(* CODESYS project kr_achse.library
   Title: Kr_Achse
   Version: 2.23.0.7
   Placeholder: Kr_Achse
   Company: Progress

Project tree, tasks and I/O mapping:
  libraries: Tc2_Standard, * (Beckhoff Automation GmbH)
  Data types/
    Achsen/
      data type TAchs_To_DriveAdapter
      data type TES_Achse_IN
      data type TES_Achse_OUT
      data type TIV_RB
      data type TKont_Achse_IN
      data type TKont_Achse_OUT
      data type TPDO_SI6_IN
      data type TPDO_SI6_OUT
      data type TPDO_SI6_V3_IN
      data type TPDO_SI6_V3_OUT
  POUs/
    Achsen_Bausteinen/
      Adapter/
        function block Adapter_Drive_Analog [ST]
        function block Adapter_Drive_BeckhoffEL7201 [ST]
        function block Adapter_Drive_MDS [ST]
        function block Adapter_Drive_SI6 [ST]
        function block Adapter_Drive_SI6_V3 [ST]
        function block Adapter_DriveBased_U [ST]
      FB/
        function block Bremsweg [FBD]
        function block calc_Rbist_inPhase3 [ST]
        function block calc_Val3_inPhase123 [ST]
        function block calc_Val567_inPhase45 [ST]
        function block calc_Val67_inPhase6 [ST]
        function block calc_Val7_inPhase7 [ST]
        function block CDLR [ST]
        function block Phase0 [FBD]
        function block Phase12 [FBD]
        function block Phase3 [FBD]
        function block Phase4 [FBD]
        function block Phase56 [FBD]
        function block Phase7 [FBD]
        function block switchPhase [ST]
        function block Trnsf1Lreal [ST]
      function block ES_AnalogIN [ST]
      function block ES_EL5001_A [ST]
      function block ES_EL5xx1_A [ST]
      function block ES_KL2552 [ST]
      function block ES_KL5001_A [ST]
      function block ES_KL51x1_A [ST]
      function block ES_M3120 [ST]
      function block KR_Achse_V2 [FBD]: encoder, ohne_RB, Regelung
    Nockenachsen/
      function block Nock_Incr_S_Achs [ST]
  Visualizations/
*)

// Data types/Achsen/TAchs_To_DriveAdapter
TYPE TAchs_To_DriveAdapter :
STRUCT
	motorSpeed:REAL; (*rpm*)
	SA_MotUmdr:REAL;(*Schleppabstand in Motorumdrehungen zur berechnung des IPM-Mod bei ext. Encoder  (Adapter_Drive_MDS_ExtEnc). !!! Der Schleppabstand beinhaltet schon das Vorzeichen aufgrund Achse Invers/ Not Invers !!! *)
END_STRUCT
END_TYPE

// Data types/Achsen/TES_Achse_IN
TYPE TES_Achse_IN :
STRUCT
(*#################### EingangsVariablen: NC-Baustein -> STRUKTUR(IN) -> ANWENDER-PRG. ###################################*)
	IstPos: LREAL;(*Istposition Achse *)
	SYNC: BOOL:= FALSE;
	STILL:BOOL;(*Stillstand:Dises Bit ist TRUE, wenn bei gesetztem Ausgang VOR(ZUR) der Istwert nicht größer (nicht kleiner) wird*)
	PEH:BOOL;(*Position erreicht: wird ausgegeben, solange sich der Antrieb innerhalb dem PEH-Fenster befindet*)
	RET_SollPos:LREAL;(*Rückmeldung der übergebenen Sollposition*)
	VEL_IST:REAL;(*Istwert der Geschwindigkeit: -2,-1,0,1,2 (schnell zurück, langsam zurück, steht, langsam vor, schnell vor*)
END_STRUCT
END_TYPE

// Data types/Achsen/TES_Achse_OUT
TYPE TES_Achse_OUT :
STRUCT
(*############ OUT-VARIABLEN: ANWENDER-PRG. -> STRUKTUR(OUT) -> NC-Baustein ################################*)
	MODULO:BOOL;(*Modulowert ermitteln, es müssen die Incrmente für Modulowert angegeben werden. Achtung:MODULO-Funktion wird vom Baustein nur gemacht, solange die Incrementezahl ( IstPos/IBW) kleiner den Grenzen eines DINT ist, andernfalls wird MOD ignoriert*)
	MODULOVAL_INC:REAL;(*Wert in Incrementen für MODULO-Funktion*)
	SETPOS:BOOL;(*Istposition auf "Refpos" setzen *)
	REF:BOOL; (*Anwahl der Referenzfahrt unter beachtung von REFVEL1,REFVEL2 (VAR_IN am FB) und Modus "REF_ON" *)
	Refpos: REAL; (*Wert für "REF" und "SETPOS" *)
	Start_Pos: BOOL;(*Start-Bit zur Positionierung. *)
	SollPos: LREAL;(*Zielposition bei Positionierung*)
	V_Pos:REAL:=2.0;(*Geschwindigkeit beim Positionieren: 1= nur schleich,2= EIL-Schleich
						!! bei Verwendung der DC-Klemme KL2552 als ES-Achse wird hier die Geschwindigkeit in % angegeben !! *)
	JOGFW: BOOL;(*Manuell vor*)
	JOGBW: BOOL;(*manuell zurück*)
	V_JOG: REAL:=1.0;(*manuelle Geschwindigkeit: 1=langsam, 2=schnell
					!! bei Verwendung der DC-Klemme KL2552 als ES-Achse wird hier die Geschwindigkeit in % angegeben !! Beim Positioniervorgang wird hier die Schleichgeschwindigkeit angegeben !!! *)
END_STRUCT
END_TYPE

// Data types/Achsen/TIV_RB
TYPE TIV_RB :
STRUCT
	Phase:INT;(*akutelle Phase: 0 = Stillstand / 1..7 = Fahrt vorwärts / -1..-7 = Fahrt rückwärts*)
	PhCng:INT;(*aktuelle Phase x100 /letztePhase x10 / Ursache des Phasenwechsels x1:

071=Phase 0 wurde aus Phase 7 eingeleitet
  da das Ziel mit VE7=0 erreicht war.
072=Phase 0 wurde aus Phase 7 eingeleitet
   da ACC=0 und VEL=0 waren, das Ziel war nicht erreicht oder es war nicht Start_Pos gesetzt 
073=Phase 0 wurde aus Phase 7 eingeleitet da Fehler in Phase 7 auftrat (Geschw. 0 oder ACC=0 wurde nicht erreicht

0X8 = Phase=0 aus PhaseX gesetzt da Ruck=0, Stillstand, 
  Fehler oder abbruch durch anderen Achsbefehl vorliegt

101=Phase 1 wurde aus Phase 0 eingeleitet da Ziel in positiver richtung liegt
102=Phase -1 wurde aus Phase 0 eingeleitet da Ziel in negativer richtung liegt

123=Phase 1 wurde aus Phase 2 eingeleitet da Acc höher geworden ist

131=Phase 1 wurde aus Phase 3 eingeleitet
  da weder Ziel noch VEL_Soll noch ACC_Soll erreicht ist/wird
141=Phase 1 wurde eingeleitet weil Sollgeschw. unterschritten war 


2x1=Phase 2 wurde eingeleitet da die Sollbeschleunigung erreicht ist
311=Phase 3 wurde aus Phase1 eingeleitet da VE3 den Wert für V_Pos erreicht hat
321=Phase 3 wurde aus Phase2 eingeleitet da VE3 den Wert für V_Pos erreicht hat

312=Phase 3 wurde aus Ph.1 eingeleitet da der Resverfahrweg aufgebraucht ist
322=Phase 3 wurde aus Ph.2 eingeleitet da der Resverfahrweg aufgebraucht ist

313=Phase 3 wurde aus Ph.1 eingeleitet da die 
323=Phase 3 wurde aus Ph.2 eingeleitet da die 
 Istbeschleunigung höher ist als die Vorgegebene ACC-Soll.

431=Phase 4 wurde aus Phase 3 eingeleitet
 da die Istbeschleunigung=0 ist
472=Phase 4 wurde aus Phase 7 eingeleitet
  da ACC_IST=0 aber VE7>0

541=Phase 5 wurde aus Phase 4 eingeleitet weil Zieldiff aufbegraucht war
542=Phase 5 wurde eingeleitet weil Sollgeschw. überschritten war 
563=Phase 5 wurde aus Phase 6 eingeleitet weil kein Befehl ansteht und (dadurch) die Bremsrampe steiler geworden ist
573=Phase 5 wurde aus Phase 7 eingeleitet weil VE7>0 und das Ziel überschritten würde
574=Phase 5 wurde aus Phase 7 eingeleitet weil VE7>0 und VE7>sollvel
535=Phase 5 wurde aus Phase 3 eingeleitet weil Restweg aufgebraucht war und ACC_IST im nächsten Zyklus < 0 war


651=Phase 6 wurde aus Phase 5 eingeleitet da die Soll-DCC erreicht war

751=Phase 7 wurde aus Ph.5 eingeleitet
 da VE7=0 erreicht wird (VE7 darf nicht neg. werden) 
761=Phase 7 wurde aus Ph.6 eingeleitet da
  da VE7=0 erreicht wird (VE7 darf nicht neg. werden) 
752=Phase 7 wurde aus Ph.5 eingeleitet da da nicht das Ziel, aber da die Sollgeschwindigkeit VE7=V_Soll und VE7>0 erreicht wird (Online-Änder. von V_soll durch niedrigeren Wert)
762=Phase 7 wurde aus Ph.6 eingeleitet da da nicht das Ziel, aber da die Sollgeschwindigkeit VE7=V_Soll und VE7>0 erreicht wird (Online-Änder. von V_soll durch niedrigeren Wert)
753=Phase 7 wurde aus Ph.5 eingeleitet da da nicht das Ziel, aber da die Sollbeschleunigung überschritten ist
763=Phase 7 wurde aus Ph.6 eingeleitet da da nicht das Ziel, aber da die Sollbeschleunigung überschritten ist

*)
	FL_PhChnge:BOOL;(*Flanke Phasenänderung *)
	VSoll_Ph4_ok:BOOL;(* Der Merker besagt: V-Soll wird in Phase 4 exackt erreicht, denn die vorausichtliche Endgeschwindigkeit VE3 überstieg in Phase 1 oder 2 für
min. 1Zyklus nicht V_Soll, diese wurde anschliessend nicht mehr geändert und die Phase 3 wurde wegen erreichen von VE3>=V_Soll eingeleitet. In Phase3 wurde ebenso 
nie V_Soll geändert.D.h. in Phase 3 wird Die Endgeschw. VE3= V4sein. Die Infomation ist notwendig um in Phase4 die VEL_IST der V_Soll gleichsetzen zu können
Ähnlich verhält es sich wenn eine niedrigere Geschwindigkeit in Phase 5 angefahren wird, das Ende der Phase5 schliesst dann in Phase4 mit V_Soll=Vel_IST an*)
	P_T:LREAL;
	VEL_IST:LREAL;
	ACC_IST:LREAL;
	VEL_IST_LAST:LREAL;
	ACC_IST_Last:LREAL;
	Sollpos_Return:LREAL;(*Die Sollosition wird übernommen: Bei Phase ><0:  wenn das Ziel nicht überfahren wird / aus Phase0 heraus bei Start_Pos *)
	ZielDiff: LREAL;(*Die Zieldiff ist die Differenz zum Ziel in Fahrtrichtung ( neg= Ziel wurde überfahren).
Sie wird im Positioniermodus aus der Sollposition, bei Jog aus LimitposJog berechnet.
Zieldiff=0 steht auch für "kein Befehl - Stoppen"*)
	SollVel_ubrn:LREAL;
	SollAcc_ubrn:LREAL;
	SollDcc_ubrn:LREAL;
	SollRb_ubrn:LREAL;
	StartPos_ubrn:BOOL;(*Zielfahrt läuft (Positionierung) wurde übernommen*)
	Jog_ubrn:BOOL; (* Jog vorwärts oder rückwärts(auch Referenzfahrt) *)
	Err_ID:LREAL;(*Fehler-Nr (vorkomma)  in Phase (nachkomma). Siehe Beschreibung in TKont_Achse_IN. positiver Fehler führen zum Abbremsen und Schnellhalt ohne Ruckbegrenzung*)
	PosTime:LREAL;(*Restzeit beim positionieren bis zum Erreichen des Zieles . -1 = unbekannt*)
	BrakingDist:LREAL;(*Bremsweg bei Wegnahme aller Befehle mit aktueller Deccel  und RB*)
	BrakingTime:LREAL;(*Bremszeit bei Wegnahme aller Befehle mit aktueller Deccel  und RB*)
	HalfBreakErrorWay:LREAL;(* Der halbe BremsfehlerWeg ist die halbe Differenz der Bremswegänderung zwischen 2 Zyklen, Vorzeichenbehaftet, d.h. + Bremsweg wird grösser / - Bremsweg wird kleiner *)
	ErrorWay:LREAL;(*Der höchste Fehler-Weg (Absolutwert, immer positiv) der während einer Phase<>0 aufgetreten ist, er setzt sich zusammen aus dem gefahrenen Weg zwischen 2 Zyklen + BremsfehlerWeg*)
	ErrorVel:LREAL;(*Die Geschwindigkeitsdifferenz die aufgrund der höchsten aufgetrenden Beschleunigung  in Latenzzeit erreicht wurde*)
	HalfCyklWay:LREAL;(*Der Weg der aufgrund der aktuellen Geschwindigkeit in 1/2 Zykluszeit zurückgelegt würde, Absoluter Wert*)
	HalfCyklVelDiff:LREAL;(*Die Geschwindigkeitsdfifferenz aufgrund der  Beschleunigung in einem  1/2 Zyklus. Vorzeichenbehaftet!!! HalfCyklVelDiff=ACC_IST*T_Zykl/2: pos: Geschwindigkeitsbetrag wird größer / neg=wird kleiner*)

	PhasenCalc_done:BOOL;	(*Berechnungen von AccIst und VelIst für diesen Zyklus wurden gemacht  - keinen weiteren Phasen-FB bearbeiten *)
	LimitPosJog_activ:BOOL;(* die Limitpos_Jog ist aktiv: Achse hält im Jog-Modus an vor der angegebenen Grenze*)
	T_Zykl:LREAL;

END_STRUCT
END_TYPE

// Data types/Achsen/TKont_Achse_IN
TYPE TKont_Achse_IN :
STRUCT
(*#################### EingangsVariablen: NC-Baustein -> STRUKTUR(IN) -> ANWENDER-PRG. ###################################*)
	IstPos: LREAL;(*Istposition Achse *)
	SYNC: BOOL := FALSE;(*Achse ist referenziert. SYNC wird gelöscht, wenn REF-Modus angewählt wird*)
	Schleppabst: REAL;(*aktueller Schleppabstand in mm*)
	PEH:BOOL;(*Position erreicht,PEH-Fenster am FB als Parameter übergeben!! PEH wird bei Positioniermodus und bei REF-Modus ausgegeben*)
	RET_SollPos:LREAL;(*Rückmeldung der übergebenen Sollposition. Wird mit Ruckbegrenzung positioniert, dann wird die Sollposition nur zurückgemeldet, sofern sie angefahren kann. Das bedeutet: wird während dem Positioniervorgang eine neue Sollposition übergeben, aber diese nicht in RET_SollPos zurückgemeldet, war eine online-Zieländerung nicht möglich . Der Antrieb fährt dann das alte Ziel an, gibt nach erreichen des alten Zieles und Stillstand die neue Sollposition aus(nicht PEH) und fährt diese an. *)
	ACC_IST:REAL;(*Istwert der Beschleunigung, positiv=Beschleunigen, negativ=Bremsen*)
	VEL_IST:REAL;(*Istwert der Geschwindigkeit, positiv oder negativ*)
	Err_ID:INT;(*Fehler-Nr .
 positiver Fehler führen zum Abbremsen und Schnellhalt ohne Ruckbegrenzung
Err_ID <> 0 bleibt erhalten bis alle Befehle (Start, Jog) zurückgenommen wurden und die Achse im Stillstand ist.
	1=ungültige Geschwindigkeit
	2=ungültige Beschleunigung
	3=ungültige verzögerung
	4=ungültige Ruckbegrenzung
	5=doppelbefehl
	6=Abbruch der Positionierung in Phase1 da der Restweg kleiner als der theoretische Weg in einem Zyklus ist
	7=Watchdog: Ruckbegrenzung wurde überschritten
	8=Watchdog: Beschleunigung (Hochlauframpe) wurde überschritten
	9=Watchdog: Verzögerung (Bremsrampe) wurde überschritten
	-10=zu Hohe Ruckbegrenzung: die Ruckbegrenzung muss mindestens 10 Zyklen aktiv sein bis zum erreichen der Endbeschleunigung! - Die Positionierung wird ohne Ruckbegrenzung ausgeführt
	-11=Geschwindigkeitsdifferenz bei Übergang in Phase 4 überschreitet zulässiges Maximum. Die Istgeschw. wird nicht =Sollgeschwindigkeit gesetzt.
	12=Die entfernteste übergeben Zielposition wäre mit Ruckbegrenzung überschritten worden 
	13=Geschwindigkeitsvorzeichen stimmt nicht mit Phasenvorzeichung überein
	14=Fehler in Phase7: Es wird nicht Ruckbegrenzt abgebremst

	100=Fehlerhafte parametrierung der Eingangswerte VAR_INPUT am FB
	101=Unzulaessiger Istwertoffset
		*)
	Err_in_Phase:INT;(*Phase, in welcher der Fehler (Err_ID) aufgetreten ist*)
	PosTime:LREAL;(*Restzeit beim positionieren bis zum Erreichen des Zieles . -1 = unbekannt*)
	BrakingDist:LREAL;(*Bremsweg im Positioniermodus oder im Jog-Modus*)
	BrakingTime:LREAL;(*Bremszeit im Positioniermodus oder im Jog-Modus*)
	Phase:INT;
	P_T:LREAL;
END_STRUCT
END_TYPE

// Data types/Achsen/TKont_Achse_OUT
TYPE TKont_Achse_OUT :
STRUCT
(*############ OUT-VARIABLEN: ANWENDER-PRG. -> STRUKTUR(OUT) -> NC-Baustein ################################*)
	RESET: BOOL;(*Reset: setzt den Schleppabstand auf 0, somit findet keine Lageregelung mit KV-Faktor statt. Unterbricht das Positionieren mit Ruckbegrenzung (Antrieb fährt ohne Ruckbegrenzung weiter, positionieren, Jog oder Ref). Kann unabhängig zu allen Fahrbefehlen gesetzt werden *)
	SETPOS:BOOL;(* Istposition setzen: der Schleppabstand wird auf 0 gesetzt und die Istposition auf"REFPOS", solange SETPOS TRUE ist.Achse fährt ohne Ruckbegrenzung weiter. Hat keine Funktion bei KR_MDS_Ethercat wenn Incrementalgeber=false*)
	REF:BOOL;(*Referenzfahrt ausführen.Die beiden Referenzgeschwindigkeiten (REFVEL1=zum suchen des Endschalters, REFVEL2=zum
				suchen der Nullspur)müssen am FB der Achse als Eingangsparameter übergeben werden. !! ACHTUNG: Nachdem bei 
				Angewählter "REF" die Achse "SYNC" gesetzt hat, fährt sie mit "REFVEL2" und "ACC_SJR" auf Zielposition= "Refpos"
				und gibt bei erreichen von "Refpos" "PEH" aus. Wird "REF" mit setzen von "SYNC" weggenommen, bremst die Achse mit
				"ACC_SJR"  bis zum Stillstand ab und bleibt stehen.Hat keine Funktion wenn Incrementalgeber=false*)
	Refpos: REAL; (*Istwert bei Modus REF oder SETPOS*)
	Start_Pos: BOOL;(*Start-Bit zur Positionierung. Achtung: wird bei Ruckbegrenztem Positioniervorgang Start weggenommen, Bremst der Antrieb erst ab, nachdem er die Positionier-Geschwindigkeit erreicht hat. Soll er sofort ohne Ruckbegrenzung abbremsen, muß "RESET" für mind. 1 Zyklus gesetzt werden.*)
	SollPos: LREAL;(*Zielposition bei Positionierung. Das Ziel kann während der Positionierung geändert werden. Das neue Ziel wird sofort angefahren, außer beim Positionieren mit Ruckbegtenzung. In diesem Fall hat die Achse die neue Position übernommen, wenn sie in "Sollpos.RET" die neue Position zurückmeldet *)
	V_Pos:REAL:=500;(*Geschwindigkeit beim Positionieren, sie kann während der Positionierung geändert werden*)
	ACC_Pos: REAL:=300;(*Beschleunigung beim positionieren, sie kann während der Positionierung geändert werden*)
	DCC_Pos: REAL:=300;(*Verzögerung beim positionieren  sie kann während der Positionierung geändert werden*)
	JOGFW: BOOL; (*Hand-Betrieb vor, mit V_JOG*)
	JOGBW: BOOL; (*Hand-Betrieb zurück, mit V_JOG*)
	V_JOG: REAL; (*Geschwindigkeit bei Handbetrieb, sie kann während der Positionierung geändert werden*)
	ACC_JR: REAL:=800;(*Beschleunigung im Jog-Modus und bei Referenzfahrt*)
	DCC_JRS: REAL:=800;(*Verzögerung  im Jog-Modus, bei Referenzfahrt und beim Anhalten ohne Ruckbegrenzung*)

	RB:LREAL;(*Ruckbegrenzung. Sie wird nur in Phase 0 (im Stillstand der Achse) übernommen oder in jeder Phase wenn RB=0 ist, dann wird nicht RB-Begrenzt weiterpositioniert. RB kann jederzeit geändert werden.*)
	LimitposJog:LREAL:=1E100;(*Die Limit-pos Jog bietet die Möglichkeit, im Jog-Betrieb exackt an der angegebenen Position anzuhalten. Die Achse fährt im Jog-Betrieb nur, wenn die LimitposJog in Fahrtrichtung liegt. Der Initialwert 1E100 bedeutet, dass die Funktion deaktiviert ist (Achse hält nicht an)*)
	IstWertOffset:LREAL;(*Offset, der  auf dem Istwert(Benutzereinheit bzw. mm) Online aufgerechnent wird. Bei Absolutgebern (Incrementalgeber=false) wird der Offset in Incremente
						umgerechnet und addiert, sodass ein Geber-Überschlag intern ausserhalb den Verfahrbereich verschoben wird*)
END_STRUCT
END_TYPE

// Data types/Achsen/TPDO_SI6_IN
{attribute 'pack_mode' := '1'}
TYPE TPDO_SI6_IN :
(*
	IO Struktur für SI6-Achsen
*)
STRUCT
	A516_StatusWord:WORD;	(*
	BIT:
		0 Ready to switch on 
		1 Switched on 
		2 Operation enabled 
		3 Fault 
		4 Voltage enabled 
		5 Quick stop (1 = Kein Schnellhalt aktiv )
		6 Switch on disabled 
		7 Warning 
*)
	A545_AktPosition:DINT;	(*Aktuelle Position [inc]*)
	A632_SchleppFehler:DINT;	(*Aktueller Schleppfehler [inc]*)
	E00_I_Motor:REAL;		(*Aktueller Strom [A]*)
	E03_UZK:REAL;			(*Aktuelle Zwischenkreisspannung [V]*)
	E15_AktVel:REAL;			(*Aktuelle Geschwindigkeit [U/m]*)
	E43_ErrUrsache:SINT;		(*Ursache für das zuletzt aufgetretene Ereignis E82*)
	E48_GerateStatus:SINT;	(*Zustand des Umrichters
		0 Selbsttest 
		1 Einschaltsperre 
		2 Einschaltbereit 
		3 Eingeschaltet 
		4 Freigegeben 
		5 Störung 
		6 Störungsreaktion 
		7 Schnellhalt 
*)
	E82_ErrArt:SINT;			(*Anzeige des aktuelle aktiven Ereignises/Störung*)
	E90_AktMoment:REAL;	(*Aktuelles Moment im Bezug auf C09 [0.01%]*)
END_STRUCT
END_TYPE

// Data types/Achsen/TPDO_SI6_OUT
{attribute 'pack_mode' := '1'}
TYPE TPDO_SI6_OUT :
(*
	IO Struktur für SI6-Achsen
*)
STRUCT

	A515_ControlWord:WORD;	(*
	BIT:
		0 Switch on 
		1 Enable voltage 
		2 Quick stop	(0 = Schnellhalt angefordert; 1 = Kein Schnellhalt angefordert )
		3 Enable operation 
		4– 6: Operation mode specific * 
		8 Halt
		9
		10
		11 Bit0 Parameterumschaltung
		12 Bit1 Paramterumschaltung 
		13 Anforderung Paramterumschaltung aktivieren
*)
	A559_MaxTorque:WORD:=1500;	(*Maximal zulässiges Drehmoment  [0.1%]  (In E65/E66 kann das effektive maximale Moment ausgelesen werden) *)
	A567_TargetPos:DINT;		(*Sollposition für Controllerbased-Achsen (OP-Mode 8) [inc]*)
	A638_TargetVel:DINT;		(*Sollgeschwindigkeit für Drivebased-Achsen (OP-Mode 3) [inc/s]*)
	A541_OpMode:BYTE;		(*Operationsmodus*)

END_STRUCT
END_TYPE

// Data types/Achsen/TPDO_SI6_V3_IN
{attribute 'pack_mode' := '1'}
TYPE TPDO_SI6_V3_IN :
(*
	IO Struktur für SI6-Achsen
*)
STRUCT
	A516_StatusWord:WORD;	(*
	BIT:
		0 Ready to switch on 
		1 Switched on 
		2 Operation enabled 
		3 Fault 
		4 Voltage enabled 
		5 Quick stop (1 = Kein Schnellhalt aktiv )
		6 Switch on disabled 
		7 Warning 
*)
	A545_AktPosition:DINT;	(*Aktuelle Position [inc]*)
	A595_Rot_Touch_Probe_Status :WORD;	(*
	BIT:
		0 Touch Probe enabled
		1  Positive Flanke erkannt
		2 Negative Flanke erkannt
*)
	E00_I_Motor:REAL;		(*Aktueller Strom [A]*)
	E15_AktVel:REAL;			(*Aktuelle Geschwindigkeit [upm]*)
	E22_i2t_Umrichter :REAL;	(*i2t Umrichter [%]*)
	E23_i2t_Motor :REAL;		(*i2t Motor [%]*)
	E43_ErrUrsache:SINT;		(*Ursache für das zuletzt aufgetretene Ereignis E82*)
	E48_GerateStatus:SINT;	(*Zustand des Umrichters
		0 Selbsttest 
		1 Einschaltsperre 
		2 Einschaltbereit 
		3 Eingeschaltet 
		4 Freigegeben 
		5 Störung 
		6 Störungsreaktion 
		7 Schnellhalt 
*)
	E82_ErrArt:SINT;			(*Anzeige des aktuelle aktiven Ereignises/Störung*)
	E90_AktMoment:REAL;	(*Aktuelles Moment im Bezug auf C09 [0.01%]*)
	E201_Statusword2 : WORD; (*
	BIT: 
		0: Betriebsbereitschaft (Quelle: E79[0]: 1 = Konfiguration aktiv, Selbsttest nicht aktiv, keine Störung und keine Störungsreaktion) 
		1: Betriebsbereitschaft (Quelle: E79[1]: 1 = Konfiguration aktiv, Selbsttest nicht aktiv, Anlaufsperre ok (Zustand <> Einschaltsperre), keine Störung und keine Störungsreaktion) 
		2: Betriebsbereitschaft (Quelle: E79[2]: 1 = Selbsttest nicht aktiv)
		3: Bremse eingefallen (Quelle: F08[0], gegebenenfalls übersteuert durch Sicherheitsmodul) 0 = Bremse nicht einfallend angesteuert oder einfallend angesteuert, Einfallzeit ist noch nicht abgelaufen; 1 = Bremse einfallend angesteuert, Einfallzeit ist abgelaufen (F05) 
		4: Bremse gelüftet (Quelle: F09[0], gegebenenfalls übersteuert durch Sicherheitsmodul) 0 = Bremse nicht lüftend angesteuert oder lüftend angesteuert, Lüftzeit ist nicht abgelaufen; 1 = Bremse lüftend angesteuert, Lüftzeit ist abgelaufen (F04) 
		5: Sollwertbereit (Quelle: I97: 1= Status "Freigegeben", Bremse ist gelüftet und bei Asynchronmotoren ist die Magnetisierung aufgebaut. Es liegt kein Halt oder Schnellhalt vor. ) 
		6: Tippen aktiv 
		7: Wirksames Signal Positiver Hardware-Endschalter (Quelle: I805)
		8: Wirksames Signal Negativer Hardware-Endschalter (Quelle: I806) 
		9: In Referenz (Quelle: I86) 
		10: STO	
		11: SS1
		12: SS2
*)
END_STRUCT
END_TYPE

// Data types/Achsen/TPDO_SI6_V3_OUT
{attribute 'pack_mode' := '1'}
TYPE TPDO_SI6_V3_OUT :
(*
	IO Struktur für SI6-Achsen
*)
STRUCT

	A515_ControlWord:WORD;	(*
	BIT:
		0 Switch on 
		1 Enable voltage 
		2 Quick stop	(0 = Schnellhalt angefordert; 1 = Kein Schnellhalt angefordert )
		3 Enable operation 
		4– 6: Operation mode specific * 
		8 Halt
		9
		10
		11 Bit0 Parameterumschaltung
		12 Bit1 Paramterumschaltung 
		13 Anforderung Paramterumschaltung aktivieren
*)
	A541_OpMode:BYTE;		(*Operationsmodus*)
	A559_MaxTorque:WORD:=1500;	(*Maximal zulässiges Drehmoment  [0.1%]  (In E65/E66 kann das effektive maximale Moment ausgelesen werden) *)
	A567_TargetPos:DINT;		(*Sollposition für Controllerbased-Achsen (OP-Mode 8) [inc]*)
	A594_Rot_Touch_Probe_Function:WORD;	(*
	BIT:
		0 = enable Touch Probe
		1  = Trigger type (0=bei erstem Flankenwechsel; 1=bei jedem Flankenwechsel)
		2 = Trigger source (0=Binärsignal I110; 1=Nullimpuls des Positionsencoders)
		3 	
		4 = Positive Edge  (Flankenerkennung aktivieren)
		5 = Negative Edge (Flankenerkennung aktivieren)
*)
	A638_TargetVel:DINT;		(*Sollgeschwindigkeit für Drivebased-Achsen (OP-Mode 3) [inc/s]*)
END_STRUCT
END_TYPE

// POUs/Achsen_Bausteinen/Adapter/Adapter_Drive_Analog
FUNCTION_BLOCK Adapter_Drive_Analog(*Adapter für  Analoge Ausgangsklemme
 *)
VAR
END_VAR
VAR_INPUT
	DriveAdapter_from_Achs:TAchs_To_DriveAdapter;
	nMax_Motor:REAL:=3000.0;(*Maximaldrehzahl in upm für Skalierung.durch Angabe eines negativen Wertes wird der Drehzahlsollwert invertiert *)
END_VAR
VAR_OUTPUT
	U_Out: INT; (*Output Int*)
END_VAR

U_Out:=REAL_TO_INT(LIMIT(-32767,(32767*DriveAdapter_from_Achs.motorSpeed/nMax_Motor),32767));

END_FUNCTION_BLOCK

// POUs/Achsen_Bausteinen/Adapter/Adapter_Drive_BeckhoffEL7201
FUNCTION_BLOCK Adapter_Drive_BeckhoffEL7201 (*Adapter für Beckhoff Servomotorklemme EL7201
 *)
VAR
END_VAR
VAR_INPUT
	DriveAdapter_from_Achs:TAchs_To_DriveAdapter;
	VelEncRes_9010_14:REAL:=268435; (*Velocity encoder resolution in CoE 9010:14*)
	nMax_Motor:REAL:=1000.0;(*Maximaldrehzahl in upm für Skalierung.durch Angabe eines negativen Wertes wird der Drehzahlsollwert invertiert *)
END_VAR
VAR_OUTPUT
	TargetVel: DINT; (*Target Velocity*)
END_VAR

TargetVel:=REAL_TO_DINT(
	LIMIT(
		-1,
		DriveAdapter_from_Achs.motorSpeed / nMax_Motor,
		1
	)*VelEncRes_9010_14*nMax_Motor/60
);

END_FUNCTION_BLOCK

// POUs/Achsen_Bausteinen/Adapter/Adapter_Drive_MDS
FUNCTION_BLOCK Adapter_Drive_MDS (*Adapter für MDS-Umrichter (Option IPM-Mode)
 *)
VAR
END_VAR
VAR_INPUT
	DriveAdapter_from_Achs:TAchs_To_DriveAdapter;
	D02_nMax_Motor:REAL:=3000.0;(*Maximaldrehzahl in upm für Skalierung.durch Angabe eines negativen Wertes wird der Drehzahlsollwert invertiert *)
	E153_EngineCounterVal: DWORD;(* Counter-Wert E153. Der Wert wird zur Berechnung von "I421_TargetPos" herangezogen. Nur bei IPM-Mod relevant, wird "I421_TargetPos" des Umrichters nicht verwendet, bracuh hier nichts parametriert zu werden!*)
	IncPerTurnEngine: DWORD;(*Impulse / Motroumdrehung des Motorgebers. Bei EnDat ist 10_0000H anzugeben. Der Wert wird zur Berechnung von "I421_TargetPos" herangezogen. Nur bei IPM-Mod relevant, wird "I421_TargetPos" des Umrichters nicht verwendet, bracuh hier nichts parametriert zu werden!*)
END_VAR
VAR_OUTPUT
	D230_nSoll: INT;
	I421_TargetPos: DWORD;
END_VAR

D230_nSoll:=REAL_TO_INT(LIMIT(-16384,(16384*DriveAdapter_from_Achs.motorSpeed/D02_nMax_Motor),16384));

IF D02_nMax_Motor>0 THEN
	I421_TargetPos:=E153_EngineCounterVal+REAL_TO_DWORD(DriveAdapter_from_Achs.SA_MotUmdr*DWORD_TO_REAL(IncPerTurnEngine));
ELSE
	I421_TargetPos:=E153_EngineCounterVal-REAL_TO_DWORD(DriveAdapter_from_Achs.SA_MotUmdr*DWORD_TO_REAL(IncPerTurnEngine));
END_IF

END_FUNCTION_BLOCK

// POUs/Achsen_Bausteinen/Adapter/Adapter_Drive_SI6
FUNCTION_BLOCK Adapter_Drive_SI6 (*Adapter für SI6-Umrichter (Drive und Controllerbased)	*)
VAR
END_VAR
VAR_INPUT
	DriveAdapter_from_Achs:TAchs_To_DriveAdapter;
	B13_nMax_Motor:REAL:=3000.0;(*Maximaldrehzahl in Upm für Skalierung.durch Angabe eines negativen Wertes wird der Drehzahlsollwert invertiert *)
	A585_IncPerTurnEngine: DWORD;(*Impulse / Motroumdrehung des Motorgebers*)
	A559_MaxTorque:WORD:=1500;	(*Maximales Drehmoment [0.1%]*)
END_VAR
VAR_IN_OUT
	Achs_IO_IN :TPDO_SI6_IN;				(*Verknüpfung zu de IN-Struktur der Achse*)
	Achs_IO_OUT :TPDO_SI6_OUT;			(*Verknüpfung zu de OUT-Struktur der Achse*)
END_VAR

Achs_IO_OUT.A638_TargetVel:=REAL_TO_DINT(LIMIT(((DriveAdapter_from_Achs.motorSpeed/60.0) *DWORD_TO_REAL(A585_IncPerTurnEngine)), -ABS((B13_nMax_Motor/60.0)*DWORD_TO_REAL(A585_IncPerTurnEngine)), ABS((B13_nMax_Motor/60.0)*DWORD_TO_REAL(A585_IncPerTurnEngine))));

IF B13_nMax_Motor>0 THEN
	Achs_IO_OUT.A567_TargetPos:=Achs_IO_IN.A545_AktPosition + REAL_TO_DINT(LIMIT(-2147483648, DriveAdapter_from_Achs.SA_MotUmdr*DWORD_TO_REAL(A585_IncPerTurnEngine), 2147483647));
ELSE
	Achs_IO_OUT.A567_TargetPos:=Achs_IO_IN.A545_AktPosition - REAL_TO_DINT(LIMIT(-2147483648 ,DriveAdapter_from_Achs.SA_MotUmdr*DWORD_TO_REAL(A585_IncPerTurnEngine), 2147483647));
END_IF

Achs_IO_OUT.A559_MaxTorque := A559_MaxTorque;

END_FUNCTION_BLOCK

// POUs/Achsen_Bausteinen/Adapter/Adapter_Drive_SI6_V3
FUNCTION_BLOCK Adapter_Drive_SI6_V3 (*Adapter für SI6-Umrichter (Drive und Controllerbased)	*)
VAR
END_VAR
VAR_INPUT
	DriveAdapter_from_Achs:TAchs_To_DriveAdapter;
	B13_nMax_Motor:REAL:=3000.0;(*Maximaldrehzahl in Upm für Skalierung.durch Angabe eines negativen Wertes wird der Drehzahlsollwert invertiert *)
	A585_IncPerTurnEngine: DWORD;(*Impulse / Motroumdrehung des Motorgebers*)
END_VAR
VAR_IN_OUT
	Achs_IO_IN :TPDO_SI6_V3_IN;				(*Verknüpfung zu de IN-Struktur der Achse*)
	Achs_IO_OUT :TPDO_SI6_V3_OUT;			(*Verknüpfung zu de OUT-Struktur der Achse*)
END_VAR

Achs_IO_OUT.A638_TargetVel:=REAL_TO_DINT(LIMIT(((DriveAdapter_from_Achs.motorSpeed/60.0) *DWORD_TO_REAL(A585_IncPerTurnEngine)), -ABS((B13_nMax_Motor/60.0)*DWORD_TO_REAL(A585_IncPerTurnEngine)), ABS((B13_nMax_Motor/60.0)*DWORD_TO_REAL(A585_IncPerTurnEngine))));

IF B13_nMax_Motor>0 THEN
	Achs_IO_OUT.A567_TargetPos:=Achs_IO_IN.A545_AktPosition + REAL_TO_DINT(LIMIT(-2147483648, DriveAdapter_from_Achs.SA_MotUmdr*DWORD_TO_REAL(A585_IncPerTurnEngine), 2147483647));
ELSE
	Achs_IO_OUT.A567_TargetPos:=Achs_IO_IN.A545_AktPosition - REAL_TO_DINT(LIMIT(-2147483648 ,DriveAdapter_from_Achs.SA_MotUmdr*DWORD_TO_REAL(A585_IncPerTurnEngine), 2147483647));
END_IF

END_FUNCTION_BLOCK

// POUs/Achsen_Bausteinen/Adapter/Adapter_DriveBased_U
FUNCTION_BLOCK Adapter_DriveBased_U (*Universal-Adapter für Umrichter Drive-based (z.b. AX5000 Beckhoff
V1.0 30.08.2018 WLA. *)
VAR
END_VAR
VAR_INPUT
	DriveAdapter_from_Achs:TAchs_To_DriveAdapter;
	nMax_Motor:REAL;(*Maximaldrehzahl in Upm für Skalierung.durch Angabe eines negativen Wertes wird der Drehzahlsollwert invertiert. Der Sollwert wird auch auf diesen Wert limitiert *)
	Skale_dig_p_rpm: REAL;	(*Drivebased Skalierung: Einheit in Digit/rpm für Targvel (=Digits für 1 Umdrehung pro Minute*)
END_VAR

VAR_OUTPUT
	Targvel: DINT;
END_VAR

Targvel:=REAL_TO_DINT(LIMIT((DriveAdapter_from_Achs.motorSpeed *Skale_dig_p_rpm), -ABS(nMax_Motor*Skale_dig_p_rpm), ABS(nMax_Motor*Skale_dig_p_rpm)));

END_FUNCTION_BLOCK

// POUs/Achsen_Bausteinen/FB/Bremsweg
FUNCTION_BLOCK Bremsweg(*Bremsweg berechnet den aktuellen Bremsweg. Das Ergebnis versteht sich für
den Fall das  sofort Phase 3 ->5 -> 6 -> 7 eingeleitet wird.*)
VAR_INPUT
	Vel_Ist:LREAL; (*das Vorzeichen hat keine Relevanz da ABS gebildet wird *)
	Acc_Ist:LREAL; (*Beschleunigung vorzeichenbehaftet: neg=verzögerung*)
	Dcc_Max: LREAL;(*maximale verzögerung vom Anwender; positiver Wert!!*)
	RB:LREAL;(*Ruckbegrenzung mm/s^3*)
	Phase: INT;(*0..7*)
	ErrorVel_in_P7: LREAL;(*Der Wert ist für die Entscheidung Notwendig, ob nach Phase 7 Geschwindigkeit=0=Stop erreicht wird (VE7A<=ErrorVel_in_P7) oder
ob der VE7A >0 (VE7A>ErrorVel_in_P7) ist und nochmal Phase 5-6-7 folgen. In diesem Fall werhäht sich T_Brems und S_Brems entsprechend*)
END_VAR
VAR_OUTPUT
	s_Brems:LREAL;
	t_brems:LREAL;
	VE3A_inPhase123: LREAL;(*VE3A_inPhase123 ist die Geschwindigkeit ABS(VE3) in Phase 1,2 oder 3 die beim einleiten der Phase3 erreicht würde*)
	VE7A_inPhase7: LREAL;
END_VAR
VAR
	Val3: calc_Val3_inPhase123;
	Val567: calc_Val567_inPhase45;
	Val67: calc_Val67_inPhase6;
	Val7: calc_Val7_inPhase7;
	Abs_Phase: INT;
END_VAR
VAR // added by the converter: edge detectors and wires of the graphical bodies
    _w1 : ANY;
END_VAR

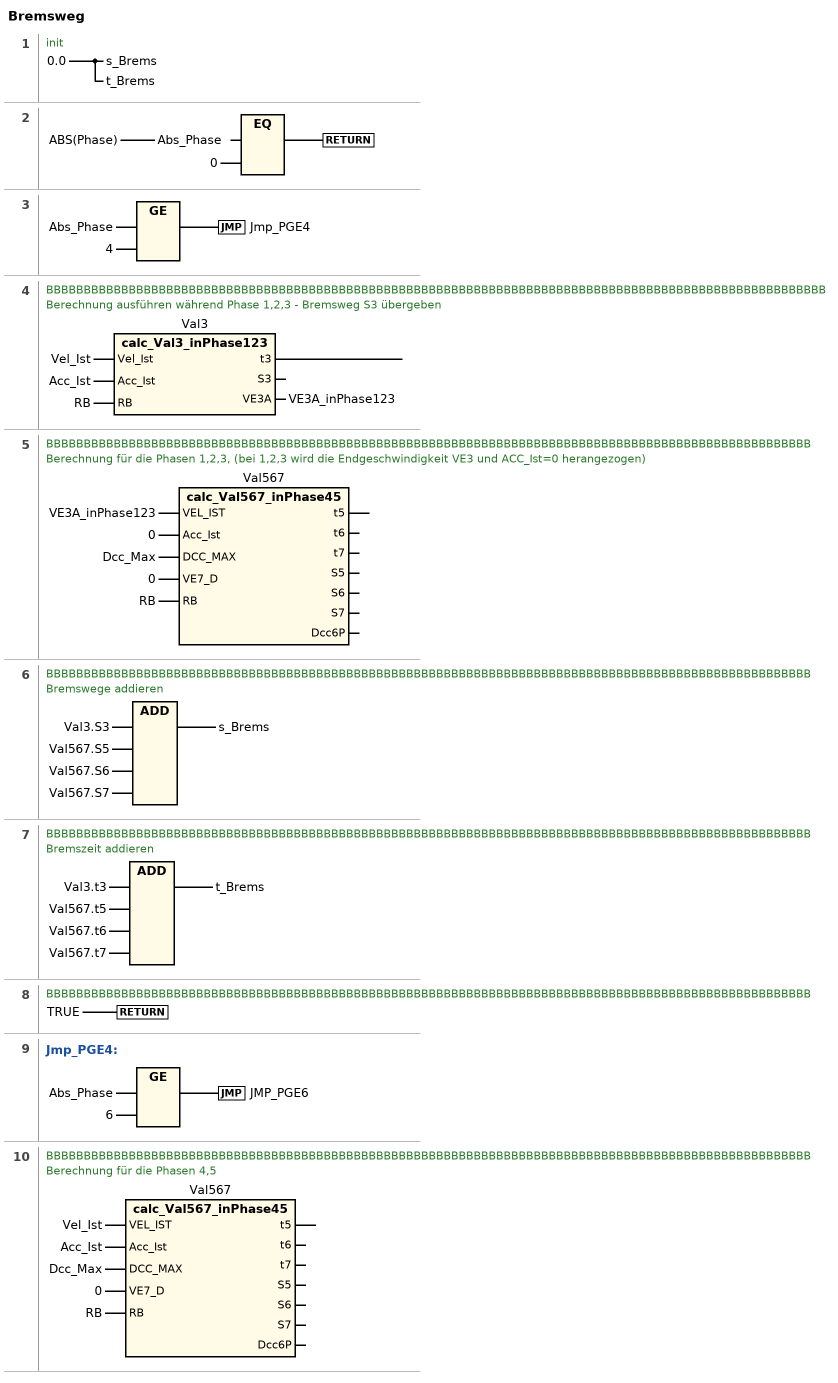
// NETWORK 1
// init
s_Brems := 0.0;
t_Brems := 0.0;

// NETWORK 2
_w1 := ABS(Phase);
Abs_Phase := _w1;
IF _w1 = 0 THEN RETURN; END_IF

// NETWORK 3
IF Abs_Phase >= 4 THEN JMP Jmp_PGE4; END_IF

// NETWORK 4
// 					BBBBBBBBBBBBBBBBBBBBBBBBBBBBBBBBBBBBBBBBBBBBBBBBBBBBBBBBBBBBBBBBBBBBBBBBBBBBBBBBBBBBBBBBBBBBBBBBBBBBBBBB
// Berechnung ausführen während Phase 1,2,3 - Bremsweg S3 übergeben
//
Val3(Vel_Ist := Vel_Ist, Acc_Ist := Acc_Ist, RB := RB, VE3A => VE3A_inPhase123); // calc_Val3_inPhase123

// NETWORK 5
// 					BBBBBBBBBBBBBBBBBBBBBBBBBBBBBBBBBBBBBBBBBBBBBBBBBBBBBBBBBBBBBBBBBBBBBBBBBBBBBBBBBBBBBBBBBBBBBBBBBBBBBB
// Berechnung für die Phasen 1,2,3, (bei 1,2,3 wird die Endgeschwindigkeit VE3 und ACC_Ist=0 herangezogen)
//
Val567(VEL_IST := VE3A_inPhase123, Acc_Ist := 0, DCC_MAX := Dcc_Max, VE7_D := 0, RB := RB); // calc_Val567_inPhase45

// NETWORK 6
// 					BBBBBBBBBBBBBBBBBBBBBBBBBBBBBBBBBBBBBBBBBBBBBBBBBBBBBBBBBBBBBBBBBBBBBBBBBBBBBBBBBBBBBBBBBBBBBBBBBBBBBB
// Bremswege addieren
//
s_Brems := Val3.S3 + Val567.S5 + Val567.S6 + Val567.S7;

// NETWORK 7
// 					BBBBBBBBBBBBBBBBBBBBBBBBBBBBBBBBBBBBBBBBBBBBBBBBBBBBBBBBBBBBBBBBBBBBBBBBBBBBBBBBBBBBBBBBBBBBBBBBBBBBBB
// Bremszeit addieren
//
t_Brems := Val3.t3 + Val567.t5 + Val567.t6 + Val567.t7;

// NETWORK 8
// 					BBBBBBBBBBBBBBBBBBBBBBBBBBBBBBBBBBBBBBBBBBBBBBBBBBBBBBBBBBBBBBBBBBBBBBBBBBBBBBBBBBBBBBBBBBBBBBBBBBBBBB
//
//
RETURN;

// NETWORK 9
Jmp_PGE4:
IF Abs_Phase >= 6 THEN JMP JMP_PGE6; END_IF

// NETWORK 10
// 					BBBBBBBBBBBBBBBBBBBBBBBBBBBBBBBBBBBBBBBBBBBBBBBBBBBBBBBBBBBBBBBBBBBBBBBBBBBBBBBBBBBBBBBBBBBBBBBBBBBBBB
// Berechnung für die Phasen 4,5
//
Val567(VEL_IST := Vel_Ist, Acc_Ist := Acc_Ist, DCC_MAX := Dcc_Max, VE7_D := 0, RB := RB); // calc_Val567_inPhase45

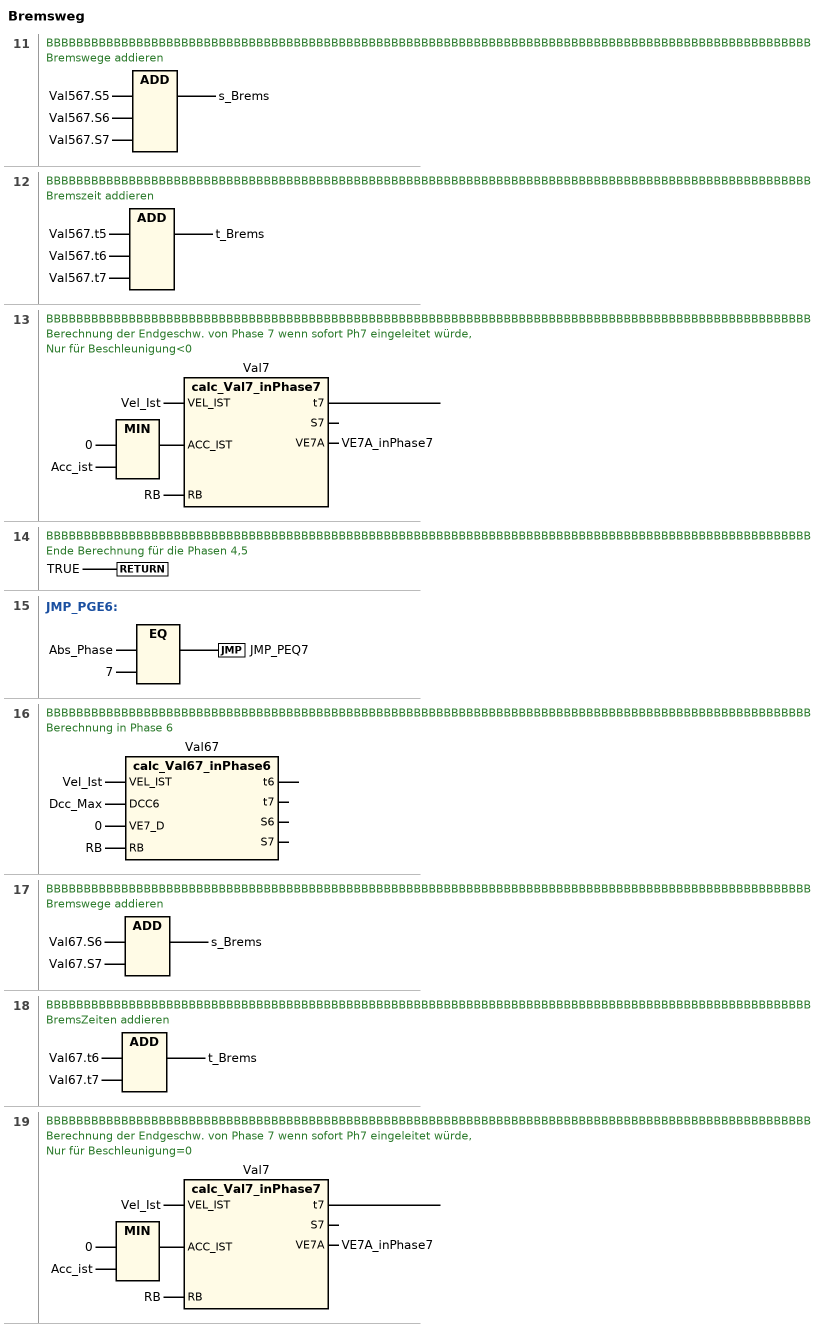
// NETWORK 11
// 					BBBBBBBBBBBBBBBBBBBBBBBBBBBBBBBBBBBBBBBBBBBBBBBBBBBBBBBBBBBBBBBBBBBBBBBBBBBBBBBBBBBBBBBBBBBBBBBBBBBBBB
// Bremswege addieren
//
s_Brems := Val567.S5 + Val567.S6 + Val567.S7;

// NETWORK 12
// 					BBBBBBBBBBBBBBBBBBBBBBBBBBBBBBBBBBBBBBBBBBBBBBBBBBBBBBBBBBBBBBBBBBBBBBBBBBBBBBBBBBBBBBBBBBBBBBBBBBBBBB
// Bremszeit addieren
//
t_Brems := Val567.t5 + Val567.t6 + Val567.t7;

// NETWORK 13
// 					BBBBBBBBBBBBBBBBBBBBBBBBBBBBBBBBBBBBBBBBBBBBBBBBBBBBBBBBBBBBBBBBBBBBBBBBBBBBBBBBBBBBBBBBBBBBBBBBBBBBBB
// Berechnung der Endgeschw. von Phase 7 wenn sofort Ph7 eingeleitet würde,
// Nur für Beschleunigung<0
//
Val7(VEL_IST := Vel_Ist, ACC_IST := MIN(0, Acc_ist), RB := RB, VE7A => VE7A_inPhase7); // calc_Val7_inPhase7

// NETWORK 14
// 					BBBBBBBBBBBBBBBBBBBBBBBBBBBBBBBBBBBBBBBBBBBBBBBBBBBBBBBBBBBBBBBBBBBBBBBBBBBBBBBBBBBBBBBBBBBBBBBBBBBBBB
// Ende Berechnung für die Phasen 4,5
//
RETURN;

// NETWORK 15
JMP_PGE6:
IF Abs_Phase = 7 THEN JMP JMP_PEQ7; END_IF

// NETWORK 16
// 					BBBBBBBBBBBBBBBBBBBBBBBBBBBBBBBBBBBBBBBBBBBBBBBBBBBBBBBBBBBBBBBBBBBBBBBBBBBBBBBBBBBBBBBBBBBBBBBBBBBBBB
// Berechnung in Phase 6
//
Val67(VEL_IST := Vel_Ist, DCC6 := Dcc_Max, VE7_D := 0, RB := RB); // calc_Val67_inPhase6

// NETWORK 17
// 					BBBBBBBBBBBBBBBBBBBBBBBBBBBBBBBBBBBBBBBBBBBBBBBBBBBBBBBBBBBBBBBBBBBBBBBBBBBBBBBBBBBBBBBBBBBBBBBBBBBBBB
// Bremswege addieren
//
s_Brems := Val67.S6 + Val67.S7;

// NETWORK 18
// 					BBBBBBBBBBBBBBBBBBBBBBBBBBBBBBBBBBBBBBBBBBBBBBBBBBBBBBBBBBBBBBBBBBBBBBBBBBBBBBBBBBBBBBBBBBBBBBBBBBBBBB
// BremsZeiten addieren
//
t_Brems := Val67.t6 + Val67.t7;

// NETWORK 19
// 					BBBBBBBBBBBBBBBBBBBBBBBBBBBBBBBBBBBBBBBBBBBBBBBBBBBBBBBBBBBBBBBBBBBBBBBBBBBBBBBBBBBBBBBBBBBBBBBBBBBBBB
// Berechnung der Endgeschw. von Phase 7 wenn sofort Ph7 eingeleitet würde,
// Nur für Beschleunigung=0
//
Val7(VEL_IST := Vel_Ist, ACC_IST := MIN(0, Acc_ist), RB := RB, VE7A => VE7A_inPhase7); // calc_Val7_inPhase7

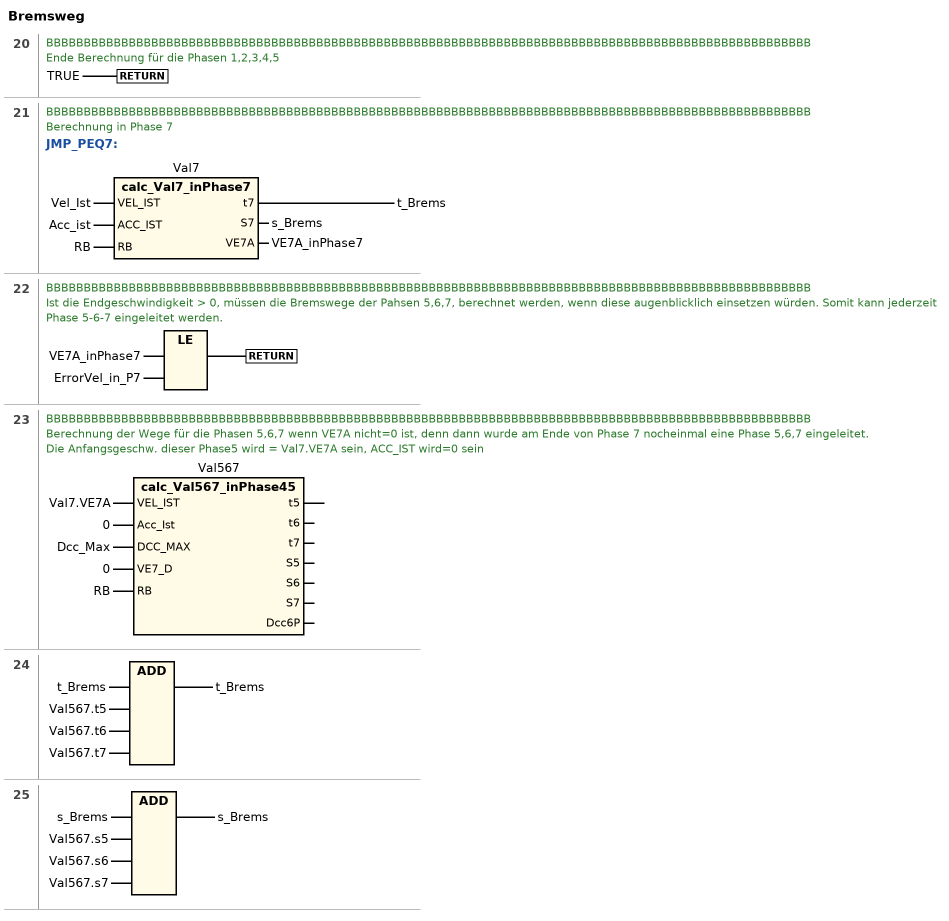
// NETWORK 20
// 					BBBBBBBBBBBBBBBBBBBBBBBBBBBBBBBBBBBBBBBBBBBBBBBBBBBBBBBBBBBBBBBBBBBBBBBBBBBBBBBBBBBBBBBBBBBBBBBBBBBBBB
// Ende Berechnung für die Phasen 1,2,3,4,5
//
RETURN;

// NETWORK 21
// 					BBBBBBBBBBBBBBBBBBBBBBBBBBBBBBBBBBBBBBBBBBBBBBBBBBBBBBBBBBBBBBBBBBBBBBBBBBBBBBBBBBBBBBBBBBBBBBBBBBBBBB
// Berechnung in Phase 7
//
JMP_PEQ7:
Val7(VEL_IST := Vel_Ist, ACC_IST := Acc_ist, RB := RB, S7 => s_Brems, VE7A => VE7A_inPhase7); // calc_Val7_inPhase7
t_Brems := Val7.t7;

// NETWORK 22
// 					BBBBBBBBBBBBBBBBBBBBBBBBBBBBBBBBBBBBBBBBBBBBBBBBBBBBBBBBBBBBBBBBBBBBBBBBBBBBBBBBBBBBBBBBBBBBBBBBBBBBBB
// Ist die Endgeschwindigkeit > 0, müssen die Bremswege der Pahsen 5,6,7, berechnet werden, wenn diese augenblicklich einsetzen würden. Somit kann jederzeit Phase 5-6-7 eingeleitet werden.
//
IF VE7A_inPhase7 <= ErrorVel_in_P7 THEN RETURN; END_IF

// NETWORK 23
// 					BBBBBBBBBBBBBBBBBBBBBBBBBBBBBBBBBBBBBBBBBBBBBBBBBBBBBBBBBBBBBBBBBBBBBBBBBBBBBBBBBBBBBBBBBBBBBBBBBBBBBB
// Berechnung der Wege für die Phasen 5,6,7 wenn VE7A nicht=0 ist, denn dann wurde am Ende von Phase 7 nocheinmal eine Phase 5,6,7 eingeleitet.
// Die Anfangsgeschw. dieser Phase5 wird = Val7.VE7A sein, ACC_IST wird=0 sein
//
Val567(VEL_IST := Val7.VE7A, Acc_Ist := 0, DCC_MAX := Dcc_Max, VE7_D := 0, RB := RB); // calc_Val567_inPhase45

// NETWORK 24
t_Brems := t_Brems + Val567.t5 + Val567.t6 + Val567.t7;

// NETWORK 25
s_Brems := s_Brems + Val567.s5 + Val567.s6 + Val567.s7;

END_FUNCTION_BLOCK

// POUs/Achsen_Bausteinen/FB/calc_Val3_inPhase123
FUNCTION_BLOCK calc_Val3_inPhase123(*Die Funktion berechnet t3,S3 und VE3 in den Phasen 1,2 oder 3 wenn sofort Phase3 eingeleitet würde.
Bedingung: Phase = 0,1,2,3 / ACC_IST>=0 

t3 ist die Restzeit bis zum Ende der Phase3, also wo ACC_IST zu 0 abgebaut wurde.
VE3  ist die Endgeschwindigkeit am Ende der Phase 3
S3: Sie ist die Reststrecke die bis zum Ende der Phase 3 verbraucht sein wird.
*)

VAR_INPUT
	Vel_Ist:LREAL;(*aktuelle Geschw. pos. oder negativ, das Vorzeichen hat keine Relevanz das ABS gebildet wird*)
	Acc_Ist:LREAL;(*ACC_IST ist in Phase3 immer positiv, es wird aber dennoch ABS gebildet*)
	RB:LREAL;(*Soll - Ruckbegtenzungswert in mm/s^3. Zulässige Werte: RB >=0. Bei 0 ist RB deaktiviert*)
END_VAR
VAR_OUTPUT
	t3:LREAL;(*Zeit für Phase 3*)
	S3:LREAL;(*Strecke für Phase3, >=0*)
	VE3A:LREAL;(*Absolutwert der Geschw. am Ende Phase3, pos. oder negativ (abhängig von Vel_IST*)
END_VAR
VAR
	DV3P: LREAL;(*positiver Wert der Geschwindigkeitsdifferenz in Phase 3*)
	Acc_IstA: LREAL;
END_VAR

Acc_IstA:=ABS(Acc_Ist);

IF RB<=0 THEN
	t3:=0;
	DV3P:=0;
	VE3A:=ABS(VEL_IST);
	s3:=0;
	RETURN;
END_IF

t3:=Acc_IstA/RB;(*Beschl. muss in Phase3 zu 0 abgebaut werden, t3 ergibt die Zeit die notwendig ist bis ACC=0 ist*)
DV3P:=Acc_IstA*t3-0.5*RB*EXPT(t3,2); (*test ok Exel*)
VE3A:=ABS(VEL_IST)+DV3P;(* test ok Exel*)
s3:=ABS(Vel_Ist) * t3 + 0.5*Acc_IstA*EXPT(t3,2) - 1/6.0*RB*EXPT(t3,3);(*test ok Exel*)

END_FUNCTION_BLOCK

// POUs/Achsen_Bausteinen/FB/Phase3
FUNCTION_BLOCK Phase3
VAR_INPUT
	Achs_CMD:TKont_Achse_OUT;
END_VAR
VAR_OUTPUT
END_VAR
VAR_IN_OUT
	IV_RB: TIV_RB;
END_VAR
VAR
	Bremsweg: Bremsweg;
	Temp_LReal: LREAL;
	calc_Rbist_inPhase3: calc_Rbist_inPhase3;
	AccLimit0: BOOL;
	switchPhase1_3: switchPhase;
	switchPhase5_5: switchPhase;
	switchPhase4_1: switchPhase;
	RbKomp_Ph3: BOOL;
END_VAR
VAR // added by the converter: edge detectors and wires of the graphical bodies
    _w1 : LREAL;
    _w2, _w3, _w4 : BOOL;
END_VAR

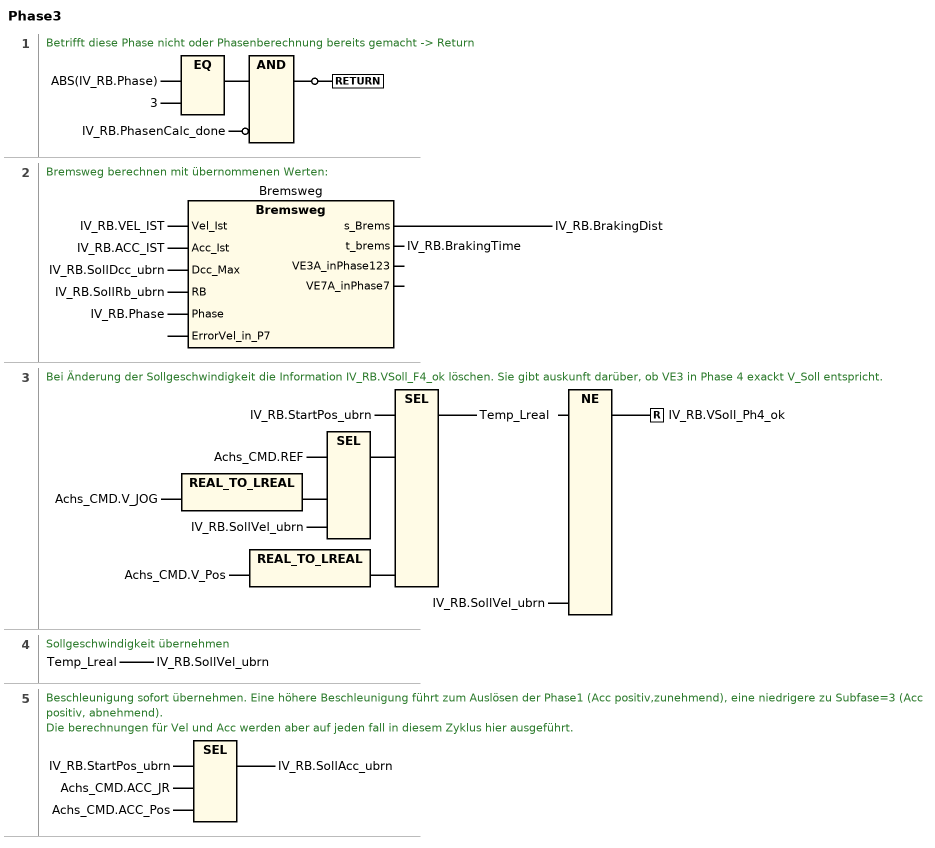
// NETWORK 1
// Betrifft diese Phase nicht oder Phasenberechnung bereits gemacht -> Return
IF NOT ((ABS(IV_RB.Phase)) = 3 AND NOT IV_RB.PhasenCalc_done) THEN RETURN; END_IF

// NETWORK 2
// Bremsweg berechnen mit übernommenen Werten:
Bremsweg(
    Vel_Ist := IV_RB.VEL_IST,
    Acc_Ist := IV_RB.ACC_IST,
    Dcc_Max := IV_RB.SollDcc_ubrn,
    RB := IV_RB.SollRb_ubrn,
    Phase := IV_RB.Phase,
    t_brems => IV_RB.BrakingTime);
IV_RB.BrakingDist := Bremsweg.s_Brems;

// NETWORK 3
// Bei Änderung der Sollgeschwindigkeit die Information IV_RB.VSoll_F4_ok löschen. Sie gibt auskunft darüber, ob VE3 in Phase 4 exackt V_Soll entspricht.
_w1 := SEL(IV_RB.StartPos_ubrn, SEL(Achs_CMD.REF, REAL_TO_LREAL(Achs_CMD.V_JOG), IV_RB.SollVel_ubrn), REAL_TO_LREAL(Achs_CMD.V_Pos));
Temp_Lreal := _w1;
IV_RB.VSoll_Ph4_ok R= _w1 <> IV_RB.SollVel_ubrn;

// NETWORK 4
// Sollgeschwindigkeit übernehmen
IV_RB.SollVel_ubrn := Temp_Lreal;

// NETWORK 5
// 					Beschleunigung sofort übernehmen. Eine höhere Beschleunigung führt zum Auslösen der Phase1 (Acc positiv,zunehmend), eine niedrigere zu Subfase=3 (Acc positiv, abnehmend).
// Die berechnungen für Vel und Acc werden aber auf jeden fall in diesem Zyklus hier ausgeführt.
//
IV_RB.SollAcc_ubrn := SEL(IV_RB.StartPos_ubrn, Achs_CMD.ACC_JR, Achs_CMD.ACC_Pos);

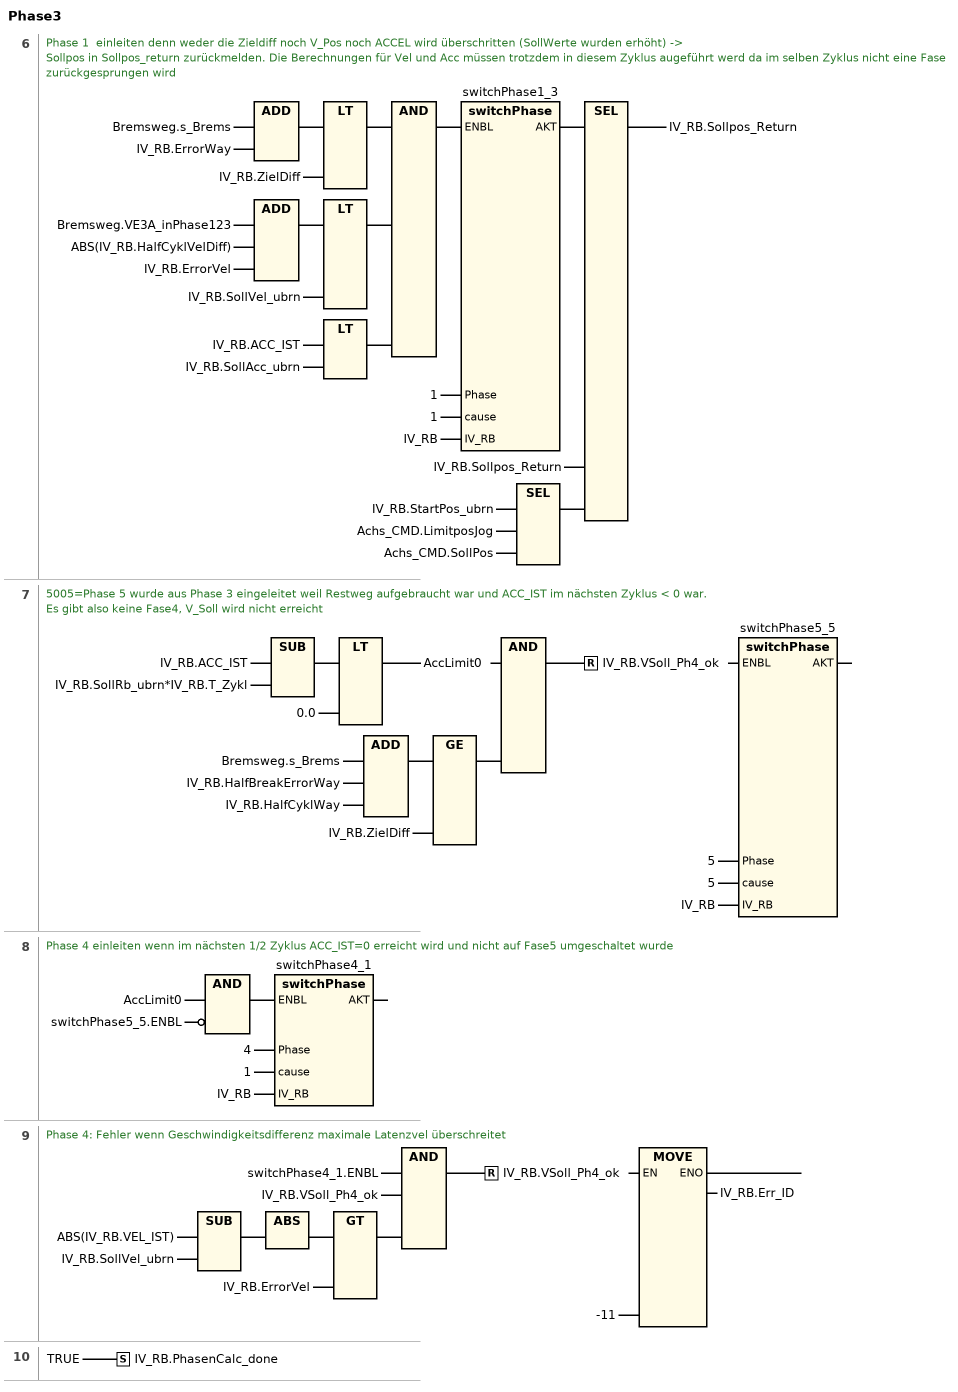
// NETWORK 6
// 					 Phase 1  einleiten denn weder die Zieldiff noch V_Pos noch ACCEL wird überschritten (SollWerte wurden erhöht) ->
//  Sollpos in Sollpos_return zurückmelden. Die Berechnungen für Vel und Acc müssen trotzdem in diesem Zyklus augeführt werd da im selben Zyklus nicht eine Fase zurückgesprungen wird
//
switchPhase1_3(
    ENBL := Bremsweg.s_Brems + IV_RB.ErrorWay < IV_RB.ZielDiff AND Bremsweg.VE3A_inPhase123 + (ABS(IV_RB.HalfCyklVelDiff)) + IV_RB.ErrorVel < IV_RB.SollVel_ubrn AND IV_RB.ACC_IST < IV_RB.SollAcc_ubrn,
    Phase := 1,
    cause := 1,
    IV_RB := IV_RB); // switchPhase
IV_RB.Sollpos_Return := SEL(switchPhase1_3.AKT, IV_RB.Sollpos_Return, SEL(IV_RB.StartPos_ubrn, Achs_CMD.LimitposJog, Achs_CMD.SollPos));

// NETWORK 7
// 					5005=Phase 5 wurde aus Phase 3 eingeleitet weil Restweg aufgebraucht war und ACC_IST im nächsten Zyklus < 0 war.
// Es gibt also keine Fase4, V_Soll wird nicht erreicht
//
_w2 := IV_RB.ACC_IST - (IV_RB.SollRb_ubrn*IV_RB.T_Zykl) < 0.0;
AccLimit0 := _w2;
_w3 := _w2 AND Bremsweg.s_Brems + IV_RB.HalfBreakErrorWay + IV_RB.HalfCyklWay >= IV_RB.ZielDiff;
IV_RB.VSoll_Ph4_ok R= _w3;
switchPhase5_5(ENBL := _w3, Phase := 5, cause := 5, IV_RB := IV_RB); // switchPhase

// NETWORK 8
// Phase 4 einleiten wenn im nächsten 1/2 Zyklus ACC_IST=0 erreicht wird und nicht auf Fase5 umgeschaltet wurde
switchPhase4_1(ENBL := AccLimit0 AND NOT switchPhase5_5.ENBL, Phase := 4, cause := 1, IV_RB := IV_RB); // switchPhase

// NETWORK 9
//
// Phase 4: Fehler wenn Geschwindigkeitsdifferenz maximale Latenzvel überschreitet
//
_w4 := switchPhase4_1.ENBL AND IV_RB.VSoll_Ph4_ok AND ABS((ABS(IV_RB.VEL_IST)) - IV_RB.SollVel_ubrn) > IV_RB.ErrorVel;
IV_RB.VSoll_Ph4_ok R= _w4;
IF _w4 THEN IV_RB.Err_ID := -11; END_IF

// NETWORK 10
IV_RB.PhasenCalc_done S= TRUE;

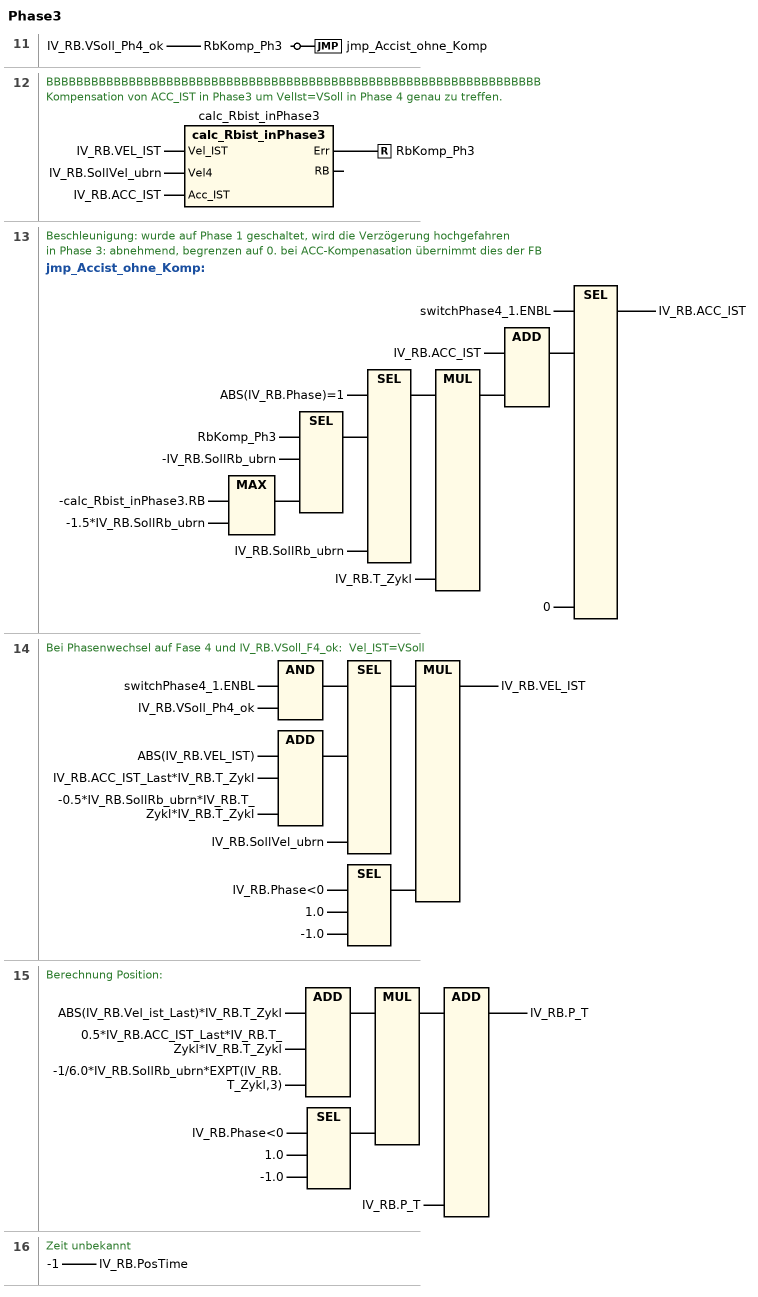
// NETWORK 11
RbKomp_Ph3 := IV_RB.VSoll_Ph4_ok;
IF NOT IV_RB.VSoll_Ph4_ok THEN JMP jmp_Accist_ohne_Komp; END_IF

// NETWORK 12
// 					BBBBBBBBBBBBBBBBBBBBBBBBBBBBBBBBBBBBBBBBBBBBBBBBBBBBBBBBBBBBBBBBBB
// Kompensation von ACC_IST in Phase3 um VelIst=VSoll in Phase 4 genau zu treffen.
//
calc_Rbist_inPhase3(Vel_IST := IV_RB.VEL_IST, Vel4 := IV_RB.SollVel_ubrn, Acc_IST := IV_RB.ACC_IST);
RbKomp_Ph3 R= calc_Rbist_inPhase3.Err;

// NETWORK 13
// 					Beschleunigung: wurde auf Phase 1 geschaltet, wird die Verzögerung hochgefahren
// in Phase 3: abnehmend, begrenzen auf 0. bei ACC-Kompenasation übernimmt dies der FB
//
jmp_Accist_ohne_Komp:
IV_RB.ACC_IST := SEL(switchPhase4_1.ENBL, IV_RB.ACC_IST + SEL(ABS(IV_RB.Phase)=1, SEL(RbKomp_Ph3, -IV_RB.SollRb_ubrn, MAX(-calc_Rbist_inPhase3.RB, -1.5*IV_RB.SollRb_ubrn)), IV_RB.SollRb_ubrn) * IV_RB.T_Zykl, 0);

// NETWORK 14
// 					Bei Phasenwechsel auf Fase 4 und IV_RB.VSoll_F4_ok:  Vel_IST=VSoll
//
//
IV_RB.VEL_IST := SEL(switchPhase4_1.ENBL AND IV_RB.VSoll_Ph4_ok, (ABS(IV_RB.VEL_IST)) + (IV_RB.ACC_IST_Last*IV_RB.T_Zykl) + (-0.5*IV_RB.SollRb_ubrn*IV_RB.T_Zykl*IV_RB.T_Zykl), IV_RB.SollVel_ubrn) * SEL(IV_RB.Phase<0, 1.0, -1.0);

// NETWORK 15
// Berechnung Position:
IV_RB.P_T := ((ABS(IV_RB.Vel_ist_Last)*IV_RB.T_Zykl) + (0.5*IV_RB.ACC_IST_Last*IV_RB.T_Zykl*IV_RB.T_Zykl) + (-1/6.0*IV_RB.SollRb_ubrn*EXPT(IV_RB.T_Zykl,3))) * SEL(IV_RB.Phase<0, 1.0, -1.0) + IV_RB.P_T;

// NETWORK 16
// Zeit unbekannt
IV_RB.PosTime := -1;

END_FUNCTION_BLOCK

// POUs/Achsen_Bausteinen/FB/switchPhase
FUNCTION_BLOCK switchPhase (*übergit die angegeben Phase - Nr, wobei das Vorzeichen erhalten bleibt, es wird nur der Betrag übernommen*)
VAR_INPUT
	ENBL: BOOL;
	Phase: INT;
	cause: INT;(*Ursache der Phasenänderung*)
END_VAR
VAR_OUTPUT
	AKT: BOOL;
END_VAR
VAR
END_VAR
VAR_IN_OUT
	IV_RB:TIV_RB;
END_VAR

IF ENBL THEN

	AKT:=TRUE;

	IF ABS(IV_RB.Phase)<>ABS(Phase) THEN
		IV_RB.FL_PhChnge:=TRUE;
		IV_RB.PhCng:=ABS(Phase*100)+ABS(IV_RB.Phase)*10+cause;
	END_IF

	IF IV_RB.Phase<0 THEN(*aktuelle Phase ist negativ*)
		IV_RB.Phase:=-ABS(Phase); (*altes vorzeichen beibehalten!*)
	ELSIF IV_RB.Phase>0 THEN(*aktuelle Phase ist positiv und nicht 0*)
		IV_RB.Phase:=ABS(Phase);
	ELSE (*Es wurde aus Phase=0 gestartet, Vorzeichen wird übernommen*)
		IV_RB.Phase:=Phase;
	END_IF

ELSE

	AKT:=FALSE;
END_IF

END_FUNCTION_BLOCK

// POUs/Achsen_Bausteinen/FB/calc_Rbist_inPhase3
FUNCTION_BLOCK calc_Rbist_inPhase3 (*Damit in Phase 4 die Geschwindigkeit VEL_IST=Vel4 gesetzt werden kann (die Sollgeschw. trotz Latenzzeitfehler genau „getroffen“ wird), wird
die Ruckbegrenzung durch eine Funktion berechnet. Über diese wird dann ACC_IST und VEL_Ist berechnet:
RB=f(ACC_IST,DV3P)
DV3P = 1/2 * ACC_IST^2 / RB  ->  RB = 1/2 * ACC_IST^2 / DV3P

*) 

VAR_INPUT
	Vel_IST: LREAL;(*das Vorzeichen hat keine Relevanz da ABS gebildet wird *)
	Vel4:LREAL;(* Sollgeschwindigkeit die in Fase4 erreicht werden soll. Das Vorzeichen hat keine Relevanz da ABS gebildet wird *)
	Acc_IST: LREAL;(*korrigierte Geschwindigkeit*)
END_VAR
VAR_OUTPUT
	Err: BOOL;
	RB: LREAL;
END_VAR
VAR
	DV3P: LREAL;
END_VAR

DV3P:= ABS(Vel4) - ABS(Vel_Ist);
IF DV3P<=0 THEN
	Err:=TRUE;
	RETURN;
ELSE
	Err:=FALSE;
	RB:= 0.5 * EXPT(ACC_IST,2)/DV3P;
END_IF

END_FUNCTION_BLOCK

// POUs/Achsen_Bausteinen/FB/calc_Val567_inPhase45
FUNCTION_BLOCK calc_Val567_inPhase45 (*Die Funktion gibt die Werte t5, t6, t7, s5, s6, s7, DCC6 zurück, die bis zum erreichen von VEL_IST = VE7_D mit ACC_IST=0 benötigt werden.*)

VAR_INPUT
	VEL_IST: LREAL;(* Vorzeichen hat keine Relevanz da ABS gebildet wird. Wenn die Achse in Phase 1,2,3 ist: hier VE3 aus Funktion calc_Val3_inPhase123 übergeben*)
	Acc_Ist:LREAL; (* Vorzeichen hat keine Relevanz da ABS gebildet wird. Wenn die Achse in Phase 1,2,3 ist: hier 0  übergeben damit die Vollen Phase 5+6+7 gerechnet wird*)
	DCC_MAX: LREAL;(* positiver Wert!!*)
	VE7_D:LREAL;(*gewünschte Endgeschwindigkeit am Ende von Phase7. ist beim Zielpositionieren = 0*)
	RB:LREAL;(*Ruckbegrenzung mm/s^3*)
END_VAR
VAR_OUTPUT
	t5: LREAL;			(*Restzeit in Phase 5*)
	t6: LREAL;			(*Restzeit in Phase 6*)
	t7: LREAL;			(*Restzeit in Phase 7*)
	S5: LREAL;			(*Reststrecke in Phase5*)
	S6: LREAL;			(*Reststrecke in Phase6*)
	S7: LREAL;			(*Reststrecke in Phase7*)
	Dcc6P: LREAL;	(*Verzögerung in Phase 6 *)
END_VAR
VAR
	DV5P:LREAL;
	DV6P: LREAL;
	DV7P: LREAL;
	VEL_ISTA: LREAL;
	VE7_DA: LREAL;
	ACC_ISTA: LREAL;
END_VAR

VEL_ISTA:=ABS(VEL_IST);
VE7_DA:=MIN(ABS(VE7_D),VEL_ISTA);(*VE7_DA muss eine kleiner Geschwindigkeit als die Istgeschwindigkeit sein*)
ACC_ISTA:=ABS(ACC_IST);

IF DCC_MAX <=0 THEN RETURN;END_IF

IF RB<=0 THEN
	t5:=0;
	DV5P:=0;
	S5:=0;
	t7:=0;
	DV7P:=0;
	S7:=0;

	DV6P:=VEL_ISTA - VE7_DA;
	DCC6P:=DCC_MAX;
	t6:= DV6P / DCC6P;
	S6:=VEL_ISTA * t6 - 0.5 * DCC6P * EXPT(t6, 2);
	RETURN;
END_IF


(*Annahme: DV6P=0 denn DCC6P überschreitet nicht DCC_MAX, VE3 fällt zur hälfte auf DV7  : *)
DCC6P := SQRT(MAX(0,(VEL_ISTA * RB + 0.5 * EXPT(ACC_ISTA, 2) - VE7_DA * RB)));

(*Kontrolle: DCC6 > DCC_MAX ? *)
IF DCC6P <= DCC_MAX THEN (* NEIN -> DCC6  beibehalten*)
	t6:=0;
	S6:=0;
	DV6P:=0;
	DV7P:= 0.5 * EXPT(DCC6P, 2) / RB;
	DV5P:= DV7P - 0.5 * EXPT(ACC_ISTA, 2) / RB;

ELSE	(* Ja -> DCC6 = DCC_MAX setzen *)
	DCC6P:=DCC_MAX;
	DV7P:= 0.5 * EXPT(DCC6P, 2) / RB;
	DV5P:= DV7P - 0.5 * EXPT(ACC_ISTA, 2) / RB;
	DV6P:= VEL_ISTA - DV5P - DV7P - VE7_DA;
	t6:= DV6P / DCC6P;
	t6:= MAX(t6,0);
	S6:= (VEL_ISTA - DV5P  - 0.5 * DCC6P * t6) * t6;
	S6:=MAX(S6,0);
END_IF

(* weitere Berechnungen für t5,(t6)=0, t7, S5, (S6=0), S7. Diese sind für beide Fälle gültig:*)
t5:= (DCC6P - ACC_ISTA) / RB;
t5:= MAX(t5,0);
S5:= Vel_IstA * t5 - 0.5 * ACC_ISTA *EXPT( t5, 2) - 1/6.0 * RB * EXPT(t5, 3);
S5:=MAX(S5,0);
t7:= DCC6P / RB;
S7:=(VE7_DA + DV7P -  0.5*DCC6P*t7 +  1/6.0*RB*EXPT(t7,2))*t7;
S7:=MAX(S7,0);

END_FUNCTION_BLOCK

// POUs/Achsen_Bausteinen/FB/Phase7
FUNCTION_BLOCK Phase7
VAR_INPUT
	Achs_CMD:TKont_Achse_OUT;
END_VAR
VAR_IN_OUT
	IV_RB: TIV_RB;
END_VAR
VAR
	Bremsweg: Bremsweg;
	SollVel: LREAL;
	VE7_caEQ_0: BOOL;		(*Das Ende der Phase 7 (ACCIST=0) wird mit Vel=0 erreicht.*)
	ZielDiff_ueberschr: BOOL;
	switchPhase5_3: switchPhase;
	switchPhase5_4: switchPhase;
	switchPhase4_2: switchPhase;
	switchPhase0_1: switchPhase;
	switchPhase0_2: switchPhase;
	switchPhase0_3: switchPhase;
	Variante2: BOOL;
	Dcc_Komp: LREAL;
	DccKomp_akt: BOOL;
END_VAR
VAR_OUTPUT
	PEH: BOOL;
END_VAR
VAR // added by the converter: edge detectors and wires of the graphical bodies
    _w1 : ANY;
    _w2, _w3 : BOOL;
END_VAR

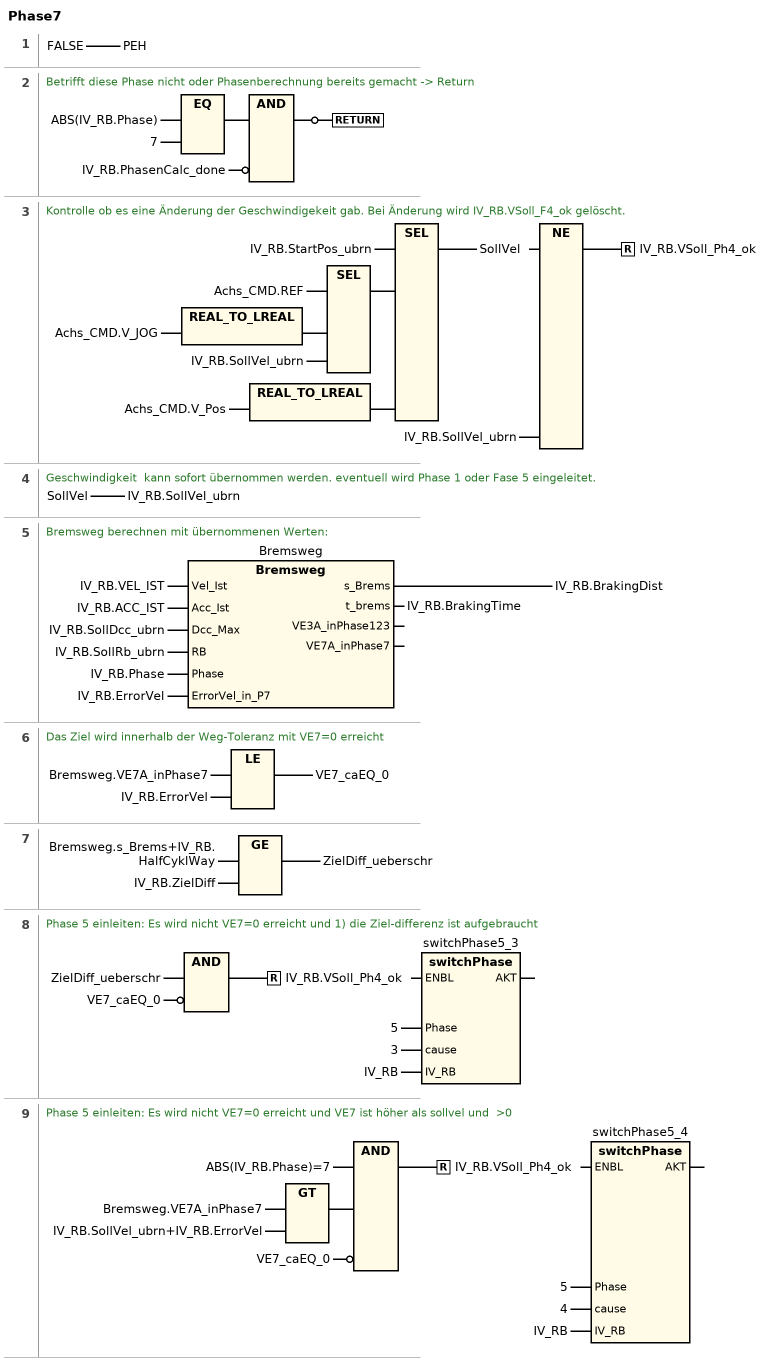
// NETWORK 1
PEH := FALSE;

// NETWORK 2
// Betrifft diese Phase nicht oder Phasenberechnung bereits gemacht -> Return
IF NOT ((ABS(IV_RB.Phase)) = 7 AND NOT IV_RB.PhasenCalc_done) THEN RETURN; END_IF

// NETWORK 3
// Kontrolle ob es eine Änderung der Geschwindigekeit gab. Bei Änderung wird IV_RB.VSoll_F4_ok gelöscht.
_w1 := SEL(IV_RB.StartPos_ubrn, SEL(Achs_CMD.REF, REAL_TO_LREAL(Achs_CMD.V_JOG), IV_RB.SollVel_ubrn), REAL_TO_LREAL(Achs_CMD.V_Pos));
SollVel := _w1;
IV_RB.VSoll_Ph4_ok R= _w1 <> IV_RB.SollVel_ubrn;

// NETWORK 4
// Geschwindigkeit  kann sofort übernommen werden. eventuell wird Phase 1 oder Fase 5 eingeleitet.
IV_RB.SollVel_ubrn := SollVel;

// NETWORK 5
// Bremsweg berechnen mit übernommenen Werten:
Bremsweg(
    Vel_Ist := IV_RB.VEL_IST,
    Acc_Ist := IV_RB.ACC_IST,
    Dcc_Max := IV_RB.SollDcc_ubrn,
    RB := IV_RB.SollRb_ubrn,
    Phase := IV_RB.Phase,
    ErrorVel_in_P7 := IV_RB.ErrorVel,
    t_brems => IV_RB.BrakingTime);
IV_RB.BrakingDist := Bremsweg.s_Brems;

// NETWORK 6
// Das Ziel wird innerhalb der Weg-Toleranz mit VE7=0 erreicht
VE7_caEQ_0 := Bremsweg.VE7A_inPhase7 <= IV_RB.ErrorVel;

// NETWORK 7
ZielDiff_ueberschr := (Bremsweg.s_Brems+IV_RB.HalfCyklWay) >= IV_RB.ZielDiff;

// NETWORK 8
// Phase 5 einleiten: Es wird nicht VE7=0 erreicht und 1) die Ziel-differenz ist aufgebraucht
_w2 := ZielDiff_ueberschr AND NOT VE7_caEQ_0;
IV_RB.VSoll_Ph4_ok R= _w2;
switchPhase5_3(ENBL := _w2, Phase := 5, cause := 3, IV_RB := IV_RB); // switchPhase

// NETWORK 9
// Phase 5 einleiten: Es wird nicht VE7=0 erreicht und VE7 ist höher als sollvel und  >0
_w3 := (ABS(IV_RB.Phase)=7) AND Bremsweg.VE7A_inPhase7 > (IV_RB.SollVel_ubrn+IV_RB.ErrorVel) AND NOT VE7_caEQ_0;
IV_RB.VSoll_Ph4_ok R= _w3;
switchPhase5_4(ENBL := _w3, Phase := 5, cause := 4, IV_RB := IV_RB); // switchPhase

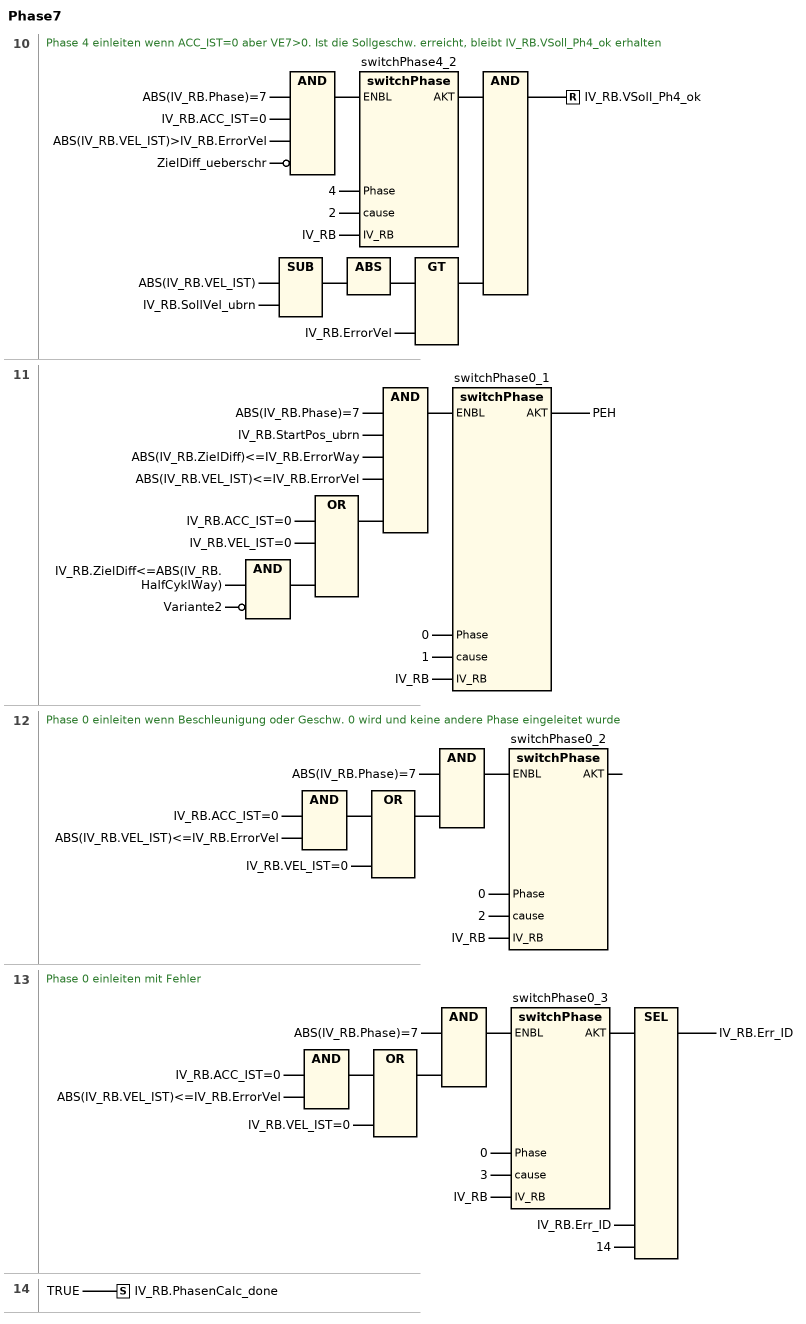
// NETWORK 10
// Phase 4 einleiten wenn ACC_IST=0 aber VE7>0. Ist die Sollgeschw. erreicht, bleibt IV_RB.VSoll_Ph4_ok erhalten
switchPhase4_2(
    ENBL := (ABS(IV_RB.Phase)=7) AND (IV_RB.ACC_IST=0) AND (ABS(IV_RB.VEL_IST)>IV_RB.ErrorVel) AND NOT ZielDiff_ueberschr,
    Phase := 4,
    cause := 2,
    IV_RB := IV_RB); // switchPhase
IV_RB.VSoll_Ph4_ok R= switchPhase4_2.AKT AND ABS((ABS(IV_RB.VEL_IST)) - IV_RB.SollVel_ubrn) > IV_RB.ErrorVel;

// NETWORK 11
switchPhase0_1(
    ENBL := (ABS(IV_RB.Phase)=7) AND IV_RB.StartPos_ubrn AND (ABS(IV_RB.ZielDiff)<=IV_RB.ErrorWay) AND (ABS(IV_RB.VEL_IST)<=IV_RB.ErrorVel) AND ((IV_RB.ACC_IST=0) OR (IV_RB.VEL_IST=0) OR (IV_RB.ZielDiff<=ABS(IV_RB.HalfCyklWay)) AND NOT Variante2),
    Phase := 0,
    cause := 1,
    IV_RB := IV_RB); // switchPhase
PEH := switchPhase0_1.AKT;

// NETWORK 12
// Phase 0 einleiten wenn Beschleunigung oder Geschw. 0 wird und keine andere Phase eingeleitet wurde
switchPhase0_2(
    ENBL := (ABS(IV_RB.Phase)=7) AND ((IV_RB.ACC_IST=0) AND (ABS(IV_RB.VEL_IST)<=IV_RB.ErrorVel) OR (IV_RB.VEL_IST=0)),
    Phase := 0,
    cause := 2,
    IV_RB := IV_RB); // switchPhase

// NETWORK 13
// Phase 0 einleiten mit Fehler
switchPhase0_3(
    ENBL := (ABS(IV_RB.Phase)=7) AND ((IV_RB.ACC_IST=0) AND (ABS(IV_RB.VEL_IST)<=IV_RB.ErrorVel) OR (IV_RB.VEL_IST=0)),
    Phase := 0,
    cause := 3,
    IV_RB := IV_RB); // switchPhase
IV_RB.Err_ID := SEL(switchPhase0_3.AKT, IV_RB.Err_ID, 14);

// NETWORK 14
IV_RB.PhasenCalc_done S= TRUE;

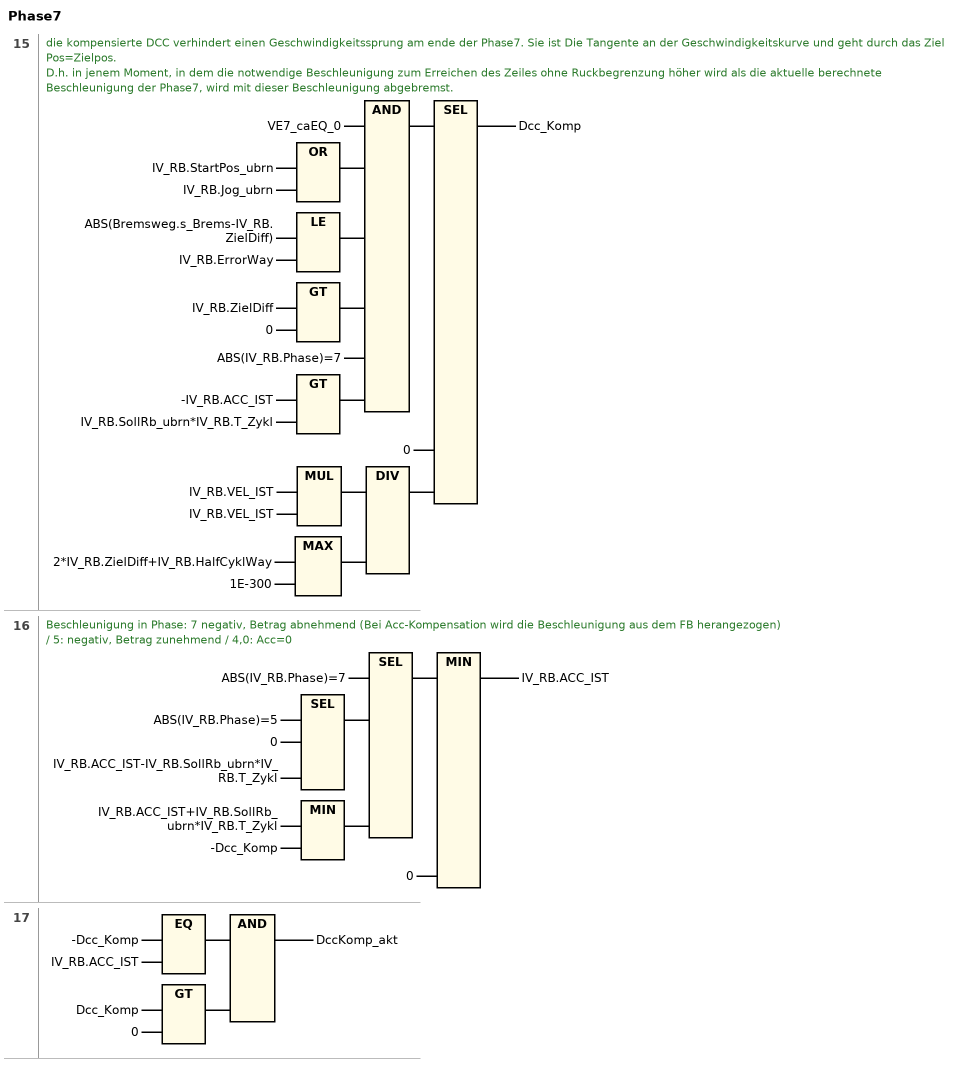
// NETWORK 15
// 					die kompensierte DCC verhindert einen Geschwindigkeitssprung am ende der Phase7. Sie ist Die Tangente an der Geschwindigkeitskurve und geht durch das Ziel Pos=Zielpos.
// D.h. in jenem Moment, in dem die notwendige Beschleunigung zum Erreichen des Zeiles ohne Ruckbegrenzung höher wird als die aktuelle berechnete Beschleunigung der Phase7, wird mit dieser Beschleunigung abgebremst.
//
Dcc_Komp := SEL(VE7_caEQ_0 AND (IV_RB.StartPos_ubrn OR IV_RB.Jog_ubrn) AND (ABS(Bremsweg.s_Brems-IV_RB.ZielDiff)) <= IV_RB.ErrorWay AND IV_RB.ZielDiff > 0 AND (ABS(IV_RB.Phase)=7) AND (-IV_RB.ACC_IST) > (IV_RB.SollRb_ubrn*IV_RB.T_Zykl), 0, (IV_RB.VEL_IST * IV_RB.VEL_IST) / MAX(2*IV_RB.ZielDiff+IV_RB.HalfCyklWay, 1E-300));

// NETWORK 16
// 					Beschleunigung in Phase: 7 negativ, Betrag abnehmend (Bei Acc-Kompensation wird die Beschleunigung aus dem FB herangezogen)
//  / 5: negativ, Betrag zunehmend / 4,0: Acc=0
//
IV_RB.ACC_IST := MIN(SEL(ABS(IV_RB.Phase)=7, SEL(ABS(IV_RB.Phase)=5, 0, IV_RB.ACC_IST-IV_RB.SollRb_ubrn*IV_RB.T_Zykl), MIN(IV_RB.ACC_IST+IV_RB.SollRb_ubrn*IV_RB.T_Zykl, -Dcc_Komp)), 0);

// NETWORK 17
DccKomp_akt := (-Dcc_Komp) = IV_RB.ACC_IST AND Dcc_Komp > 0;

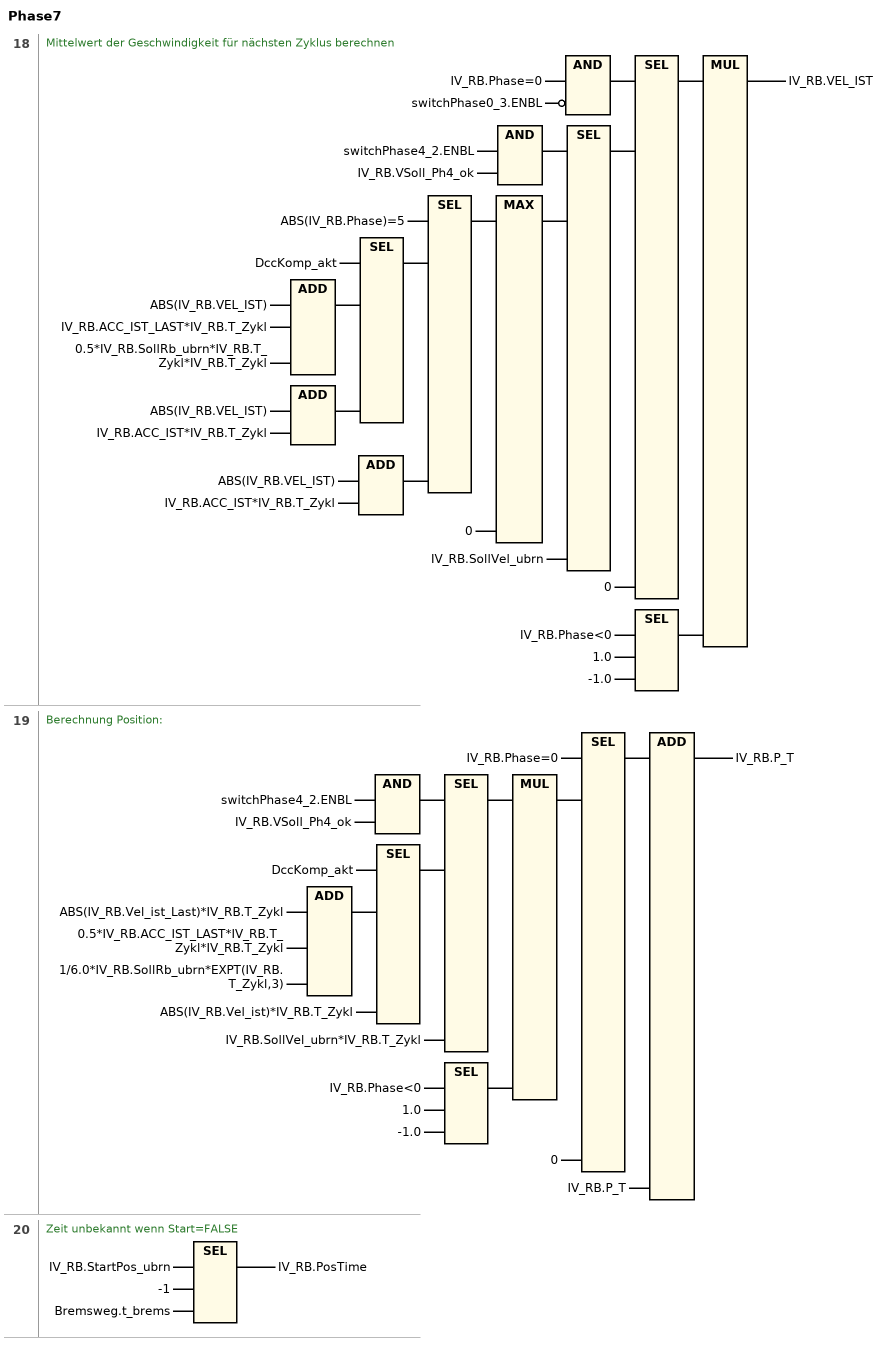
// NETWORK 18
// Mittelwert der Geschwindigkeit für nächsten Zyklus berechnen
IV_RB.VEL_IST := SEL((IV_RB.Phase=0) AND NOT switchPhase0_3.ENBL, SEL(switchPhase4_2.ENBL AND IV_RB.VSoll_Ph4_ok, MAX(SEL(ABS(IV_RB.Phase)=5, SEL(DccKomp_akt, (ABS(IV_RB.VEL_IST)) + (IV_RB.ACC_IST_LAST*IV_RB.T_Zykl) + (0.5*IV_RB.SollRb_ubrn*IV_RB.T_Zykl*IV_RB.T_Zykl), (ABS(IV_RB.VEL_IST)) + (IV_RB.ACC_IST*IV_RB.T_Zykl)), (ABS(IV_RB.VEL_IST)) + (IV_RB.ACC_IST*IV_RB.T_Zykl)), 0), IV_RB.SollVel_ubrn), 0) * SEL(IV_RB.Phase<0, 1.0, -1.0);

// NETWORK 19
// Berechnung Position:
IV_RB.P_T := SEL(IV_RB.Phase=0, SEL(switchPhase4_2.ENBL AND IV_RB.VSoll_Ph4_ok, SEL(DccKomp_akt, (ABS(IV_RB.Vel_ist_Last)*IV_RB.T_Zykl) + (0.5*IV_RB.ACC_IST_LAST*IV_RB.T_Zykl*IV_RB.T_Zykl) + (1/6.0*IV_RB.SollRb_ubrn*EXPT(IV_RB.T_Zykl,3)), ABS(IV_RB.Vel_ist)*IV_RB.T_Zykl), IV_RB.SollVel_ubrn*IV_RB.T_Zykl) * SEL(IV_RB.Phase<0, 1.0, -1.0), 0) + IV_RB.P_T;

// NETWORK 20
// Zeit unbekannt wenn Start=FALSE
IV_RB.PosTime := SEL(IV_RB.StartPos_ubrn, -1, Bremsweg.t_brems);

END_FUNCTION_BLOCK

// POUs/Achsen_Bausteinen/FB/calc_Val7_inPhase7
FUNCTION_BLOCK calc_Val7_inPhase7 (* Die Funktion gibt die Werte S7,t7,VE7 zurück, die bis zum erreichen von ACC=0 erreicht werden, wenn die Achse in Phase 5,6 oder 7 ist, d.h. wenn sofort Phase 7 eingeleitet würde*)
VAR_INPUT
	VEL_IST: LREAL;(*das Vorzeichen hat keine Relevanz da ABS gebildet wird *)
	ACC_IST:LREAL; (*das Vorzeichen hat keine Relevanz da ABS gebildet wird. Istbeschleunigung*)
	RB:LREAL;(*Ruckbegrenzung mm/s^3*)
END_VAR
VAR_OUTPUT
	t7: LREAL;			(*Restzeit in Phase 7*)
	S7: LREAL;			(*Reststrecke in Phase 7*)
	VE7A:LREAL; (* VE7 bei erreichen von ACC_IST=0. Ist der wert negativ, dann kann bis zum Stillstand der Achse ACC_IST nicht mehr auf 0 abgebaut werden*)
END_VAR
VAR
	VEL_ISTA: LREAL;
	DV7P: LREAL;
	ACC_ISTA: LREAL;
END_VAR

VEL_ISTA:=ABS(VEL_IST);
ACC_ISTA:=ABS(ACC_IST);

IF RB<=0 THEN
	t7:=0;
	DV7P:=0;
	S7:=0;
	VE7A:=VEL_ISTA;
	RETURN;
END_IF

t7:=ACC_ISTA / RB; (*Zeit bis ACC_IST=0*)
DV7P:= 0.5 * EXPT(ACC_ISTA, 2) / RB; (*DV7*)
VE7A:=MAX(0,(VEL_ISTA - DV7P));
S7:= ( VEL_ISTA - 1/3.0 * ACC_ISTA * t7 ) * t7;
S7:=MAX(S7,0);

END_FUNCTION_BLOCK

// POUs/Achsen_Bausteinen/FB/calc_Val67_inPhase6
FUNCTION_BLOCK calc_Val67_inPhase6 (*Die Funktion berechnet die Werte t6,t7,S6,S7 während der Phase 6.
*)
VAR_INPUT
	VEL_IST: LREAL;(*das Vorzeichen hat keine Relevanz da ABS gebildet wird *)
	DCC6:LREAL; (*Beschleunigung in Phase6, positiver Wert *)
	VE7_D:LREAL;(*gewünschte Endgeschwindigkeit am Ende von Phase7. ist beim Zielpositionieren = 0.*)
	RB:LREAL;(*Ruckbegrenzung mm/s^3*)
END_VAR
VAR_OUTPUT
	t6: LREAL;			(*Restzeit in Phase 6*)
	t7: LREAL;			(*Restzeit in Phase 7*)
	S6: LREAL;			(*Reststrecke in Phase 6*)
	S7: LREAL;			(*Reststrecke in Phase 7*)
END_VAR
VAR
	VEL_ISTA: LREAL;
	VE7_DA: LREAL;
	DV7P: LREAL;
	DV6P: LREAL;
	DCC6A: LREAL;
END_VAR

VEL_ISTA:=ABS(VEL_IST);
VE7_DA:=MIN(ABS(VE7_D),VEL_ISTA);(*VE7_DA muss eine kleiner Geschwindigkeit als die Istgeschwindigkeit sein*)
DCC6A:=ABS(DCC6);
IF DCC6A=0 THEN RETURN;END_IF

IF RB<=0 THEN
	t7:=0;
	DV7P:=0;
	S7:=0;
	DV6P:=VEL_ISTA - VE7_DA;
	t6:=DV6P / DCC6A;
	S6:=(VEL_ISTA - 0.5 * DCC6A * t6) * t6;
	RETURN;
END_IF

t7:=DCC6A / RB; (*Zeit für Phase 7*)
DV7P:= ( DCC6A - 0.5 * RB * t7)* t7;
S7:=(VE7_DA + DV7P -  0.5*DCC6A*t7 +  1/6.0*RB*EXPT(t7,2))*t7;
S7:=MAX(S7,0);

DV6P:=VEL_ISTA - DV7P - VE7_DA;
t6:=DV6P / DCC6A;
S6:=(VEL_ISTA - 0.5 * DCC6A * t6) * t6;

END_FUNCTION_BLOCK

// POUs/Achsen_Bausteinen/FB/CDLR
FUNCTION_BLOCK CDLR
VAR_INPUT
	IN: LREAL;
END_VAR
VAR_OUTPUT
	Q: BOOL;
END_VAR
VAR
	IN_LAST: LREAL;
END_VAR

Q:=IN <> IN_LAST;
IN_LAST:=IN;

END_FUNCTION_BLOCK

// POUs/Achsen_Bausteinen/FB/Phase0
FUNCTION_BLOCK Phase0
VAR_INPUT
	Achs_CMD:TKont_Achse_OUT;
	P_T: LREAL;
	REFSTATUS: INT;
	RefVel1: LREAL;
	RefVel2: LREAL;
END_VAR
VAR_OUTPUT
END_VAR
VAR_IN_OUT
	IV_RB: TIV_RB;
END_VAR
VAR
	Bremsweg: Bremsweg;
	switchPhase: switchPhase;
END_VAR
VAR // added by the converter: edge detectors and wires of the graphical bodies
    _w1, _w2 : BOOL;
END_VAR

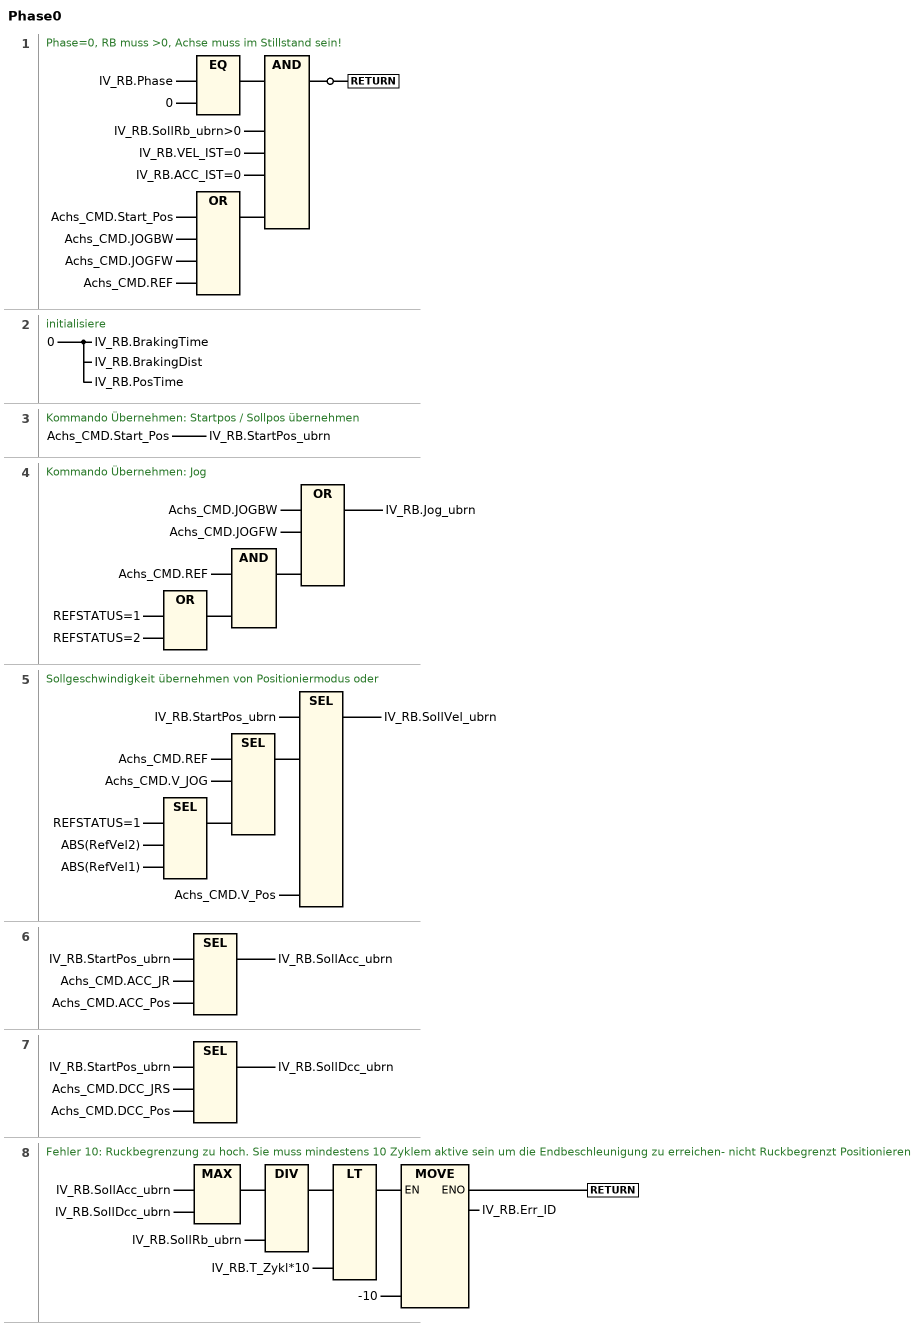
// NETWORK 1
// Phase=0, RB muss >0, Achse muss im Stillstand sein!
IF NOT (IV_RB.Phase = 0 AND (IV_RB.SollRb_ubrn>0) AND (IV_RB.VEL_IST=0) AND (IV_RB.ACC_IST=0) AND (Achs_CMD.Start_Pos OR Achs_CMD.JOGBW OR Achs_CMD.JOGFW OR Achs_CMD.REF)) THEN RETURN; END_IF

// NETWORK 2
// initialisiere
IV_RB.BrakingTime := 0;
IV_RB.BrakingDist := 0;
IV_RB.PosTime := 0;

// NETWORK 3
// Kommando Übernehmen: Startpos / Sollpos übernehmen
IV_RB.StartPos_ubrn := Achs_CMD.Start_Pos;

// NETWORK 4
// Kommando Übernehmen: Jog
IV_RB.Jog_ubrn := Achs_CMD.JOGBW OR Achs_CMD.JOGFW OR Achs_CMD.REF AND ((REFSTATUS=1) OR (REFSTATUS=2));

// NETWORK 5
// Sollgeschwindigkeit übernehmen von Positioniermodus oder
IV_RB.SollVel_ubrn := SEL(IV_RB.StartPos_ubrn, SEL(Achs_CMD.REF, Achs_CMD.V_JOG, SEL(REFSTATUS=1, ABS(RefVel2), ABS(RefVel1))), Achs_CMD.V_Pos);

// NETWORK 6
IV_RB.SollAcc_ubrn := SEL(IV_RB.StartPos_ubrn, Achs_CMD.ACC_JR, Achs_CMD.ACC_Pos);

// NETWORK 7
IV_RB.SollDcc_ubrn := SEL(IV_RB.StartPos_ubrn, Achs_CMD.DCC_JRS, Achs_CMD.DCC_Pos);

// NETWORK 8
// Fehler 10: Ruckbegrenzung zu hoch. Sie muss mindestens 10 Zyklem aktive sein um die Endbeschleunigung zu erreichen- nicht Ruckbegrenzt Positionieren
_w1 := MAX(IV_RB.SollAcc_ubrn, IV_RB.SollDcc_ubrn) / IV_RB.SollRb_ubrn < (IV_RB.T_Zykl*10);
IF _w1 THEN IV_RB.Err_ID := -10; END_IF
IF _w1 THEN RETURN; END_IF

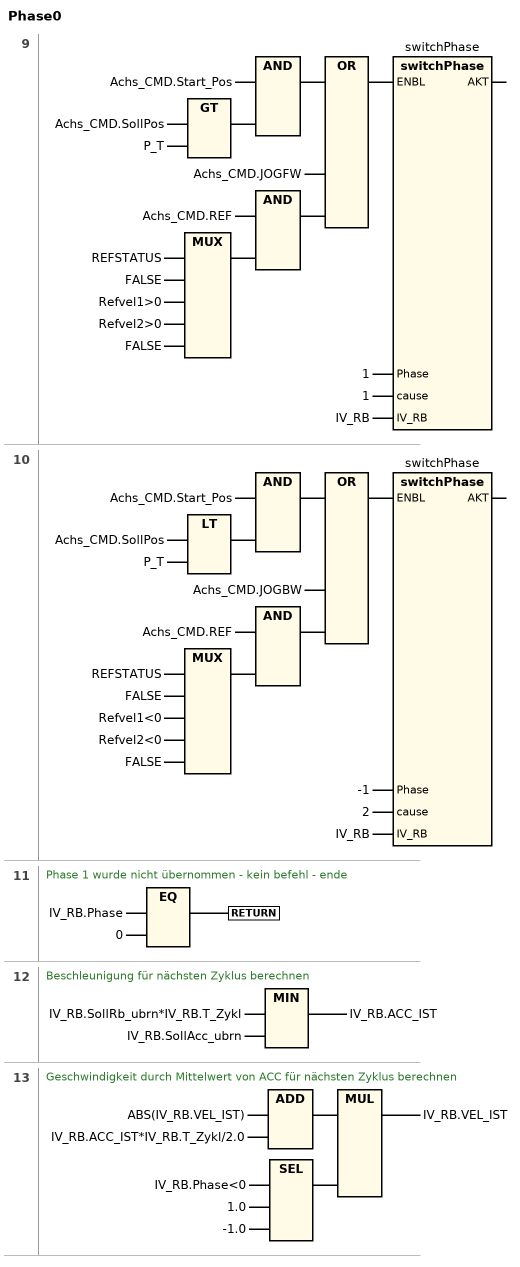
// NETWORK 9
switchPhase(
    ENBL := Achs_CMD.Start_Pos AND Achs_CMD.SollPos > P_T OR Achs_CMD.JOGFW OR Achs_CMD.REF AND MUX(REFSTATUS, FALSE, Refvel1>0, Refvel2>0, FALSE),
    Phase := 1,
    cause := 1,
    IV_RB := IV_RB);

// NETWORK 10
switchPhase(
    ENBL := Achs_CMD.Start_Pos AND Achs_CMD.SollPos < P_T OR Achs_CMD.JOGBW OR Achs_CMD.REF AND MUX(REFSTATUS, FALSE, Refvel1<0, Refvel2<0, FALSE),
    Phase := -1,
    cause := 2,
    IV_RB := IV_RB);

// NETWORK 11
// Phase 1 wurde nicht übernommen - kein befehl - ende
IF IV_RB.Phase = 0 THEN RETURN; END_IF

// NETWORK 12
// Beschleunigung für nächsten Zyklus berechnen
IV_RB.ACC_IST := MIN(IV_RB.SollRb_ubrn*IV_RB.T_Zykl, IV_RB.SollAcc_ubrn);

// NETWORK 13
// Geschwindigkeit durch Mittelwert von ACC für nächsten Zyklus berechnen
IV_RB.VEL_IST := ((ABS(IV_RB.VEL_IST)) + (IV_RB.ACC_IST*IV_RB.T_Zykl/2.0)) * SEL(IV_RB.Phase<0, 1.0, -1.0);

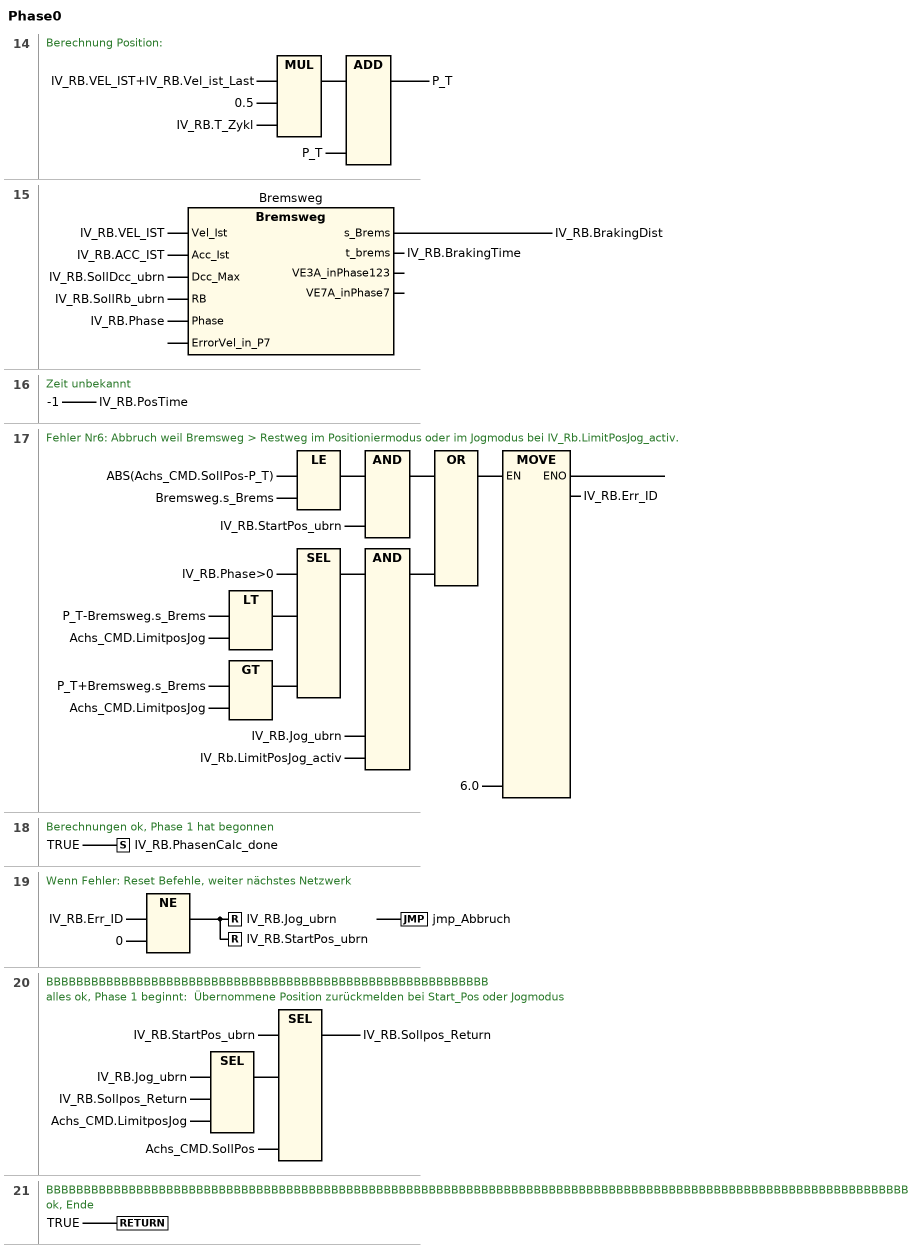
// NETWORK 14
// Berechnung Position:
P_T := (IV_RB.VEL_IST+IV_RB.Vel_ist_Last) * 0.5 * IV_RB.T_Zykl + P_T;

// NETWORK 15
Bremsweg(
    Vel_Ist := IV_RB.VEL_IST,
    Acc_Ist := IV_RB.ACC_IST,
    Dcc_Max := IV_RB.SollDcc_ubrn,
    RB := IV_RB.SollRb_ubrn,
    Phase := IV_RB.Phase,
    t_brems => IV_RB.BrakingTime);
IV_RB.BrakingDist := Bremsweg.s_Brems;

// NETWORK 16
// Zeit unbekannt
IV_RB.PosTime := -1;

// NETWORK 17
// Fehler Nr6: Abbruch weil Bremsweg > Restweg im Positioniermodus oder im Jogmodus bei IV_Rb.LimitPosJog_activ.
IF (ABS(Achs_CMD.SollPos-P_T)) <= Bremsweg.s_Brems AND IV_RB.StartPos_ubrn OR SEL(IV_RB.Phase>0, (P_T-Bremsweg.s_Brems) < Achs_CMD.LimitposJog, (P_T+Bremsweg.s_Brems) > Achs_CMD.LimitposJog) AND IV_RB.Jog_ubrn AND IV_Rb.LimitPosJog_activ THEN
    IV_RB.Err_ID := 6.0;
END_IF

// NETWORK 18
// Berechnungen ok, Phase 1 hat begonnen
IV_RB.PhasenCalc_done S= TRUE;

// NETWORK 19
// Wenn Fehler: Reset Befehle, weiter nächstes Netzwerk
_w2 := IV_RB.Err_ID <> 0;
IV_RB.Jog_ubrn R= _w2;
IV_RB.StartPos_ubrn R= _w2;
IF _w2 THEN JMP jmp_Abbruch; END_IF

// NETWORK 20
// 					BBBBBBBBBBBBBBBBBBBBBBBBBBBBBBBBBBBBBBBBBBBBBBBBBBBBBBBBBBB
// alles ok, Phase 1 beginnt:  Übernommene Position zurückmelden bei Start_Pos oder Jogmodus
//
IV_RB.Sollpos_Return := SEL(IV_RB.StartPos_ubrn, SEL(IV_RB.Jog_ubrn, IV_RB.Sollpos_Return, Achs_CMD.LimitposJog), Achs_CMD.SollPos);

// NETWORK 21
// 					BBBBBBBBBBBBBBBBBBBBBBBBBBBBBBBBBBBBBBBBBBBBBBBBBBBBBBBBBBBBBBBBBBBBBBBBBBBBBBBBBBBBBBBBBBBBBBBBBBBBBBBBBBBBBBBBBBB
// ok, Ende
//
RETURN;

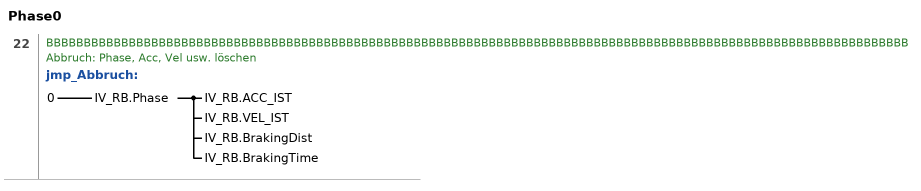
// NETWORK 22
// 					BBBBBBBBBBBBBBBBBBBBBBBBBBBBBBBBBBBBBBBBBBBBBBBBBBBBBBBBBBBBBBBBBBBBBBBBBBBBBBBBBBBBBBBBBBBBBBBBBBBBBBBBBBBBBBBBBBB
// Abbruch: Phase, Acc, Vel usw. löschen
//
jmp_Abbruch:
IV_RB.Phase := 0;
IV_RB.ACC_IST := 0;
IV_RB.VEL_IST := 0;
IV_RB.BrakingDist := 0;
IV_RB.BrakingTime := 0;

END_FUNCTION_BLOCK

// POUs/Achsen_Bausteinen/FB/Phase12
FUNCTION_BLOCK Phase12
VAR_INPUT
	Achs_CMD:TKont_Achse_OUT;
END_VAR
VAR_OUTPUT
END_VAR
VAR_IN_OUT
	IV_RB: TIV_RB;
END_VAR
VAR
	Bremsweg: Bremsweg;
	SollDcc: LREAL;		(*zu prüfender DCC-Wert bzw. Sollwerrt von Achs_CMD*)
	VE3Limit: BOOL;		(*VE3-Limit ist wegen V-Soll erreicht*)
	Temp_Lreal: LREAL;
	aktiv_: BOOL;
	First_Cykl_: BOOL;(*erster Zyklus der Bearbeitung dieser Phase in diesem Basutein*)
	switchPhase3_1: switchPhase;
	switchPhase3_2: switchPhase;
	switchPhase3_3: switchPhase;
	switchPhase2_1: switchPhase;
	switchPhase1_3: switchPhase;
END_VAR
VAR // added by the converter: edge detectors and wires of the graphical bodies
    _w1, _w2, _w5, _w6, _w7, _w8 : BOOL;
    _w3, _w4 : LREAL;
END_VAR

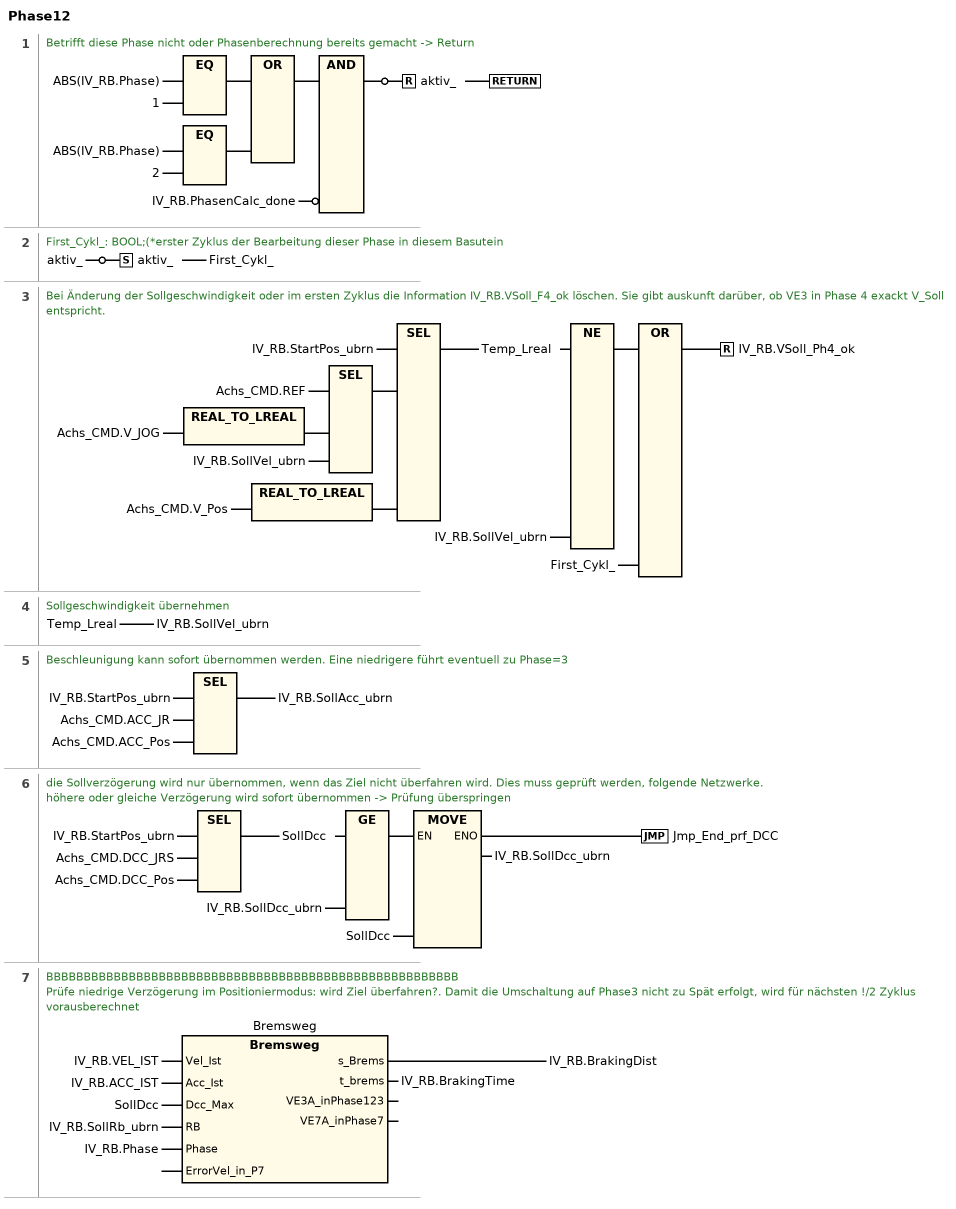
// NETWORK 1
// Betrifft diese Phase nicht oder Phasenberechnung bereits gemacht -> Return
_w1 := NOT (((ABS(IV_RB.Phase)) = 1 OR (ABS(IV_RB.Phase)) = 2) AND NOT IV_RB.PhasenCalc_done);
aktiv_ R= _w1;
IF _w1 THEN RETURN; END_IF

// NETWORK 2
// First_Cykl_: BOOL;(*erster Zyklus der Bearbeitung dieser Phase in diesem Basutein
_w2 := NOT aktiv_;
aktiv_ S= _w2;
First_Cykl_ := _w2;

// NETWORK 3
// Bei Änderung der Sollgeschwindigkeit oder im ersten Zyklus die Information IV_RB.VSoll_F4_ok löschen. Sie gibt auskunft darüber, ob VE3 in Phase 4 exackt V_Soll entspricht.
_w3 := SEL(IV_RB.StartPos_ubrn, SEL(Achs_CMD.REF, REAL_TO_LREAL(Achs_CMD.V_JOG), IV_RB.SollVel_ubrn), REAL_TO_LREAL(Achs_CMD.V_Pos));
Temp_Lreal := _w3;
IV_RB.VSoll_Ph4_ok R= _w3 <> IV_RB.SollVel_ubrn OR First_Cykl_;

// NETWORK 4
// Sollgeschwindigkeit übernehmen
IV_RB.SollVel_ubrn := Temp_Lreal;

// NETWORK 5
// Beschleunigung kann sofort übernommen werden. Eine niedrigere führt eventuell zu Phase=3
IV_RB.SollAcc_ubrn := SEL(IV_RB.StartPos_ubrn, Achs_CMD.ACC_JR, Achs_CMD.ACC_Pos);

// NETWORK 6
// 					die Sollverzögerung wird nur übernommen, wenn das Ziel nicht überfahren wird. Dies muss geprüft werden, folgende Netzwerke.
// höhere oder gleiche Verzögerung wird sofort übernommen -> Prüfung überspringen
//
_w4 := SEL(IV_RB.StartPos_ubrn, Achs_CMD.DCC_JRS, Achs_CMD.DCC_Pos);
SollDcc := _w4;
IF _w4 >= IV_RB.SollDcc_ubrn THEN IV_RB.SollDcc_ubrn := SollDcc; END_IF
IF _w4 >= IV_RB.SollDcc_ubrn THEN JMP Jmp_End_prf_DCC; END_IF

// NETWORK 7
// 					BBBBBBBBBBBBBBBBBBBBBBBBBBBBBBBBBBBBBBBBBBBBBBBBBBBBBBB
// Prüfe niedrige Verzögerung im Positioniermodus: wird Ziel überfahren?. Damit die Umschaltung auf Phase3 nicht zu Spät erfolgt, wird für nächsten !/2 Zyklus vorausberechnet
//
Bremsweg(
    Vel_Ist := IV_RB.VEL_IST,
    Acc_Ist := IV_RB.ACC_IST,
    Dcc_Max := SollDcc,
    RB := IV_RB.SollRb_ubrn,
    Phase := IV_RB.Phase,
    t_brems => IV_RB.BrakingTime);
IV_RB.BrakingDist := Bremsweg.s_Brems;

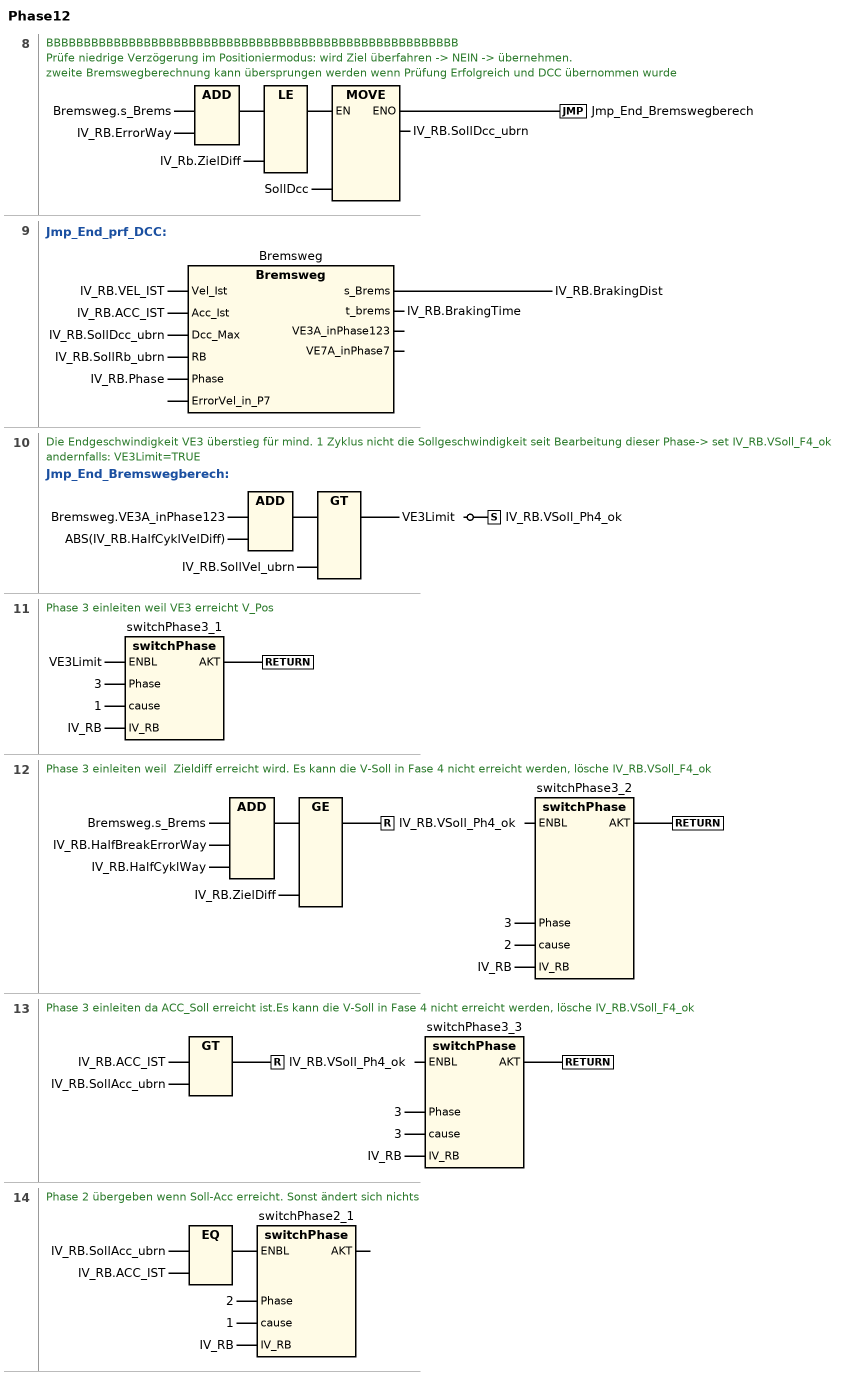
// NETWORK 8
// 					BBBBBBBBBBBBBBBBBBBBBBBBBBBBBBBBBBBBBBBBBBBBBBBBBBBBBBB
// Prüfe niedrige Verzögerung im Positioniermodus: wird Ziel überfahren -> NEIN -> übernehmen.
// zweite Bremswegberechnung kann übersprungen werden wenn Prüfung Erfolgreich und DCC übernommen wurde
//
_w5 := Bremsweg.s_Brems + IV_RB.ErrorWay <= IV_Rb.ZielDiff;
IF _w5 THEN IV_RB.SollDcc_ubrn := SollDcc; END_IF
IF _w5 THEN JMP Jmp_End_Bremswegberech; END_IF

// NETWORK 9
Jmp_End_prf_DCC:
Bremsweg(
    Vel_Ist := IV_RB.VEL_IST,
    Acc_Ist := IV_RB.ACC_IST,
    Dcc_Max := IV_RB.SollDcc_ubrn,
    RB := IV_RB.SollRb_ubrn,
    Phase := IV_RB.Phase,
    t_brems => IV_RB.BrakingTime);
IV_RB.BrakingDist := Bremsweg.s_Brems;

// NETWORK 10
// 					Die Endgeschwindigkeit VE3 überstieg für mind. 1 Zyklus nicht die Sollgeschwindigkeit seit Bearbeitung dieser Phase-> set IV_RB.VSoll_F4_ok
// andernfalls: VE3Limit=TRUE
//
Jmp_End_Bremswegberech:
_w6 := Bremsweg.VE3A_inPhase123 + (ABS(IV_RB.HalfCyklVelDiff)) > IV_RB.SollVel_ubrn;
VE3Limit := _w6;
IV_RB.VSoll_Ph4_ok S= NOT _w6;

// NETWORK 11
// Phase 3 einleiten weil VE3 erreicht V_Pos
switchPhase3_1(ENBL := VE3Limit, Phase := 3, cause := 1, IV_RB := IV_RB); // switchPhase
IF switchPhase3_1.AKT THEN RETURN; END_IF

// NETWORK 12
// Phase 3 einleiten weil  Zieldiff erreicht wird. Es kann die V-Soll in Fase 4 nicht erreicht werden, lösche IV_RB.VSoll_F4_ok
_w7 := Bremsweg.s_Brems + IV_RB.HalfBreakErrorWay + IV_RB.HalfCyklWay >= IV_RB.ZielDiff;
IV_RB.VSoll_Ph4_ok R= _w7;
switchPhase3_2(ENBL := _w7, Phase := 3, cause := 2, IV_RB := IV_RB); // switchPhase
IF switchPhase3_2.AKT THEN RETURN; END_IF

// NETWORK 13
// Phase 3 einleiten da ACC_Soll erreicht ist.Es kann die V-Soll in Fase 4 nicht erreicht werden, lösche IV_RB.VSoll_F4_ok
_w8 := IV_RB.ACC_IST > IV_RB.SollAcc_ubrn;
IV_RB.VSoll_Ph4_ok R= _w8;
switchPhase3_3(ENBL := _w8, Phase := 3, cause := 3, IV_RB := IV_RB); // switchPhase
IF switchPhase3_3.AKT THEN RETURN; END_IF

// NETWORK 14
// Phase 2 übergeben wenn Soll-Acc erreicht. Sonst ändert sich nichts
switchPhase2_1(ENBL := IV_RB.SollAcc_ubrn = IV_RB.ACC_IST, Phase := 2, cause := 1, IV_RB := IV_RB); // switchPhase

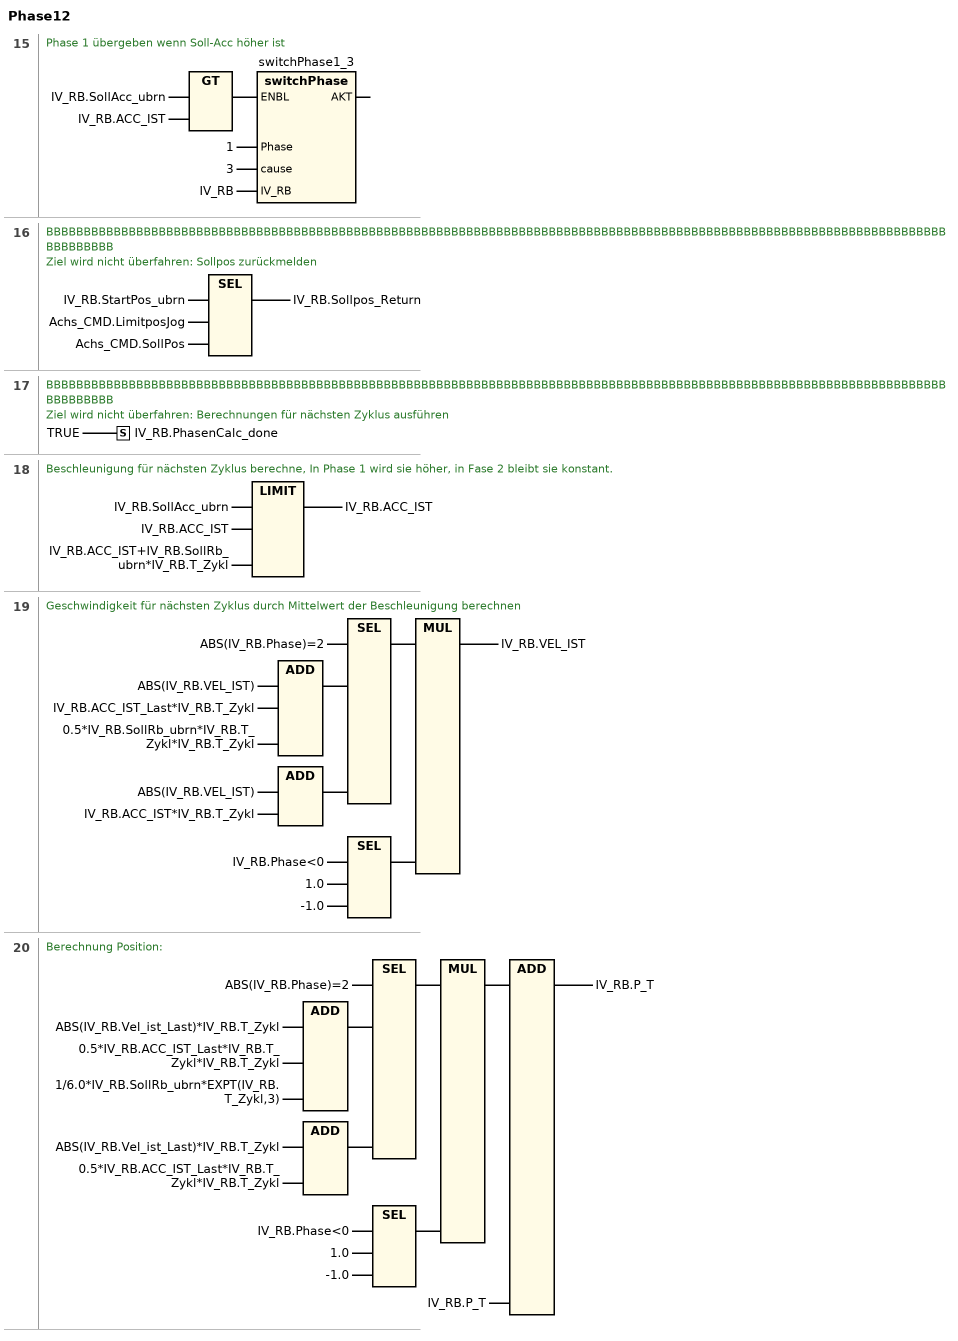
// NETWORK 15
// Phase 1 übergeben wenn Soll-Acc höher ist
switchPhase1_3(ENBL := IV_RB.SollAcc_ubrn > IV_RB.ACC_IST, Phase := 1, cause := 3, IV_RB := IV_RB); // switchPhase

// NETWORK 16
// 					BBBBBBBBBBBBBBBBBBBBBBBBBBBBBBBBBBBBBBBBBBBBBBBBBBBBBBBBBBBBBBBBBBBBBBBBBBBBBBBBBBBBBBBBBBBBBBBBBBBBBBBBBBBBBBBBBBBBBBBBBBBBBBBBB
// Ziel wird nicht überfahren: Sollpos zurückmelden
//
IV_RB.Sollpos_Return := SEL(IV_RB.StartPos_ubrn, Achs_CMD.LimitposJog, Achs_CMD.SollPos);

// NETWORK 17
// 					BBBBBBBBBBBBBBBBBBBBBBBBBBBBBBBBBBBBBBBBBBBBBBBBBBBBBBBBBBBBBBBBBBBBBBBBBBBBBBBBBBBBBBBBBBBBBBBBBBBBBBBBBBBBBBBBBBBBBBBBBBBBBBBBB
// Ziel wird nicht überfahren: Berechnungen für nächsten Zyklus ausführen
//
IV_RB.PhasenCalc_done S= TRUE;

// NETWORK 18
// Beschleunigung für nächsten Zyklus berechne, In Phase 1 wird sie höher, in Fase 2 bleibt sie konstant.
IV_RB.ACC_IST := LIMIT(IV_RB.SollAcc_ubrn, IV_RB.ACC_IST, IV_RB.ACC_IST+IV_RB.SollRb_ubrn*IV_RB.T_Zykl);

// NETWORK 19
// Geschwindigkeit für nächsten Zyklus durch Mittelwert der Beschleunigung berechnen
IV_RB.VEL_IST := SEL(ABS(IV_RB.Phase)=2, (ABS(IV_RB.VEL_IST)) + (IV_RB.ACC_IST_Last*IV_RB.T_Zykl) + (0.5*IV_RB.SollRb_ubrn*IV_RB.T_Zykl*IV_RB.T_Zykl), (ABS(IV_RB.VEL_IST)) + (IV_RB.ACC_IST*IV_RB.T_Zykl)) * SEL(IV_RB.Phase<0, 1.0, -1.0);

// NETWORK 20
// Berechnung Position:
IV_RB.P_T := SEL(ABS(IV_RB.Phase)=2, (ABS(IV_RB.Vel_ist_Last)*IV_RB.T_Zykl) + (0.5*IV_RB.ACC_IST_Last*IV_RB.T_Zykl*IV_RB.T_Zykl) + (1/6.0*IV_RB.SollRb_ubrn*EXPT(IV_RB.T_Zykl,3)), (ABS(IV_RB.Vel_ist_Last)*IV_RB.T_Zykl) + (0.5*IV_RB.ACC_IST_Last*IV_RB.T_Zykl*IV_RB.T_Zykl)) * SEL(IV_RB.Phase<0, 1.0, -1.0) + IV_RB.P_T;

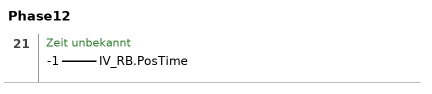
// NETWORK 21
// Zeit unbekannt
IV_RB.PosTime := -1;

END_FUNCTION_BLOCK

// POUs/Achsen_Bausteinen/FB/Phase4
FUNCTION_BLOCK Phase4
VAR_INPUT
	Achs_CMD:TKont_Achse_OUT;
END_VAR
VAR_OUTPUT
END_VAR
VAR_IN_OUT
	IV_RB: TIV_RB;
END_VAR
VAR
	Bremsweg: Bremsweg;
	SollDcc: LREAL;		(*zu prüfender DCC-Wert bzw. Sollwerrt von Achs_CMD*)
	switchPhase5_1: switchPhase;
	switchPhase5_2: switchPhase;
	switchPhase1_4: switchPhase;
END_VAR
VAR // added by the converter: edge detectors and wires of the graphical bodies
    _w1 : LREAL;
    _w2 : BOOL;
END_VAR

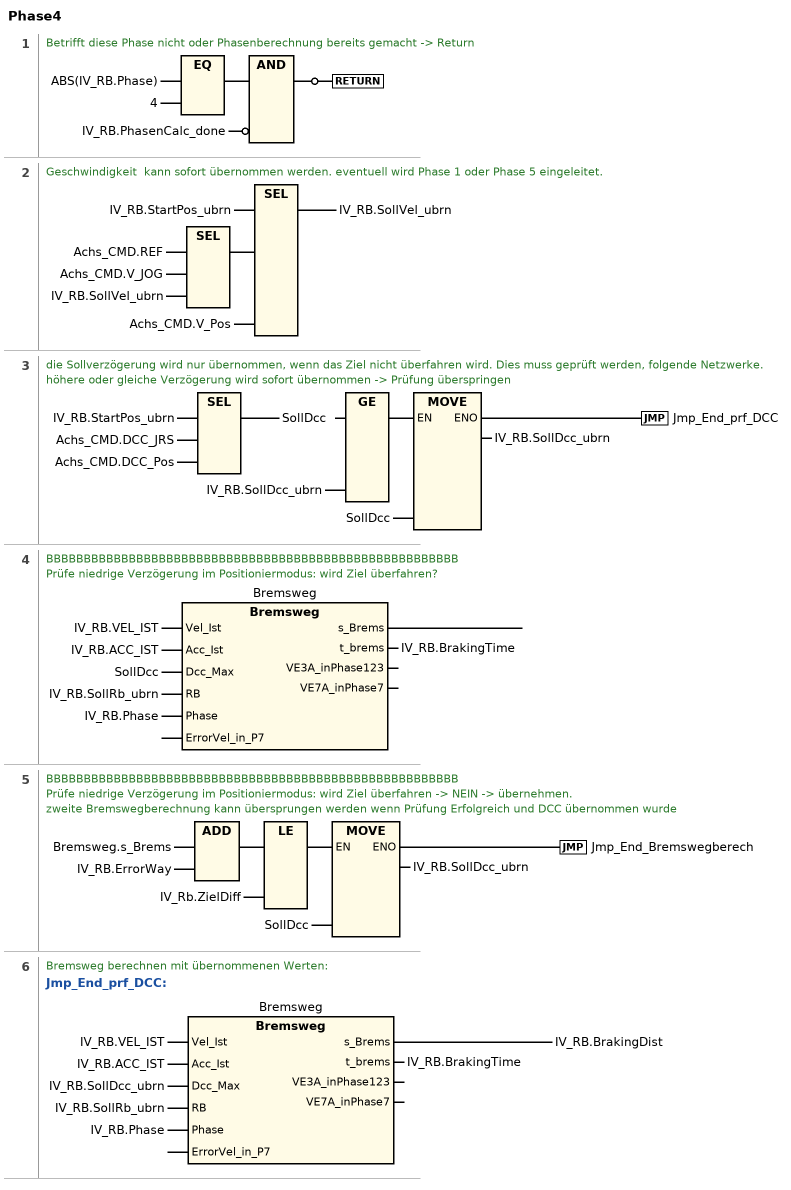
// NETWORK 1
// Betrifft diese Phase nicht oder Phasenberechnung bereits gemacht -> Return
IF NOT ((ABS(IV_RB.Phase)) = 4 AND NOT IV_RB.PhasenCalc_done) THEN RETURN; END_IF

// NETWORK 2
// Geschwindigkeit  kann sofort übernommen werden. eventuell wird Phase 1 oder Phase 5 eingeleitet.
IV_RB.SollVel_ubrn := SEL(IV_RB.StartPos_ubrn, SEL(Achs_CMD.REF, Achs_CMD.V_JOG, IV_RB.SollVel_ubrn), Achs_CMD.V_Pos);

// NETWORK 3
// 					die Sollverzögerung wird nur übernommen, wenn das Ziel nicht überfahren wird. Dies muss geprüft werden, folgende Netzwerke.
// höhere oder gleiche Verzögerung wird sofort übernommen -> Prüfung überspringen
//
_w1 := SEL(IV_RB.StartPos_ubrn, Achs_CMD.DCC_JRS, Achs_CMD.DCC_Pos);
SollDcc := _w1;
IF _w1 >= IV_RB.SollDcc_ubrn THEN IV_RB.SollDcc_ubrn := SollDcc; END_IF
IF _w1 >= IV_RB.SollDcc_ubrn THEN JMP Jmp_End_prf_DCC; END_IF

// NETWORK 4
// 					BBBBBBBBBBBBBBBBBBBBBBBBBBBBBBBBBBBBBBBBBBBBBBBBBBBBBBB
// Prüfe niedrige Verzögerung im Positioniermodus: wird Ziel überfahren?
//
Bremsweg(
    Vel_Ist := IV_RB.VEL_IST,
    Acc_Ist := IV_RB.ACC_IST,
    Dcc_Max := SollDcc,
    RB := IV_RB.SollRb_ubrn,
    Phase := IV_RB.Phase,
    t_brems => IV_RB.BrakingTime);

// NETWORK 5
// 					BBBBBBBBBBBBBBBBBBBBBBBBBBBBBBBBBBBBBBBBBBBBBBBBBBBBBBB
// Prüfe niedrige Verzögerung im Positioniermodus: wird Ziel überfahren -> NEIN -> übernehmen.
// zweite Bremswegberechnung kann übersprungen werden wenn Prüfung Erfolgreich und DCC übernommen wurde
//
_w2 := Bremsweg.s_Brems + IV_RB.ErrorWay <= IV_Rb.ZielDiff;
IF _w2 THEN IV_RB.SollDcc_ubrn := SollDcc; END_IF
IF _w2 THEN JMP Jmp_End_Bremswegberech; END_IF

// NETWORK 6
// Bremsweg berechnen mit übernommenen Werten:
Jmp_End_prf_DCC:
Bremsweg(
    Vel_Ist := IV_RB.VEL_IST,
    Acc_Ist := IV_RB.ACC_IST,
    Dcc_Max := IV_RB.SollDcc_ubrn,
    RB := IV_RB.SollRb_ubrn,
    Phase := IV_RB.Phase,
    t_brems => IV_RB.BrakingTime);
IV_RB.BrakingDist := Bremsweg.s_Brems;

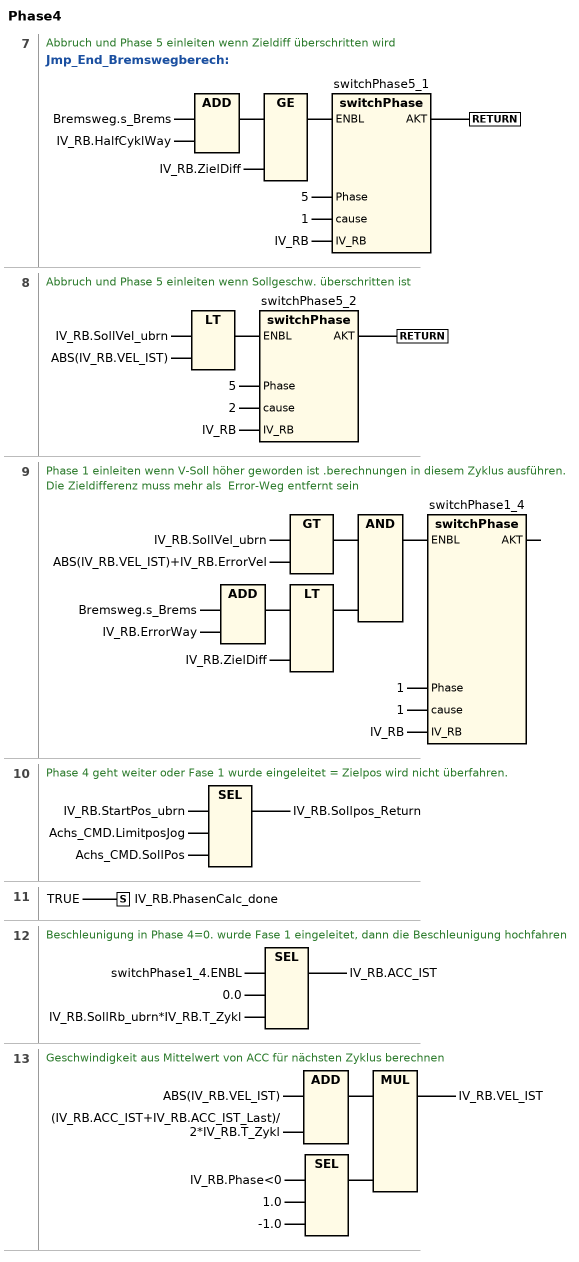
// NETWORK 7
// Abbruch und Phase 5 einleiten wenn Zieldiff überschritten wird
Jmp_End_Bremswegberech:
switchPhase5_1(
    ENBL := Bremsweg.s_Brems + IV_RB.HalfCyklWay >= IV_RB.ZielDiff,
    Phase := 5,
    cause := 1,
    IV_RB := IV_RB); // switchPhase
IF switchPhase5_1.AKT THEN RETURN; END_IF

// NETWORK 8
// Abbruch und Phase 5 einleiten wenn Sollgeschw. überschritten ist
switchPhase5_2(ENBL := IV_RB.SollVel_ubrn < (ABS(IV_RB.VEL_IST)), Phase := 5, cause := 2, IV_RB := IV_RB); // switchPhase
IF switchPhase5_2.AKT THEN RETURN; END_IF

// NETWORK 9
// 					Phase 1 einleiten wenn V-Soll höher geworden ist .berechnungen in diesem Zyklus ausführen.
// Die Zieldifferenz muss mehr als  Error-Weg entfernt sein
//
switchPhase1_4(
    ENBL := IV_RB.SollVel_ubrn > (ABS(IV_RB.VEL_IST)+IV_RB.ErrorVel) AND Bremsweg.s_Brems + IV_RB.ErrorWay < IV_RB.ZielDiff,
    Phase := 1,
    cause := 1,
    IV_RB := IV_RB); // switchPhase

// NETWORK 10
// Phase 4 geht weiter oder Fase 1 wurde eingeleitet = Zielpos wird nicht überfahren.
IV_RB.Sollpos_Return := SEL(IV_RB.StartPos_ubrn, Achs_CMD.LimitposJog, Achs_CMD.SollPos);

// NETWORK 11
IV_RB.PhasenCalc_done S= TRUE;

// NETWORK 12
// Beschleunigung in Phase 4=0. wurde Fase 1 eingeleitet, dann die Beschleunigung hochfahren
IV_RB.ACC_IST := SEL(switchPhase1_4.ENBL, 0.0, IV_RB.SollRb_ubrn*IV_RB.T_Zykl);

// NETWORK 13
// Geschwindigkeit aus Mittelwert von ACC für nächsten Zyklus berechnen
IV_RB.VEL_IST := ((ABS(IV_RB.VEL_IST)) + ((IV_RB.ACC_IST+IV_RB.ACC_IST_Last)/2*IV_RB.T_Zykl)) * SEL(IV_RB.Phase<0, 1.0, -1.0);

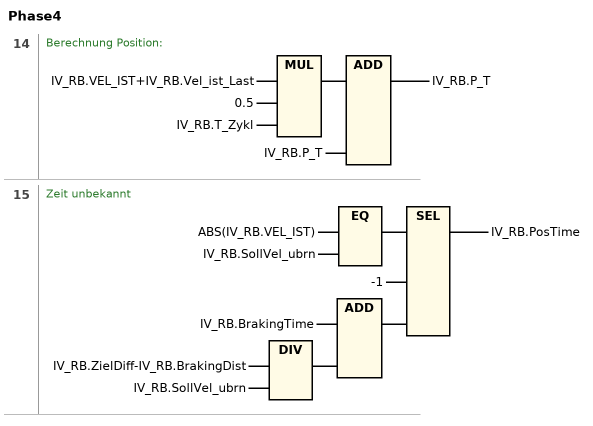
// NETWORK 14
// Berechnung Position:
IV_RB.P_T := (IV_RB.VEL_IST+IV_RB.Vel_ist_Last) * 0.5 * IV_RB.T_Zykl + IV_RB.P_T;

// NETWORK 15
// Zeit unbekannt
IV_RB.PosTime := SEL((ABS(IV_RB.VEL_IST)) = IV_RB.SollVel_ubrn, -1, IV_RB.BrakingTime + (IV_RB.ZielDiff-IV_RB.BrakingDist) / IV_RB.SollVel_ubrn);

END_FUNCTION_BLOCK

// POUs/Achsen_Bausteinen/FB/Phase56
FUNCTION_BLOCK Phase56
VAR_INPUT
	Achs_CMD:TKont_Achse_OUT;
END_VAR
VAR_OUTPUT
END_VAR
VAR_IN_OUT
	IV_RB: TIV_RB;
END_VAR
VAR
	Bremsweg: Bremsweg;
	SollDcc: LREAL;		(*zu prüfender DCC-Wert bzw. Sollwerrt von Achs_CMD*)
	SollVel: LREAL;
	First_Cykl_: BOOL;(*erster Zyklus der Bearbeitung dieser Phase in diesem Basutein*)
	aktiv_: BOOL;
	switchPhase7_1: switchPhase;
	switchPhase7_2: switchPhase;
	switchPhase7_3: switchPhase;
	switchPhase6_1: switchPhase;
	Prf_Vel_Zieldiff: Bremsweg;
	switchPhase7_4: switchPhase;
	Resweg_GT0: BOOL;		(*Reserveweg > 0 (Zieldiff noch nicht erreicht)*)
	switchPhase5_3: switchPhase;
END_VAR
VAR // added by the converter: edge detectors and wires of the graphical bodies
    _w1, _w2, _w4, _w5, _w6, _w7, _w8, _w9 : BOOL;
    _w3 : LREAL;
END_VAR

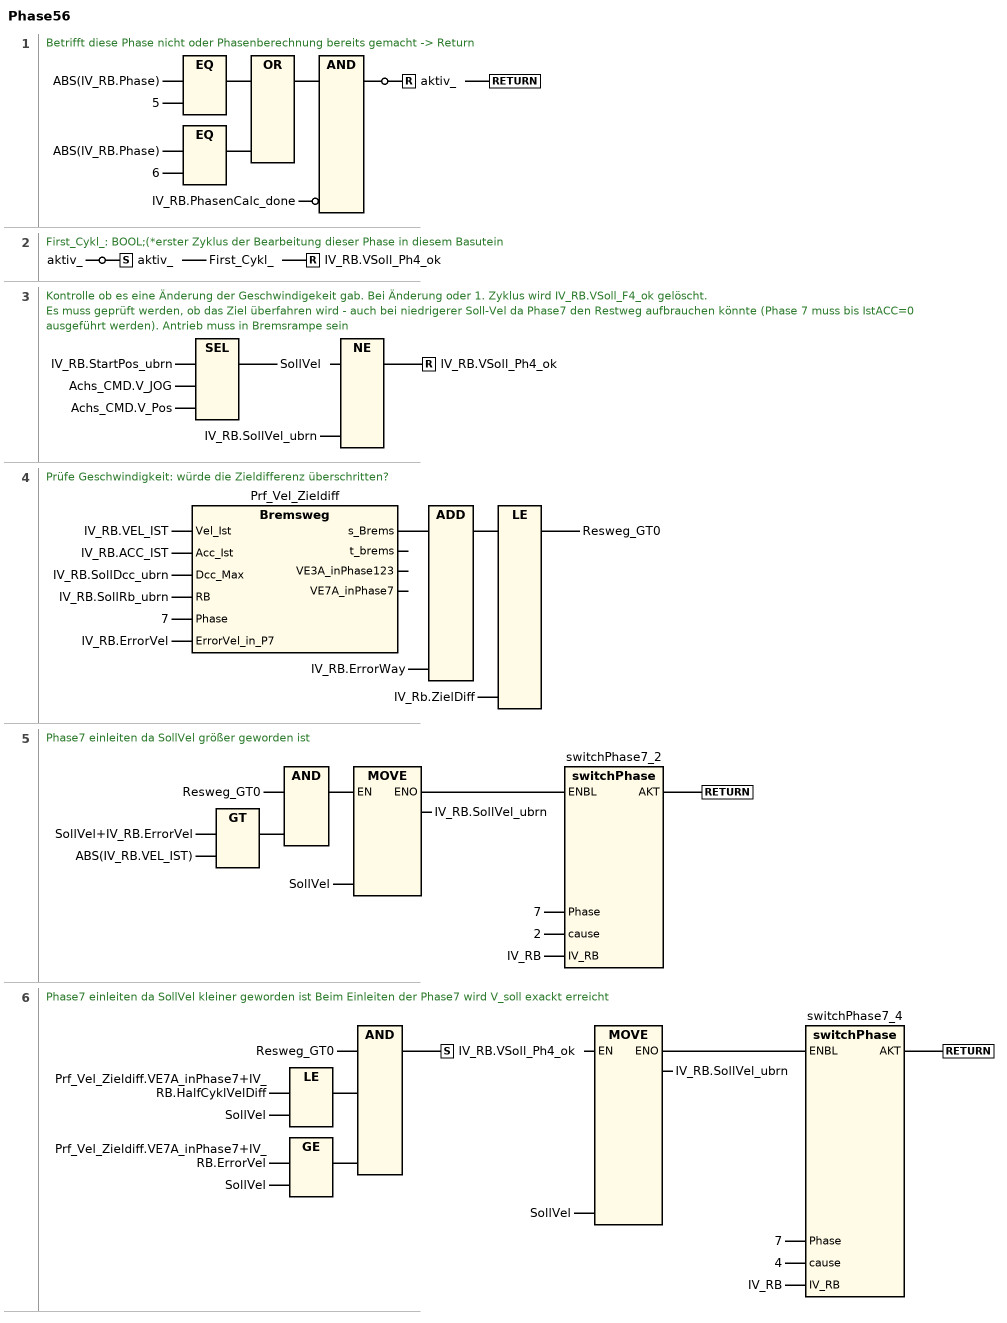
// NETWORK 1
// Betrifft diese Phase nicht oder Phasenberechnung bereits gemacht -> Return
_w1 := NOT (((ABS(IV_RB.Phase)) = 5 OR (ABS(IV_RB.Phase)) = 6) AND NOT IV_RB.PhasenCalc_done);
aktiv_ R= _w1;
IF _w1 THEN RETURN; END_IF

// NETWORK 2
// First_Cykl_: BOOL;(*erster Zyklus der Bearbeitung dieser Phase in diesem Basutein
_w2 := NOT aktiv_;
aktiv_ S= _w2;
First_Cykl_ := _w2;
IV_RB.VSoll_Ph4_ok R= _w2;

// NETWORK 3
// 					Kontrolle ob es eine Änderung der Geschwindigekeit gab. Bei Änderung oder 1. Zyklus wird IV_RB.VSoll_F4_ok gelöscht.
// Es muss geprüft werden, ob das Ziel überfahren wird - auch bei niedrigerer Soll-Vel da Phase7 den Restweg aufbrauchen könnte (Phase 7 muss bis IstACC=0 ausgeführt werden). Antrieb muss in Bremsrampe sein
//
_w3 := SEL(IV_RB.StartPos_ubrn, Achs_CMD.V_JOG, Achs_CMD.V_Pos);
SollVel := _w3;
IV_RB.VSoll_Ph4_ok R= _w3 <> IV_RB.SollVel_ubrn;

// NETWORK 4
// Prüfe Geschwindigkeit: würde die Zieldifferenz überschritten?
Prf_Vel_Zieldiff(
    Vel_Ist := IV_RB.VEL_IST,
    Acc_Ist := IV_RB.ACC_IST,
    Dcc_Max := IV_RB.SollDcc_ubrn,
    RB := IV_RB.SollRb_ubrn,
    Phase := 7,
    ErrorVel_in_P7 := IV_RB.ErrorVel); // Bremsweg
Resweg_GT0 := Prf_Vel_Zieldiff.s_Brems + IV_RB.ErrorWay <= IV_Rb.ZielDiff;

// NETWORK 5
// Phase7 einleiten da SollVel größer geworden ist
_w4 := Resweg_GT0 AND (SollVel+IV_RB.ErrorVel) > (ABS(IV_RB.VEL_IST));
IF _w4 THEN IV_RB.SollVel_ubrn := SollVel; END_IF
switchPhase7_2(ENBL := _w4, Phase := 7, cause := 2, IV_RB := IV_RB); // switchPhase
IF switchPhase7_2.AKT THEN RETURN; END_IF

// NETWORK 6
// Phase7 einleiten da SollVel kleiner geworden ist Beim Einleiten der Phase7 wird V_soll exackt erreicht
_w5 := Resweg_GT0 AND (Prf_Vel_Zieldiff.VE7A_inPhase7+IV_RB.HalfCyklVelDiff) <= SollVel AND (Prf_Vel_Zieldiff.VE7A_inPhase7+IV_RB.ErrorVel) >= SollVel;
IV_RB.VSoll_Ph4_ok S= _w5;
IF _w5 THEN IV_RB.SollVel_ubrn := SollVel; END_IF
switchPhase7_4(ENBL := _w5, Phase := 7, cause := 4, IV_RB := IV_RB); // switchPhase
IF switchPhase7_4.AKT THEN RETURN; END_IF

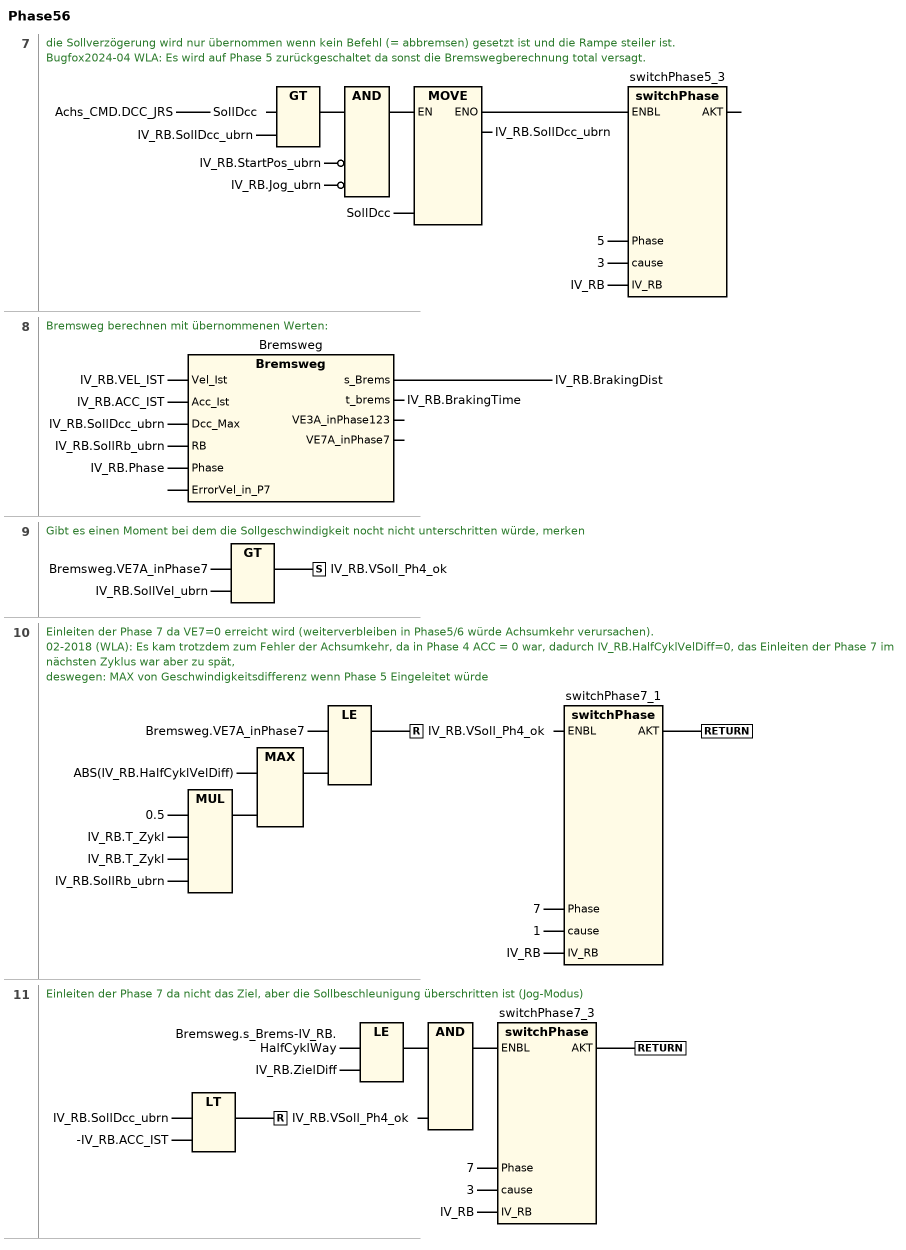
// NETWORK 7
// die Sollverzögerung wird nur übernommen wenn kein Befehl (= abbremsen) gesetzt ist und die Rampe steiler ist.
// Bugfox2024-04 WLA: Es wird auf Phase 5 zurückgeschaltet da sonst die Bremswegberechnung total versagt.
SollDcc := Achs_CMD.DCC_JRS;
_w6 := Achs_CMD.DCC_JRS > IV_RB.SollDcc_ubrn AND NOT IV_RB.StartPos_ubrn AND NOT IV_RB.Jog_ubrn;
IF _w6 THEN IV_RB.SollDcc_ubrn := SollDcc; END_IF
switchPhase5_3(ENBL := _w6, Phase := 5, cause := 3, IV_RB := IV_RB); // switchPhase

// NETWORK 8
// Bremsweg berechnen mit übernommenen Werten:
Bremsweg(
    Vel_Ist := IV_RB.VEL_IST,
    Acc_Ist := IV_RB.ACC_IST,
    Dcc_Max := IV_RB.SollDcc_ubrn,
    RB := IV_RB.SollRb_ubrn,
    Phase := IV_RB.Phase,
    t_brems => IV_RB.BrakingTime);
IV_RB.BrakingDist := Bremsweg.s_Brems;

// NETWORK 9
// Gibt es einen Moment bei dem die Sollgeschwindigkeit nocht nicht unterschritten würde, merken
IV_RB.VSoll_Ph4_ok S= Bremsweg.VE7A_inPhase7 > IV_RB.SollVel_ubrn;

// NETWORK 10
// 					Einleiten der Phase 7 da VE7=0 erreicht wird (weiterverbleiben in Phase5/6 würde Achsumkehr verursachen).
// 02-2018 (WLA): Es kam trotzdem zum Fehler der Achsumkehr, da in Phase 4 ACC = 0 war, dadurch IV_RB.HalfCyklVelDiff=0, das Einleiten der Phase 7 im nächsten Zyklus war aber zu spät,
// deswegen: MAX von Geschwindigkeitsdifferenz wenn Phase 5 Eingeleitet würde
//
_w7 := Bremsweg.VE7A_inPhase7 <= MAX(ABS(IV_RB.HalfCyklVelDiff), 0.5 * IV_RB.T_Zykl * IV_RB.T_Zykl * IV_RB.SollRb_ubrn);
IV_RB.VSoll_Ph4_ok R= _w7;
switchPhase7_1(ENBL := _w7, Phase := 7, cause := 1, IV_RB := IV_RB); // switchPhase
IF switchPhase7_1.AKT THEN RETURN; END_IF

// NETWORK 11
// Einleiten der Phase 7 da nicht das Ziel, aber die Sollbeschleunigung überschritten ist (Jog-Modus)
_w9 := (Bremsweg.s_Brems-IV_RB.HalfCyklWay) <= IV_RB.ZielDiff;
_w8 := IV_RB.SollDcc_ubrn < (-IV_RB.ACC_IST);
IV_RB.VSoll_Ph4_ok R= _w8;
switchPhase7_3(ENBL := _w9 AND _w8, Phase := 7, cause := 3, IV_RB := IV_RB); // switchPhase
IF switchPhase7_3.AKT THEN RETURN; END_IF

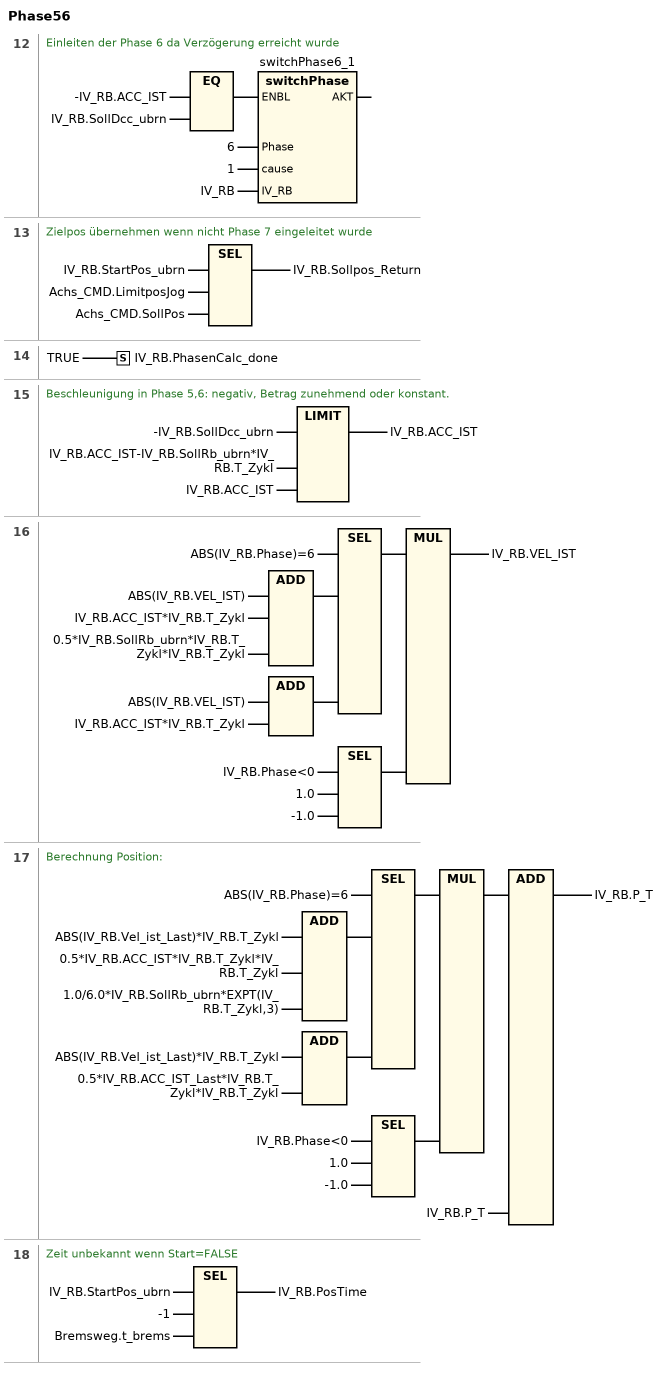
// NETWORK 12
// Einleiten der Phase 6 da Verzögerung erreicht wurde
switchPhase6_1(ENBL := (-IV_RB.ACC_IST) = IV_RB.SollDcc_ubrn, Phase := 6, cause := 1, IV_RB := IV_RB); // switchPhase

// NETWORK 13
// Zielpos übernehmen wenn nicht Phase 7 eingeleitet wurde
IV_RB.Sollpos_Return := SEL(IV_RB.StartPos_ubrn, Achs_CMD.LimitposJog, Achs_CMD.SollPos);

// NETWORK 14
IV_RB.PhasenCalc_done S= TRUE;

// NETWORK 15
// Beschleunigung in Phase 5,6: negativ, Betrag zunehmend oder konstant.
IV_RB.ACC_IST := LIMIT(-IV_RB.SollDcc_ubrn, IV_RB.ACC_IST-IV_RB.SollRb_ubrn*IV_RB.T_Zykl, IV_RB.ACC_IST);

// NETWORK 16
IV_RB.VEL_IST := SEL(ABS(IV_RB.Phase)=6, (ABS(IV_RB.VEL_IST)) + (IV_RB.ACC_IST*IV_RB.T_Zykl) + (0.5*IV_RB.SollRb_ubrn*IV_RB.T_Zykl*IV_RB.T_Zykl), (ABS(IV_RB.VEL_IST)) + (IV_RB.ACC_IST*IV_RB.T_Zykl)) * SEL(IV_RB.Phase<0, 1.0, -1.0);

// NETWORK 17
// Berechnung Position:
IV_RB.P_T := SEL(ABS(IV_RB.Phase)=6, (ABS(IV_RB.Vel_ist_Last)*IV_RB.T_Zykl) + (0.5*IV_RB.ACC_IST*IV_RB.T_Zykl*IV_RB.T_Zykl) + (1.0/6.0*IV_RB.SollRb_ubrn*EXPT(IV_RB.T_Zykl,3)), (ABS(IV_RB.Vel_ist_Last)*IV_RB.T_Zykl) + (0.5*IV_RB.ACC_IST_Last*IV_RB.T_Zykl*IV_RB.T_Zykl)) * SEL(IV_RB.Phase<0, 1.0, -1.0) + IV_RB.P_T;

// NETWORK 18
// Zeit unbekannt wenn Start=FALSE
IV_RB.PosTime := SEL(IV_RB.StartPos_ubrn, -1, Bremsweg.t_brems);

END_FUNCTION_BLOCK

// POUs/Achsen_Bausteinen/FB/Trnsf1Lreal
FUNCTION_BLOCK Trnsf1Lreal
VAR_INPUT
	ENBL: BOOL;
	IN: LREAL;
END_VAR
VAR_OUTPUT
	AKT: BOOL;
END_VAR
VAR
END_VAR
VAR_IN_OUT
	Out: LREAL;
END_VAR

IF ENBL THEN
	Out:=IN;
	AKT:=TRUE;
ELSE
	AKT:=FALSE;
END_IF

END_FUNCTION_BLOCK

// POUs/Achsen_Bausteinen/ES_AnalogIN
FUNCTION_BLOCK ES_AnalogIN (*Eil-Schleich - Achse für KL5101 - 5VGeber*)
VAR_INPUT
	DAT_FROM_PLC:TES_Achse_OUT; (*Übergabe der Parameter vom Anwenderprogramm *)
	AIN_VAL: INT;(*Istwert am Analogeingang*)

(*####################### Folgende Werte sind Regelparameter und müssen initialisiert werden##########################*)
	T_ZYKL: REAL:=0.001;(*Zykluszeit in s, in der dieser Baustein aufgerufen wird*)
	C_INVERS:BOOL:=FALSE; (*Zählrichtungsumkehr*)
	IBW:LREAL:=0.1; (*Istbewertung in mm pro Increment*)
	OPTI_KURZ:BOOL;(*optimierung bei kurzer Strecke:Ist der Verfahrweg kleiner als 2*S_SCHLEICH, dann wird auf halbem Weg beschleunugt(EIL) und auf halbem abgebremst (SCHLEICH*)
	WAITTIME_INV:REAL:=0.3;(*Wartezeit bei Richtungsumkehr in SEC*)
	WAIT_Restart_akt:BOOL;(* Wartezeit bei wiederStarten aktiv: wenn der Antrieb abgeschaltet wird, dann bleiben die Ausgänge MINDESTENS "Waittime_INV" abgeschaltet (notwendig bei 24V-DC Lineramotoren) *)
	S_SCHLEICH: REAL;(*Schleichweg*)
	S_STOP: REAL;(*Vorabschaltdifferenz, innerhalb diesem Fenster wird nicht positioniert, sondern PEH ausgegeben!*)
	T_VERZ_STILL:REAL;(*Verzögerungszeit zum Ansprechen der Stillstandsüberwachung, Sekunden*)
	IstWertOffset:LREAL;(*Offset, der  auf den Istwert(Benutzereinheit bzw. mm) Online aufgerechnent wird*)
	SSI_MAX_DIFF: DINT; (*Einheit: Incremente. Zur Überbrückung des SSI-Encoderfehlers bei Überschlag: Wenn Incremente-Sprung > SSI_MAX_DIFF, dann wird der Geberistwert eingefrohren bis wieder der richtige Wert gemeldet wird oder bis TIMEOUT überschritten ist*)
	MAX_FREESTIME_SMD_sec:REAL;(* "Ssi-Max-Differenz":Zur Überbrückung des SSI-Encoderfehlers bei Überschlag: Für maximal diese Zeit wird der Istwert eingefroren wenn er einen Sprung macht der grösser SSI_MAX_DIFF ist*)
	VEL_min:REAL;(*minimale Geschwindigkeit; bei unterschreitung dieser Geschwindigkeit für den Mess-Zeitraum "T_VERZ_STILL" wird Stillstand ausgegeben*)
	Loop_val: REAL;		(*schleife fahren: 0=nein; ansonsten: Es wird um den Betrag von S_STOP+Loop_Val vom Ziel weggefahren, abhängig vom Vorzeiche: + in pos.
							Richtung,- in neg. Richtung). Loop_val wird nur bei pos. Flanke Start oder Änderung der Sollpos bei aktivem Start ausgewertet, d.h. eine Änderung während dem Positionieren wird ignoriert*)
END_VAR
VAR_OUTPUT
	DAT_TO_PLC:TES_Achse_IN;(*Übergabe der Parameter zum Anwenderprogramm *)
	EIL_OUT:BOOL;(*Verknüpfung mit Ausgang schnell*)
	VOR_OUT:BOOL;(*Verknüpfung mit Ausgang vor*)
	ZUR_OUT:BOOL;(*Verknüpfung mit Ausgang zur*)
	ERR_INIT:BOOL:=TRUE;(*Fehler bei initialisierung oder noch nicht initialisiert*)
END_VAR

VAR

(*########################################Ausgangsvariabeln vom Baustein -> STRUKTUR(IN) ###################################*)
	IstPos: LREAL;(*Istposition Achse *)
	SYNC: BOOL := FALSE;
	PEH:BOOL;

(*####################################Folgende Daten werden intern berechnet und verwendet#####################################*)
	OFFSET_INC: LREAL;
	COUNT_INC: DINT;(*Zähler-INCREMENTE*)
	COUNT_INC_LAST: DINT;(*Zähler-INCREMENTE des letzten Zyklus, sofern Zähler-Val gültig war*)
	V_SOLL:REAL;(*Sollgeschwindifkeit, die aufgrund der berechnungen resultiert.V_F_T wird durch V_Soll UND den zulässigen Rampen (zulässige Geschw.-Änderung pro Zyklus) berechnet*)
	Zieldiff_Pos: LREAL;(*POS-Modus: Differenz zum Ziel*)
	Start_Pos_LAST: BOOL;
	SollPos: LREAL;(*Zielposition bei Positionierung*)
	TIME_VOR: REAL;
	TIME_ZUR: REAL;
	StartFRG_Pos: BOOL;
	S_SCHLEICH_I: REAL;(*Schleichweg, Intern. Der Wert S_SCHLEICH (VAR_INPUT) wird auf S_SCHLEICH_I kopiert, außer bei optimierung für kurze Strecken *)
	T_STILLST: REAL;(* abgelaufene Stillstandszeit*)
	SetIstPos: BOOL;
	IstPos_LAST: LREAL;
	IstWertOffset_LAST: LREAL;
	TIMECOUNT_SMD: LREAL;
	Vel_meas: REAL;		(*gemessene geschwindigkeit zwischen 2 Istwertmessungen im Zeitabstand von "T_VERZ_STILL"*)
	VOR_OUT_LAST: BOOL;
	ZUR_OUT_LAST: BOOL;
	IstPos_MEM: LREAL;
	Loop_akt: BOOL;(*Schleife-fahren ist aktiv*)
	c_Loop_val: REAL;(* Kopie von LoopVAL*)
END_VAR

SetIstPos:=FALSE;
(*Kontrolle der Parameter*)
IF T_ZYKL<=0 OR IBW<=0 THEN
	ERR_INIT:=TRUE;VOR_OUT:=FALSE;ZUR_OUT:=FALSE;EIL_OUT:=FALSE;RETURN;(*Regelparameter ungültig,Ausgänge abschalten*)
ELSE ERR_INIT:=FALSE;
END_IF
(*###################### ENDE INIT #####################################################*)

(* Zähler invertieren wenn INV=1*)
IF C_INVERS THEN COUNT_INC:=-AIN_VAL;ELSE COUNT_INC:=AIN_VAL;END_IF

IF ABS (COUNT_INC-COUNT_INC_LAST) > SSI_MAX_DIFF AND TIMECOUNT_SMD<MAX_FREESTIME_SMD_sec THEN
	(*Der Istwertsprung des SSI-Gebers ist > der angegebenen Differenz und die maximale Frierzeit ist noch nicht abgelaufen. Für die Angegebene Zeit wird der Istwert eingefrohren bzw. dem Sollwert nachgeführt*)
	TIMECOUNT_SMD:=TIMECOUNT_SMD+T_ZYKL; (*Zählen der laufeneden Frier-Zeit*)
ELSE (*Istwertberechnung ausführen, denn SSI_MAX_DIFF ist nicht überschritten oder MAX_FREESTIME_SMD ist abgelaufen*)
	TIMECOUNT_SMD:=0; (*Zeitzähler nullen*)
	(*Freese bei ONLINE-Istwertoffsetänderung, damit sich die Position des Antriebes nicht mechanisch verändert*)

	(* Ermittlung des Geberistwertes *)
	IstPos:=(COUNT_INC+OFFSET_INC)*IBW+IstWertOffset;
	IstWertOffset_LAST:=IstWertOffset;
	COUNT_INC_LAST:=COUNT_INC; (*COUNT_INC_LAST zuweisen*)
END_IF



(* Ermittlung des Geberistwertes *)
IstPos:=(COUNT_INC+OFFSET_INC)*IBW+IstWertOffset;



(*Stillstandsüberwachung*)
IF T_VERZ_STILL<=0 THEN
	;(*ende wegen DIV/0*)

ELSIF (VOR_OUT AND VOR_OUT_LAST) OR (ZUR_OUT AND ZUR_OUT_LAST) THEN (*fährt seit mehr als 2Zyklen in selbe Richtung*)
	T_STILLST:=T_STILLST + T_ZYKL;(*Zeitmessung läuft*)

	IF T_STILLST>T_VERZ_STILL THEN (*Periodenzeit zur geschwindigkeitsmessung ist abgelaufen: Geschwindigkeitsmessung machen*)
		vel_meas:=LREAL_TO_REAL((IstPos-IstPos_MEM)/T_STILLST);(*Geschwindigkeit messen*)
		DAT_TO_PLC.STILL:=ABS(Vel_meas)<VEL_MIN; (*Stillstandsüberwachungszeit abgelaufen ?->SET Stillstand*)
		T_STILLST:=0; (*Zeit wieder nullen um neue Periodenmessung zu machen*)
		IstPos_MEM:=IstPos;(*neue Istposition merken für nächste Messung*)
	END_IF

ELSE
	T_STILLST:=0;
	IstPos_MEM:=IstPos;
	DAT_TO_PLC.STILL:=FALSE;
END_IF




































(*############################## Achsen-Steuerung ##############################################################*)
PEH:=FALSE; (*PEH mit FALSE initialisieren*)

(*########################## Positionieren auf Sollposition######################################*)
(*POSITIONIEREN POSITIONIEREN POSITIONIEREN POSITIONIEREN POSITIONIEREN POSITIONIEREN POSITIONIEREN POSITIONIEREN *)
IF DAT_FROM_PLC.Start_Pos THEN
	Zieldiff_Pos:=DAT_FROM_PLC.Sollpos-IstPos;(*Reelle momentane Differenz zum Ziel*)
	IF NOT Start_Pos_LAST OR Sollpos<>DAT_FROM_PLC.Sollpos THEN (*Flanke Start oder änderung der Sollposition: Werte übergeben*)
		c_Loop_val:=Loop_val; (*Loop-Val speichern, wird während dem Positionieren ignoriert*)
		Loop_akt:=ABS(c_Loop_val) <>0 AND ABS(Zieldiff_Pos)<(S_STOP+ABS(c_Loop_val));
		SollPos:=DAT_FROM_PLC.Sollpos;DAT_TO_PLC.RET_SollPos:=Sollpos;StartFRG_Pos:=TRUE;(*Setzen der Startfreigabe*)
		IF OPTI_KURZ AND ABS(Zieldiff_Pos)<(2*S_SCHLEICH) THEN S_SCHLEICH_I:=LREAL_TO_REAL(ABS(Zieldiff_Pos)/2)+S_STOP;
		ELSE S_SCHLEICH_I:=S_SCHLEICH;
		END_IF
	END_IF

	IF ABS(Zieldiff_Pos)>(S_STOP+ABS(c_Loop_val)) THEN
		Loop_akt:=FALSE;
	END_IF

	IF Loop_akt THEN
		IF StartFRG_Pos THEN
			IF c_Loop_val > 0 THEN (*vorwärts schleife fahren*)
				V_SOLL:=1; (*langsam vor*)
			ELSE (*rückwärts schleife fahren*)
				V_SOLL:=-1; (*langsam zur*)
			END_IF
		ELSE
			V_SOLL:=0; (*keine Startfreigabe (Positionierung bereits ausgeführt), also STOP*)
		END_IF

	ELSIF ABS(Zieldiff_Pos)>S_STOP THEN (*Positionieren, STOP-Fenster noch nicht erreicht*)
		IF StartFRG_Pos THEN
			IF Zieldiff_Pos > 0 THEN (*vorwärts positionieren*)
				IF Zieldiff_Pos > S_SCHLEICH_I AND DAT_FROM_PLC.V_Pos>1 THEN V_SOLL:=2; (*schnell vor*)
				ELSE V_SOLL:=1; (*langsam vor*)
				END_IF
			ELSE (*rückwärts positionieren*)
				IF -Zieldiff_Pos > S_SCHLEICH_I AND DAT_FROM_PLC.V_Pos>1 THEN V_SOLL:=-2; (*schnell zurück*)
				ELSE V_SOLL:=-1; (*langsam zurück*)
				END_IF
			END_IF
		ELSE
			V_SOLL:=0; (*keine Startfreigabe (Positionierung bereits ausgeführt), also STOP*)
		END_IF
	ELSE  (*S_STOP-Fenster bereits erreicht*)
		PEH:=TRUE;
		V_SOLL:=0;
		StartFRG_Pos:=FALSE;
	END_IF


(*################### JOG-Betrieb mit konstanter Geschwindigkeit ohne Startrampe ###################*)
(* JOG JOG JOG JOG JOG JOG JOG JOG JOG JOG JOG JOG JOG JOG JOG JOG JOG JOG JOG JOG JOG JOG JOG JOG JOG JOG JOG *)
ELSIF DAT_FROM_PLC.JOGFW THEN
	V_SOLL:=DAT_FROM_PLC.V_JOG;

ELSIF DAT_FROM_PLC.JOGBW THEN
	V_SOLL:=-DAT_FROM_PLC.V_JOG;

(*####################### Anhalten, keine Bedingung erfüllt##########################################*)
(* HALT HALT HALT HALT HALT HALT HALT HALT HALT HALT HALT HALT HALT HALT HALT HALT HALT HALT HALT HALT HALT HALT *)
ELSE V_SOLL:=0;
END_IF


(*########## Berechnung der Ausgänge ###############*)
IF V_SOLL > 0 THEN (*Sollgeschwindigkeit vor*)
	IF TIME_ZUR=0 AND (TIME_VOR=0 OR  NOT WAIT_Restart_akt OR VOR_OUT) THEN (*keine Richtungsumkehr, rückwärts-Wartezeit ist abgelaufen UND keine wartezeit Restart oder abgelaufen oder fährt bereits*)
		(*positionieren vor*)
		TIME_VOR:=WAITTIME_INV;(*Wartezeit laden*)
		IF V_SOLL=2 THEN DAT_TO_PLC.VEL_IST:=2;
		ELSE DAT_TO_PLC.VEL_IST:=1;
		END_IF
	ELSE (*Rückwärts-Wartezeit läuft noch*)
		DAT_TO_PLC.VEL_IST:=0;
	END_IF
ELSIF V_SOLL < 0 THEN(*Sollgeschwindigkeit negativ*)
	IF TIME_VOR=0 AND (TIME_ZUR=0 OR  NOT WAIT_Restart_akt OR ZUR_OUT) THEN (*keine Richtungsumkehr, vorwärts-Wartezeit ist abgelaufen UND keine wartezeit Restart oder abgelaufen oder fährt bereits*)
		(*positionieren zurück*)
		TIME_ZUR:=WAITTIME_INV;(*Wartezeit "zurück" laden*)
		IF V_SOLL=-2 THEN DAT_TO_PLC.VEL_IST:=-2;
		ELSE DAT_TO_PLC.VEL_IST:=-1;
		END_IF
	ELSE (*vorwärts-Wartezeit läuft noch*)
		DAT_TO_PLC.VEL_IST:=0;
	END_IF
ELSE (*Sollgeschwindigkeit = 0, also STOP*)
	DAT_TO_PLC.VEL_IST:=0;
END_IF
(*Wartezeit decrementieren*)
TIME_VOR:=MAX((TIME_VOR-T_ZYKL),0);TIME_ZUR:=MAX((TIME_ZUR-T_ZYKL),0);
(*Zyklusverz. Var.*)
COUNT_INC_LAST:=COUNT_INC;
Start_Pos_LAST:=DAT_FROM_PLC.Start_Pos;

(*Ausgangsvariablen übergeben*)
DAT_TO_PLC.IstPos:=IstPos;
DAT_TO_PLC.SYNC:=SYNC;
DAT_TO_PLC.PEH:=PEH;
(*Ausgänge setzen*)
VOR_OUT:=DAT_TO_PLC.VEL_IST>0;
ZUR_OUT:=DAT_TO_PLC.VEL_IST<0;
EIL_OUT:=ABS(DAT_TO_PLC.VEL_IST)>=2;

IstPos_Last:=IstPos;
VOR_OUT_LAST:=VOR_OUT;
ZUR_OUT_LAST:=ZUR_OUT;

END_FUNCTION_BLOCK

// POUs/Achsen_Bausteinen/ES_EL5001_A
FUNCTION_BLOCK ES_EL5001_A(*Eil-Schleich - Achse für ES5001*)
VAR_INPUT
	COUNT_VAL: DWORD;(*Zähler-INCREMENTE*)
	DAT_FROM_PLC:TES_Achse_OUT; (*Übergabe der Parameter vom Anwenderprogramm *)

(*####################### Folgende Werte sind Regelparameter und müssen initialisiert werden##########################*)
	T_ZYKL: REAL:=0.001;(*Zykluszeit in s, in der dieser Baustein aufgerufen wird*)
	C_INVERS:BOOL:=FALSE; (*Zählrichtungsumkehr*)
	IBW:LREAL:=0.1; (*Istbewertung in mm pro Increment*)
	OPTI_KURZ:BOOL;(*optimierung bei kurzer Strecke:Ist der Verfahrweg kleiner als 2*S_SCHLEICH, dann wird auf halbem Weg beschleunugt(EIL) und auf halbem abgebremst (SCHLEICH*)
	WAITTIME_INV:REAL:=0.3;(*Wartezeit bei Richtungsumkehr in SEC*)
	S_SCHLEICH: REAL;(*Schleichweg*)
	S_STOP: REAL;(*Vorabschaltdifferenz, innerhalb diesem Fenster wird nicht positioniert, sondern PEH ausgegeben!*)
	T_VERZ_STILL:REAL;(*Verzögerungszeit zum Ansprechen der Stillstandsüberwachung, Sekunden*)
	IstWertOffset:LREAL;(*Offset, der  auf den Istwert(Benutzereinheit bzw. mm) Online aufgerechnent wird*)
	SSI_MAX_DIFF: DINT; (*Einheit: Incremente. Zur Überbrückung des SSI-Encoderfehlers bei Überschlag: Wenn Incremente-Sprung > SSI_MAX_DIFF, dann wird der Geberistwert eingefrohren bis wieder der richtige Wert gemeldet wird oder bis TIMEOUT überschritten ist*)
	MAX_FREESTIME_SMD_sec: REAL;(* "Ssi-Max-Differenz":Zur Überbrückung des SSI-Encoderfehlers bei Überschlag: Für maximal diese Zeit wird der Istwert eingefroren wenn er einen Sprung macht der grösser SSI_MAX_DIFF ist*)
	Loop_val: REAL;		(*schleife fahren: 0=nein; ansonsten: Es wird um den Betrag von S_STOP+Loop_Val vom Ziel weggefahren, abhängig vom Vorzeiche: + in pos.
							Richtung,- in neg. Richtung). Loop_val wird nur bei pos. Flanke Start oder Änderung der Sollpos bei aktivem Start ausgewertet, d.h. eine Änderung während dem Positionieren wird ignoriert*)
	IWTyp: REAL;(*Istwert Typisch: Dieser Wert ist Notwendig, um den Geberüberschlag intern ausserhalb dem typischen Istwert zu verschieben, er kann
				 mit0 (oder gar nicht = 0) parametriert werden. Nur in Sonderfällen, wo aufgrund einem hohen Verfahrweg der gesamte Geberbereich abgefahren wird, kann es notwendig sein, einen korrekten Wert anzugeben. In 
				diesem fall ist der Mittelwert zwischen Minpos und Maxpos anzugeben; eine Achse, die in diesem Fall z.B. von +20000mm bis +60000 mm verfährt, muss dann mit +40000 parametriert werden. Die maximale Anzahl der möglichen Incremente des Gebers sollte
				auf jeden Fall kontrolliert werden.*)
	Geber24Bit:BOOL;(* Es ist ein Geber angeschlossen, der nur 24-Bit liefert, d.h. der Überschlag des Gebers erfolgt nach 24 Bits: 16#00FF_FFFF -> 16#0000_0000*)
END_VAR
VAR_OUTPUT
	DAT_TO_PLC:TES_Achse_IN;(*Übergabe der Parameter zum Anwenderprogramm *)
	EIL_OUT:BOOL;(*Verknüpfung mit Ausgang schnell*)
	VOR_OUT:BOOL;(*Verknüpfung mit Ausgang vor*)
	ZUR_OUT:BOOL;(*Verknüpfung mit Ausgang zur*)
	ERR_INIT:BOOL:=TRUE;(*Fehler bei initialisierung oder noch nicht initialisiert*)
END_VAR

VAR

(*########################################Ausgangsvariabeln vom Baustein -> STRUKTUR(IN) ###################################*)
	IstPos: LREAL;(*Istposition Achse *)
	SYNC: BOOL := FALSE;
	PEH:BOOL;

(*####################################Folgende Daten werden intern berechnet und verwendet#####################################*)
	COUNT_INC: DINT;(*Zähler-INCREMENTE*)
	COUNT_INC_LAST: DINT;(*Zähler-INCREMENTE des letzten Zyklus, sofern Zähler-Val gültig war*)
	V_SOLL:REAL;(*Sollgeschwindifkeit, die aufgrund der berechnungen resultiert.V_F_T wird durch V_Soll UND den zulässigen Rampen (zulässige Geschw.-Änderung pro Zyklus) berechnet*)
	Zieldiff_Pos: LREAL;(*POS-Modus: Differenz zum Ziel*)
	Start_Pos_LAST: BOOL;
	SollPos: LREAL;(*Zielposition bei Positionierung*)
	TIME_VOR: REAL;
	TIME_ZUR: REAL;
	StartFRG_Pos: BOOL;
	S_SCHLEICH_I: REAL;(*Schleichweg, Intern. Der Wert S_SCHLEICH (VAR_INPUT) wird auf S_SCHLEICH_I kopiert, außer bei optimierung für kurze Strecken *)
	T_STILLST: REAL;(* abgelaufene Stillstandszeit*)
	SetIstPos: BOOL;
	IstPos_LAST: LREAL;
	IstWertOffset_LAST: LREAL;
	TIMECOUNT_SMD: LREAL;
	Loop_akt: BOOL;(*Schleife-fahren ist aktiv*)
	c_Loop_val: REAL;(* Kopie von LoopVAL*)
	IncOffset: DINT;
	IBW2: LREAL;
END_VAR

SetIstPos:=FALSE;
(*Kontrolle der Parameter*)
IF T_ZYKL<=0 OR IBW<=0 THEN
	ERR_INIT:=TRUE;VOR_OUT:=FALSE;ZUR_OUT:=FALSE;EIL_OUT:=FALSE;RETURN;(*Regelparameter ungültig,Ausgänge abschalten*)
ELSE ERR_INIT:=FALSE;
END_IF
(*###################### ENDE INIT #####################################################*)

DAT_TO_PLC.STILL:=FALSE;(*Stillstand mit FALSE init.*)

IF Geber24Bit THEN
	COUNT_VAL:=SHL(COUNT_VAL,8);
	IBW2:=IBW/256;
ELSE
	IBW2:=IBW;
END_IF


IncOffset:=LREAL_TO_DINT((IstWertOffset-IWTyp)/IBW2)+DWORD_TO_DINT(16#8000_0000);(*Der Istwertoffset, der Betrag der Typschen Position und die Hälfte des Gesamt-Icnremente-Bereichs müssen aufgerechnet werden, damit kein Überschlag möglich ist*)
IF C_INVERS THEN
	COUNT_INC:=DWORD_TO_DINT(16#FFFF_FFFF) - (DWORD_TO_DINT(COUNT_VAL)-IncOffset);
ELSE
	COUNT_INC:=DWORD_TO_DINT(Count_Val)+IncOffset;
END_IF

(*Stillstandsüberwachung*)
IF (VOR_OUT AND (COUNT_INC<=COUNT_INC_LAST)) OR (ZUR_OUT AND (COUNT_INC>=COUNT_INC_LAST)) THEN
	T_STILLST:=T_STILLST + T_ZYKL;
	DAT_TO_PLC.STILL:=T_STILLST>T_VERZ_STILL; (*Stillstandsüberwachungszeit abgelaufen ?->SET Stillstand*)
ELSE
	T_STILLST:=0;
END_IF

IF ABS (COUNT_INC-COUNT_INC_LAST) > SSI_MAX_DIFF AND TIMECOUNT_SMD<MAX_FREESTIME_SMD_sec THEN
	(*Der Istwertsprung des SSI-Gebers ist > der angegebenen Differenz und die maximale Frierzeit ist noch nicht abgelaufen. Für die Angegebene Zeit wird der Istwert eingefrohren bzw. dem Sollwert nachgeführt*)
	TIMECOUNT_SMD:=TIMECOUNT_SMD+T_ZYKL; (*Zählen der laufeneden Frier-Zeit*)
ELSE (*Istwertberechnung ausführen, denn SSI_MAX_DIFF ist nicht überschritten oder MAX_FREESTIME_SMD ist abgelaufen*)
	TIMECOUNT_SMD:=0; (*Zeitzähler nullen*)
	(*Freese bei ONLINE-Istwertoffsetänderung, damit sich die Position des Antriebes nicht mechanisch verändert*)

	(* Ermittlung des Geberistwertes *)
	IstPos:=DINT_TO_LREAL(COUNT_INC-DWORD_TO_DINT(16#8000_0000))*IBW2+IWTyp;(* Der Istwertoffset ist bereits den Incrementwert aufgerechnet, der halbe Gesamtincrement-Bereich und der Typ.Istwert, die ebenfalls aufgerechnet wurden, müss hier wieder abgerechnet werden: 2147483648 D = 16#8000_0000 H*)
	IstWertOffset_LAST:=IstWertOffset;
	COUNT_INC_LAST:=COUNT_INC; (*COUNT_INC_LAST zuweisen*)
END_IF



















































(*############################## Achsen-Steuerung ##############################################################*)
PEH:=FALSE; (*PEH mit FALSE initialisieren*)

(*########################## Positionieren auf Sollposition######################################*)
(*POSITIONIEREN POSITIONIEREN POSITIONIEREN POSITIONIEREN POSITIONIEREN POSITIONIEREN POSITIONIEREN POSITIONIEREN *)
IF DAT_FROM_PLC.Start_Pos THEN
	Zieldiff_Pos:=DAT_FROM_PLC.Sollpos-IstPos;(*Reelle momentane Differenz zum Ziel*)
	IF NOT Start_Pos_LAST OR Sollpos<>DAT_FROM_PLC.Sollpos THEN (*Flanke Start oder änderung der Sollposition: Werte übergeben*)
		c_Loop_val:=Loop_val; (*Loop-Val speichern, wird während dem Positionieren ignoriert*)
		Loop_akt:=ABS(c_Loop_val) <>0 AND ABS(Zieldiff_Pos)<(S_STOP+ABS(c_Loop_val));
		SollPos:=DAT_FROM_PLC.Sollpos;DAT_TO_PLC.RET_SollPos:=Sollpos;StartFRG_Pos:=TRUE;(*Setzen der Startfreigabe*)
		IF OPTI_KURZ AND ABS(Zieldiff_Pos)<(2*S_SCHLEICH) THEN S_SCHLEICH_I:=LREAL_TO_REAL(ABS(Zieldiff_Pos)/2)+S_STOP;
		ELSE S_SCHLEICH_I:=S_SCHLEICH;
		END_IF
	END_IF

	IF ABS(Zieldiff_Pos)>(S_STOP+ABS(c_Loop_val)) THEN
		Loop_akt:=FALSE;
	END_IF

	IF Loop_akt THEN
		IF StartFRG_Pos THEN
			IF c_Loop_val > 0 THEN (*vorwärts schleife fahren*)
				V_SOLL:=1; (*langsam vor*)
			ELSE (*rückwärts schleife fahren*)
				V_SOLL:=-1; (*langsam zur*)
			END_IF
		ELSE
			V_SOLL:=0; (*keine Startfreigabe (Positionierung bereits ausgeführt), also STOP*)
		END_IF

	ELSIF ABS(Zieldiff_Pos)>S_STOP THEN (*Positionieren, STOP-Fenster noch nicht erreicht*)
		IF StartFRG_Pos THEN
			IF Zieldiff_Pos > 0 THEN (*vorwärts positionieren*)
				IF Zieldiff_Pos > S_SCHLEICH_I AND DAT_FROM_PLC.V_Pos>1 THEN V_SOLL:=2; (*schnell vor*)
				ELSE V_SOLL:=1; (*langsam vor*)
				END_IF
			ELSE (*rückwärts positionieren*)
				IF -Zieldiff_Pos > S_SCHLEICH_I AND DAT_FROM_PLC.V_Pos>1 THEN V_SOLL:=-2; (*schnell zurück*)
				ELSE V_SOLL:=-1; (*langsam zurück*)
				END_IF
			END_IF
		ELSE
			V_SOLL:=0; (*keine Startfreigabe (Positionierung bereits ausgeführt), also STOP*)
		END_IF
	ELSE  (*S_STOP-Fenster bereits erreicht*)
		PEH:=TRUE;
		V_SOLL:=0;
		StartFRG_Pos:=FALSE;
	END_IF


(*################### JOG-Betrieb mit konstanter Geschwindigkeit ohne Startrampe ###################*)
(* JOG JOG JOG JOG JOG JOG JOG JOG JOG JOG JOG JOG JOG JOG JOG JOG JOG JOG JOG JOG JOG JOG JOG JOG JOG JOG JOG *)
ELSIF DAT_FROM_PLC.JOGFW THEN
	V_SOLL:=DAT_FROM_PLC.V_JOG;

ELSIF DAT_FROM_PLC.JOGBW THEN
	V_SOLL:=-DAT_FROM_PLC.V_JOG;

(*####################### Anhalten, keine Bedingung erfüllt##########################################*)
(* HALT HALT HALT HALT HALT HALT HALT HALT HALT HALT HALT HALT HALT HALT HALT HALT HALT HALT HALT HALT HALT HALT *)
ELSE V_SOLL:=0;
END_IF


(*########## Berechnung der Ausgänge ###############*)
IF V_SOLL > 0 THEN (*Sollgeschwindigkeit vor*)
	IF TIME_ZUR=0 THEN (*keine Richtungsumkehr, rückwärts-Wartezeit ist abgelaufen*)
		(*positionieren vor*)
		TIME_VOR:=WAITTIME_INV;(*Wartezeit laden*)
		IF V_SOLL=2 THEN DAT_TO_PLC.VEL_IST:=2;
		ELSE DAT_TO_PLC.VEL_IST:=1;
		END_IF
	ELSE (*Rückwärts-Wartezeit läuft noch*)
		DAT_TO_PLC.VEL_IST:=0;
	END_IF
ELSIF V_SOLL < 0 THEN(*Sollgeschwindigkeit negativ*)
	IF TIME_VOR=0 THEN (*keine Richtungsumkehr, vorwärts-Wartezeit ist abgelaufen*)
		(*positionieren zurück*)
		TIME_ZUR:=WAITTIME_INV;(*Wartezeit "zurück" laden*)
		IF V_SOLL=-2 THEN DAT_TO_PLC.VEL_IST:=-2;
		ELSE DAT_TO_PLC.VEL_IST:=-1;
		END_IF
	ELSE (*vorwärts-Wartezeit läuft noch*)
		DAT_TO_PLC.VEL_IST:=0;
	END_IF
ELSE (*Sollgeschwindigkeit = 0, also STOP*)
	DAT_TO_PLC.VEL_IST:=0;
END_IF
(*Wartezeit decrementieren*)
TIME_VOR:=MAX((TIME_VOR-T_ZYKL),0);TIME_ZUR:=MAX((TIME_ZUR-T_ZYKL),0);
(*Zyklusverz. Var.*)

Start_Pos_LAST:=DAT_FROM_PLC.Start_Pos;

(*Ausgangsvariablen übergeben*)
DAT_TO_PLC.IstPos:=IstPos;
DAT_TO_PLC.SYNC:=SYNC;
DAT_TO_PLC.PEH:=PEH;
(*Ausgänge setzen*)
VOR_OUT:=DAT_TO_PLC.VEL_IST>0;
ZUR_OUT:=DAT_TO_PLC.VEL_IST<0;
EIL_OUT:=ABS(DAT_TO_PLC.VEL_IST)>=2;
IstPos_Last:=IstPos;

END_FUNCTION_BLOCK

// POUs/Achsen_Bausteinen/ES_EL5xx1_A
FUNCTION_BLOCK ES_EL5xx1_A(*Eil-Schleich - Achse für EL5xx1*)
VAR_INPUT
	DAT_FROM_PLC:TES_Achse_OUT; (*Übergabe der Parameter vom Anwenderprogramm *)
	counter_bits:INT:=16;(*Anzahl der Bits die ein Counter verwendet*)
	COUNT_VAL: DINT;(*Verknüpfung mit COUNTER VAL*)
	COUNT_LATCH: DWORD;(*Verknüpfung mit COUNTER LATCH*)
	COUNT_STATE: BYTE;(*Verknüpfung mit COUNTER STATE*)
	EREF: BOOL; (*Verknüpfung mit Referenzeingang*)

